REGION Network 20: CHANGE TO BA3 MODE ALARM
   RUNG wire#powerrail
      Contact( #MODE_GROUP_BA_DB.BA3_REQUEST )
      Contact( #ANY_MCH_CYCLE_RUN )
      wire#w1
      I_Contact( #MODE_GROUP_BA_DB.CHANGE_TO_BA1_ALARM )
      I_Contact( #MODE_GROUP_BA_DB.CHANGE_TO_BA2_ALARM )
      I_Contact( #MODE_GROUP_BA_DB.CHANGE_TO_BA5_ALARM )
      Contact( #O_BYTE_0.CHANGE_MODE_SEOC_ALARM )
      wire#w2
      Coil( #MODE_GROUP_BA_DB.CHANGE_TO_BA3_ALARM )
   END_RUNG
   RUNG wire#powerrail
      Contact( #MODE_GROUP_BA_DB.CHANGE_TO_BA3_ALARM )
      I_Contact( #MCH_RESET_FAULTS )
   END_RUNG wire#w1
   RUNG wire#w2
      Coil( #CHANGE_TO_BA3_MODE_WRN )
   END_RUNG
   // the same network as SCL:
   #MODE_GROUP_BA_DB.CHANGE_TO_BA3_ALARM := ((#MODE_GROUP_BA_DB.BA3_REQUEST AND #ANY_MCH_CYCLE_RUN) OR (#MODE_GROUP_BA_DB.CHANGE_TO_BA3_ALARM AND NOT #MCH_RESET_FAULTS)) AND NOT #MODE_GROUP_BA_DB.CHANGE_TO_BA1_ALARM AND NOT #MODE_GROUP_BA_DB.CHANGE_TO_BA2_ALARM AND NOT #MODE_GROUP_BA_DB.CHANGE_TO_BA5_ALARM AND #O_BYTE_0.CHANGE_MODE_SEOC_ALARM;
   #CHANGE_TO_BA3_MODE_WRN := #MODE_GROUP_BA_DB.CHANGE_TO_BA3_ALARM;
END_REGION

REGION Network 21: CHANGE TO BA5 MODE ALARM
   RUNG wire#powerrail
      Contact( #MODE_GROUP_BA_DB.BA5_REQUEST )
      Contact( #ANY_MCH_CYCLE_RUN )
      wire#w1
      I_Contact( #MODE_GROUP_BA_DB.CHANGE_TO_BA1_ALARM )
      I_Contact( #MODE_GROUP_BA_DB.CHANGE_TO_BA2_ALARM )
      I_Contact( #MODE_GROUP_BA_DB.CHANGE_TO_BA3_ALARM )
      Contact( #O_BYTE_0.CHANGE_MODE_SEOC_ALARM )
      wire#w2
      Coil( #MODE_GROUP_BA_DB.CHANGE_TO_BA5_ALARM )
   END_RUNG
   RUNG wire#powerrail
      Contact( #MODE_GROUP_BA_DB.CHANGE_TO_BA5_ALARM )
      I_Contact( #MCH_RESET_FAULTS )
   END_RUNG wire#w1
   RUNG wire#w2
      Coil( #CHANGE_TO_BA5_MODE_WRN )
   END_RUNG
   // the same network as SCL:
   #MODE_GROUP_BA_DB.CHANGE_TO_BA5_ALARM := ((#MODE_GROUP_BA_DB.BA5_REQUEST AND #ANY_MCH_CYCLE_RUN) OR (#MODE_GROUP_BA_DB.CHANGE_TO_BA5_ALARM AND NOT #MCH_RESET_FAULTS)) AND NOT #MODE_GROUP_BA_DB.CHANGE_TO_BA1_ALARM AND NOT #MODE_GROUP_BA_DB.CHANGE_TO_BA2_ALARM AND NOT #MODE_GROUP_BA_DB.CHANGE_TO_BA3_ALARM AND #O_BYTE_0.CHANGE_MODE_SEOC_ALARM;
   #CHANGE_TO_BA5_MODE_WRN := #MODE_GROUP_BA_DB.CHANGE_TO_BA5_ALARM;
END_REGION

REGION Network 22: STOP END OF CYCLE WARNINGS
   RUNG wire#powerrail
      I_Contact( #MODE_GROUP_BA_DB.CHANGE_TO_BA1_ALARM )
      I_Contact( #MODE_GROUP_BA_DB.CHANGE_TO_BA2_ALARM )
      I_Contact( #MODE_GROUP_BA_DB.CHANGE_TO_BA3_ALARM )
      I_Contact( #MODE_GROUP_BA_DB.CHANGE_TO_BA5_ALARM )
      Not()
      { S7_GenerateENO := "TRUE" } Move(in := #DB_NUMBER, out1 => "DB440_MACHINE_ALARM_DECODING".GLOBAL_ALARMS_MACHINE.ALARM_DECODING)
      S_Coil( "DB440_MACHINE_ALARM_DECODING".ALARMS_CENTRAL.SEOC_WARNING )
   END_RUNG
   // the same network as SCL:
   // ENO of a box is taken as its EN; it also drops when the box reports an error
   IF NOT (NOT #MODE_GROUP_BA_DB.CHANGE_TO_BA1_ALARM AND NOT #MODE_GROUP_BA_DB.CHANGE_TO_BA2_ALARM AND NOT #MODE_GROUP_BA_DB.CHANGE_TO_BA3_ALARM AND NOT #MODE_GROUP_BA_DB.CHANGE_TO_BA5_ALARM) THEN
       "DB440_MACHINE_ALARM_DECODING".GLOBAL_ALARMS_MACHINE.ALARM_DECODING := #DB_NUMBER;
       "DB440_MACHINE_ALARM_DECODING".ALARMS_CENTRAL.SEOC_WARNING := TRUE;
   END_IF;
END_REGION

REGION Network 23: WARNINGS
   RUNG wire#powerrail
      I_Contact( #MODE_GROUP_BA_DB.NO_BA_SELECTED )
      Not()
      Move(in := #DB_NUMBER, out1 => "DB440_MACHINE_ALARM_DECODING".GLOBAL_ALARMS_MACHINE.WARNING_DECODING)
      wire#w1
      S_Coil( "DB440_MACHINE_ALARM_DECODING".ALARMS_CENTRAL.WARNING )
   END_RUNG
   RUNG wire#w1
      N_Trig( #MODE_GROUP_BA_DB.WARNING_GONE )
      Move(in := 0, out1 => "DB440_MACHINE_ALARM_DECODING".GLOBAL_ALARMS_MACHINE.WARNING_DECODING)
      R_Coil( "DB440_MACHINE_ALARM_DECODING".ALARMS_CENTRAL.WARNING )
   END_RUNG
   // the same network as SCL:
   #_w1 := NOT (NOT #MODE_GROUP_BA_DB.NO_BA_SELECTED);
   IF #_w1 THEN
       "DB440_MACHINE_ALARM_DECODING".GLOBAL_ALARMS_MACHINE.WARNING_DECODING := #DB_NUMBER;
       "DB440_MACHINE_ALARM_DECODING".ALARMS_CENTRAL.WARNING := TRUE;
   END_IF;
   #_w2 := NOT #_w1 AND #MODE_GROUP_BA_DB.WARNING_GONE;   // falling edge
   #MODE_GROUP_BA_DB.WARNING_GONE := #_w1;
   IF #_w2 THEN
       "DB440_MACHINE_ALARM_DECODING".GLOBAL_ALARMS_MACHINE.WARNING_DECODING := 0;
       "DB440_MACHINE_ALARM_DECODING".ALARMS_CENTRAL.WARNING := FALSE;
   END_IF;
END_REGION

REGION Network 24: CHANGE MODE GENERAL CONDITIONS HELP
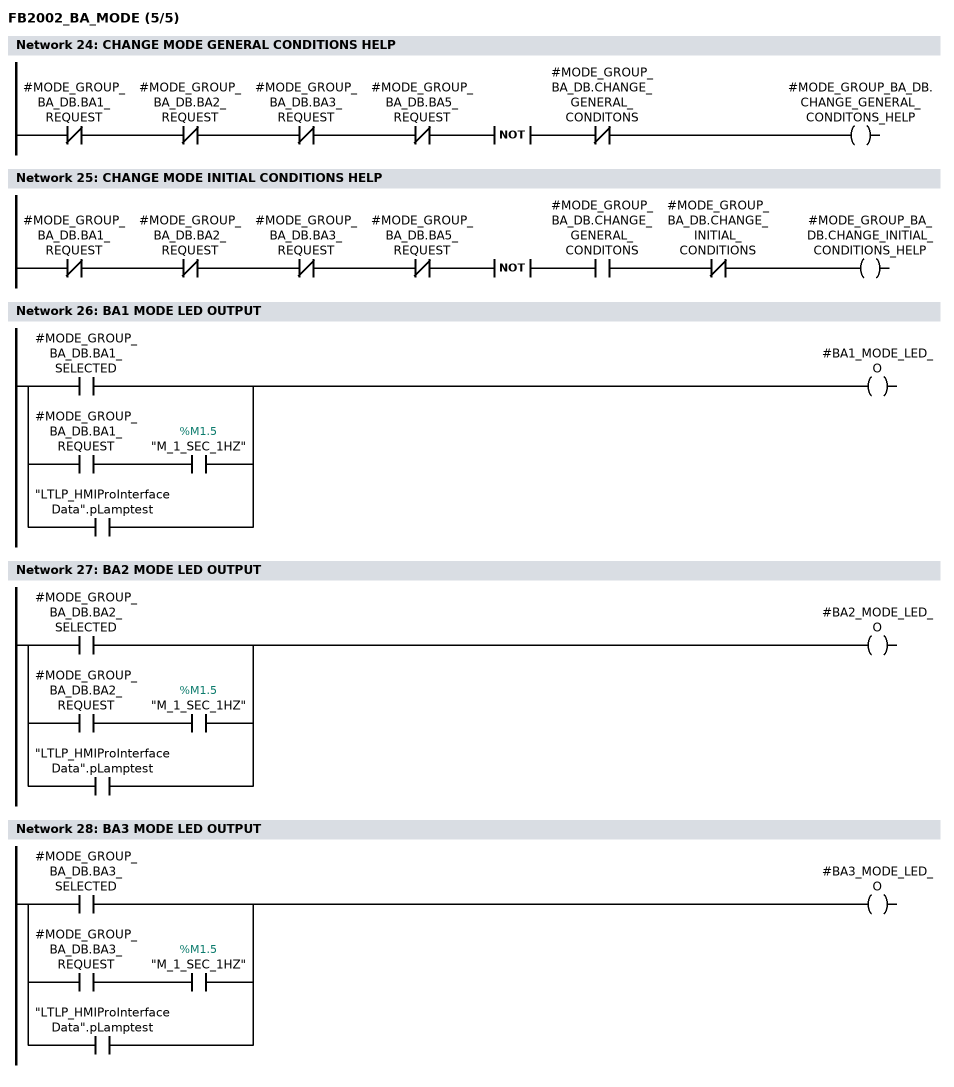
   RUNG wire#powerrail
      I_Contact( #MODE_GROUP_BA_DB.BA1_REQUEST )
      I_Contact( #MODE_GROUP_BA_DB.BA2_REQUEST )
      I_Contact( #MODE_GROUP_BA_DB.BA3_REQUEST )
      I_Contact( #MODE_GROUP_BA_DB.BA5_REQUEST )
      Not()
      I_Contact( #MODE_GROUP_BA_DB.CHANGE_GENERAL_CONDITONS )
      Coil( #MODE_GROUP_BA_DB.CHANGE_GENERAL_CONDITONS_HELP )
   END_RUNG
   // the same network as SCL:
   #MODE_GROUP_BA_DB.CHANGE_GENERAL_CONDITONS_HELP := NOT (NOT #MODE_GROUP_BA_DB.BA1_REQUEST AND NOT #MODE_GROUP_BA_DB.BA2_REQUEST AND NOT #MODE_GROUP_BA_DB.BA3_REQUEST AND NOT #MODE_GROUP_BA_DB.BA5_REQUEST) AND NOT #MODE_GROUP_BA_DB.CHANGE_GENERAL_CONDITONS;
END_REGION

REGION Network 25: CHANGE MODE INITIAL CONDITIONS HELP
   RUNG wire#powerrail
      I_Contact( #MODE_GROUP_BA_DB.BA1_REQUEST )
      I_Contact( #MODE_GROUP_BA_DB.BA2_REQUEST )
      I_Contact( #MODE_GROUP_BA_DB.BA3_REQUEST )
      I_Contact( #MODE_GROUP_BA_DB.BA5_REQUEST )
      Not()
      Contact( #MODE_GROUP_BA_DB.CHANGE_GENERAL_CONDITONS )
      I_Contact( #MODE_GROUP_BA_DB.CHANGE_INITIAL_CONDITIONS )
      Coil( #MODE_GROUP_BA_DB.CHANGE_INITIAL_CONDITIONS_HELP )
   END_RUNG
   // the same network as SCL:
   #MODE_GROUP_BA_DB.CHANGE_INITIAL_CONDITIONS_HELP := NOT (NOT #MODE_GROUP_BA_DB.BA1_REQUEST AND NOT #MODE_GROUP_BA_DB.BA2_REQUEST AND NOT #MODE_GROUP_BA_DB.BA3_REQUEST AND NOT #MODE_GROUP_BA_DB.BA5_REQUEST) AND #MODE_GROUP_BA_DB.CHANGE_GENERAL_CONDITONS AND NOT #MODE_GROUP_BA_DB.CHANGE_INITIAL_CONDITIONS;
END_REGION

REGION Network 26: BA1 MODE LED OUTPUT
   RUNG wire#powerrail
      Contact( #MODE_GROUP_BA_DB.BA1_SELECTED )
      wire#w1
      Coil( #BA1_MODE_LED_O )
   END_RUNG
   RUNG wire#powerrail
      Contact( #MODE_GROUP_BA_DB.BA1_REQUEST )
      Contact( "M_1_SEC_1HZ" )
   END_RUNG wire#w1
   RUNG wire#powerrail
      Contact( "LTLP_HMIProInterfaceData".pLamptest )
   END_RUNG wire#w1
   // the same network as SCL:
   #BA1_MODE_LED_O := #MODE_GROUP_BA_DB.BA1_SELECTED OR (#MODE_GROUP_BA_DB.BA1_REQUEST AND "M_1_SEC_1HZ") OR "LTLP_HMIProInterfaceData".pLamptest;
END_REGION

REGION Network 27: BA2 MODE LED OUTPUT
   RUNG wire#powerrail
      Contact( #MODE_GROUP_BA_DB.BA2_SELECTED )
      wire#w1
      Coil( #BA2_MODE_LED_O )
   END_RUNG
   RUNG wire#powerrail
      Contact( #MODE_GROUP_BA_DB.BA2_REQUEST )
      Contact( "M_1_SEC_1HZ" )
   END_RUNG wire#w1
   RUNG wire#powerrail
      Contact( "LTLP_HMIProInterfaceData".pLamptest )
   END_RUNG wire#w1
   // the same network as SCL:
   #BA2_MODE_LED_O := #MODE_GROUP_BA_DB.BA2_SELECTED OR (#MODE_GROUP_BA_DB.BA2_REQUEST AND "M_1_SEC_1HZ") OR "LTLP_HMIProInterfaceData".pLamptest;
END_REGION

REGION Network 28: BA3 MODE LED OUTPUT
   RUNG wire#powerrail
      Contact( #MODE_GROUP_BA_DB.BA3_SELECTED )
      wire#w1
      Coil( #BA3_MODE_LED_O )
   END_RUNG
   RUNG wire#powerrail
      Contact( #MODE_GROUP_BA_DB.BA3_REQUEST )
      Contact( "M_1_SEC_1HZ" )
   END_RUNG wire#w1
   RUNG wire#powerrail
      Contact( "LTLP_HMIProInterfaceData".pLamptest )
   END_RUNG wire#w1
   // the same network as SCL:
   #BA3_MODE_LED_O := #MODE_GROUP_BA_DB.BA3_SELECTED OR (#MODE_GROUP_BA_DB.BA3_REQUEST AND "M_1_SEC_1HZ") OR "LTLP_HMIProInterfaceData".pLamptest;
END_REGION
END_FUNCTION_BLOCK

FUNCTION_BLOCK "FB2003_CNC_MODES"   // FB2003, LAD
{ S7_Optimized_Access := 'TRUE' }
VERSION : 0.1
// stored: AutoNumber false, IsIECCheckEnabled false, IsRetainMemResEnabled false, MemoryReserve 100, SetENOAutomatically false, UDAEnableTagReadback false
   VAR_INPUT
      MODE_GROUP_NUMBER { ExternalAccessible := 'False'; ExternalVisible := 'False'; ExternalWritable := 'False'} : Int;   // MODE GROUP NUMBER
      MCH_RESET_FAULTS { ExternalAccessible := 'False'; ExternalVisible := 'False'; ExternalWritable := 'False'} : Bool;   // MACHINE RESET
      MDA_MODE_SLCTD { ExternalAccessible := 'False'; ExternalVisible := 'False'; ExternalWritable := 'False'} : Bool;   // MDA MODE SELECTED
      REF_MODE_SLCTD { ExternalAccessible := 'False'; ExternalVisible := 'False'; ExternalWritable := 'False'} : Bool;   // REFERENCE MODE SELECTED
      MODE_GROUP_GENERAL_DB { ExternalAccessible := 'False'; ExternalVisible := 'False'; ExternalWritable := 'False'} : "AUTO_SINGLE_SEMI_MANUAL";
   END_VAR
   VAR_OUTPUT
      ADDITIONAL_MODE_GROUP { ExternalAccessible := 'False'; ExternalVisible := 'False'; ExternalWritable := 'False'} : Struct
         A_AUTO { ExternalAccessible := 'False'; ExternalVisible := 'False'; ExternalWritable := 'False'} : Bool;
         A_MDA { ExternalAccessible := 'False'; ExternalVisible := 'False'; ExternalWritable := 'False'} : Bool;
         A_JOG { ExternalAccessible := 'False'; ExternalVisible := 'False'; ExternalWritable := 'False'} : Bool;
         f0_3 { ExternalAccessible := 'False'; ExternalVisible := 'False'; ExternalWritable := 'False'} : Bool;
         A_MCDisable { ExternalAccessible := 'False'; ExternalVisible := 'False'; ExternalWritable := 'False'} : Bool;
         A_MGStop { ExternalAccessible := 'False'; ExternalVisible := 'False'; ExternalWritable := 'False'} : Bool;
         A_MGStopASp { ExternalAccessible := 'False'; ExternalVisible := 'False'; ExternalWritable := 'False'} : Bool;
         A_MGReset { ExternalAccessible := 'False'; ExternalVisible := 'False'; ExternalWritable := 'False'} : Bool;
         A_TEACHIN { ExternalAccessible := 'False'; ExternalVisible := 'False'; ExternalWritable := 'False'} : Bool;
         A_REPOS { ExternalAccessible := 'False'; ExternalVisible := 'False'; ExternalWritable := 'False'} : Bool;
         A_REF { ExternalAccessible := 'False'; ExternalVisible := 'False'; ExternalWritable := 'False'} : Bool;
         f1_3 { ExternalAccessible := 'False'; ExternalVisible := 'False'; ExternalWritable := 'False'} : Bool;
         f1_4 { ExternalAccessible := 'False'; ExternalVisible := 'False'; ExternalWritable := 'False'} : Bool;
         f1_5 { ExternalAccessible := 'False'; ExternalVisible := 'False'; ExternalWritable := 'False'} : Bool;
         A_SingleBlock_B { ExternalAccessible := 'False'; ExternalVisible := 'False'; ExternalWritable := 'False'} : Bool;
         A_SingleBlock_A { ExternalAccessible := 'False'; ExternalVisible := 'False'; ExternalWritable := 'False'} : Bool;
         A_INC1 { ExternalAccessible := 'False'; ExternalVisible := 'False'; ExternalWritable := 'False'} : Bool;
         A_INC10 { ExternalAccessible := 'False'; ExternalVisible := 'False'; ExternalWritable := 'False'} : Bool;
         A_INC100 { ExternalAccessible := 'False'; ExternalVisible := 'False'; ExternalWritable := 'False'} : Bool;
         A_INC1000 { ExternalAccessible := 'False'; ExternalVisible := 'False'; ExternalWritable := 'False'} : Bool;
         A_INC10000 { ExternalAccessible := 'False'; ExternalVisible := 'False'; ExternalWritable := 'False'} : Bool;
         A_INCVar { ExternalAccessible := 'False'; ExternalVisible := 'False'; ExternalWritable := 'False'} : Bool;
         A_ContManTravel { ExternalAccessible := 'False'; ExternalVisible := 'False'; ExternalWritable := 'False'} : Bool;
         f2_7 { ExternalAccessible := 'False'; ExternalVisible := 'False'; ExternalWritable := 'False'} : Bool;
         f3 { ExternalAccessible := 'False'; ExternalVisible := 'False'; ExternalWritable := 'False'} : Byte;
         E_MMC_AUTO { ExternalAccessible := 'False'; ExternalVisible := 'False'; ExternalWritable := 'False'} : Bool;
         E_MMC_MDA { ExternalAccessible := 'False'; ExternalVisible := 'False'; ExternalWritable := 'False'} : Bool;
         E_MMC_JOG { ExternalAccessible := 'False'; ExternalVisible := 'False'; ExternalWritable := 'False'} : Bool;
         f4_3 { ExternalAccessible := 'False'; ExternalVisible := 'False'; ExternalWritable := 'False'} : Bool;
         f4_4 { ExternalAccessible := 'False'; ExternalVisible := 'False'; ExternalWritable := 'False'} : Bool;
         f4_5 { ExternalAccessible := 'False'; ExternalVisible := 'False'; ExternalWritable := 'False'} : Bool;
         f4_6 { ExternalAccessible := 'False'; ExternalVisible := 'False'; ExternalWritable := 'False'} : Bool;
         f4_7 { ExternalAccessible := 'False'; ExternalVisible := 'False'; ExternalWritable := 'False'} : Bool;
         E_MMC_TEACHIN { ExternalAccessible := 'False'; ExternalVisible := 'False'; ExternalWritable := 'False'} : Bool;
         E_MMC_REPOS { ExternalAccessible := 'False'; ExternalVisible := 'False'; ExternalWritable := 'False'} : Bool;
         E_MMC_REF { ExternalAccessible := 'False'; ExternalVisible := 'False'; ExternalWritable := 'False'} : Bool;
         f5_3 { ExternalAccessible := 'False'; ExternalVisible := 'False'; ExternalWritable := 'False'} : Bool;
         f5_4 { ExternalAccessible := 'False'; ExternalVisible := 'False'; ExternalWritable := 'False'} : Bool;
         f5_5 { ExternalAccessible := 'False'; ExternalVisible := 'False'; ExternalWritable := 'False'} : Bool;
         f5_6 { ExternalAccessible := 'False'; ExternalVisible := 'False'; ExternalWritable := 'False'} : Bool;
         f5_7 { ExternalAccessible := 'False'; ExternalVisible := 'False'; ExternalWritable := 'False'} : Bool;
         E_AUTO { ExternalAccessible := 'False'; ExternalVisible := 'False'; ExternalWritable := 'False'} : Bool;
         E_MDA { ExternalAccessible := 'False'; ExternalVisible := 'False'; ExternalWritable := 'False'} : Bool;
         E_JOG { ExternalAccessible := 'False'; ExternalVisible := 'False'; ExternalWritable := 'False'} : Bool;
         E_MGOK { ExternalAccessible := 'False'; ExternalVisible := 'False'; ExternalWritable := 'False'} : Bool;
         E_MGreseted { ExternalAccessible := 'False'; ExternalVisible := 'False'; ExternalWritable := 'False'} : Bool;
         E_NCKintJOG { ExternalAccessible := 'False'; ExternalVisible := 'False'; ExternalWritable := 'False'} : Bool;
         f6_6 { ExternalAccessible := 'False'; ExternalVisible := 'False'; ExternalWritable := 'False'} : Bool;
         E_ChanReset { ExternalAccessible := 'False'; ExternalVisible := 'False'; ExternalWritable := 'False'} : Bool;
         E_TEACHIN { ExternalAccessible := 'False'; ExternalVisible := 'False'; ExternalWritable := 'False'} : Bool;
         E_REPOS { ExternalAccessible := 'False'; ExternalVisible := 'False'; ExternalWritable := 'False'} : Bool;
         E_REF { ExternalAccessible := 'False'; ExternalVisible := 'False'; ExternalWritable := 'False'} : Bool;
         f7_3 { ExternalAccessible := 'False'; ExternalVisible := 'False'; ExternalWritable := 'False'} : Bool;
         f7_4 { ExternalAccessible := 'False'; ExternalVisible := 'False'; ExternalWritable := 'False'} : Bool;
         f7_5 { ExternalAccessible := 'False'; ExternalVisible := 'False'; ExternalWritable := 'False'} : Bool;
         f7_6 { ExternalAccessible := 'False'; ExternalVisible := 'False'; ExternalWritable := 'False'} : Bool;
         f7_7 { ExternalAccessible := 'False'; ExternalVisible := 'False'; ExternalWritable := 'False'} : Bool;
         E_INC1 { ExternalAccessible := 'False'; ExternalVisible := 'False'; ExternalWritable := 'False'} : Bool;
         E_INC10 { ExternalAccessible := 'False'; ExternalVisible := 'False'; ExternalWritable := 'False'} : Bool;
         E_INC100 { ExternalAccessible := 'False'; ExternalVisible := 'False'; ExternalWritable := 'False'} : Bool;
         E_INC1000 { ExternalAccessible := 'False'; ExternalVisible := 'False'; ExternalWritable := 'False'} : Bool;
         E_INC10000 { ExternalAccessible := 'False'; ExternalVisible := 'False'; ExternalWritable := 'False'} : Bool;
         E_INCVar { ExternalAccessible := 'False'; ExternalVisible := 'False'; ExternalWritable := 'False'} : Bool;
         E_ContManTravelAct { ExternalAccessible := 'False'; ExternalVisible := 'False'; ExternalWritable := 'False'} : Bool;
         f8_7 { ExternalAccessible := 'False'; ExternalVisible := 'False'; ExternalWritable := 'False'} : Bool;
         f9 { ExternalAccessible := 'False'; ExternalVisible := 'False'; ExternalWritable := 'False'} : Byte;
         E_HMI_INC1 { ExternalAccessible := 'False'; ExternalVisible := 'False'; ExternalWritable := 'False'} : Bool;
         E_HMI_INC10 { ExternalAccessible := 'False'; ExternalVisible := 'False'; ExternalWritable := 'False'} : Bool;
         E_HMI_INC100 { ExternalAccessible := 'False'; ExternalVisible := 'False'; ExternalWritable := 'False'} : Bool;
         E_HMI_INC1000 { ExternalAccessible := 'False'; ExternalVisible := 'False'; ExternalWritable := 'False'} : Bool;
         E_HMI_INC10000 { ExternalAccessible := 'False'; ExternalVisible := 'False'; ExternalWritable := 'False'} : Bool;
         E_HMI_INCVar { ExternalAccessible := 'False'; ExternalVisible := 'False'; ExternalWritable := 'False'} : Bool;
         E_HMI_ContManTravel { ExternalAccessible := 'False'; ExternalVisible := 'False'; ExternalWritable := 'False'} : Bool;
         f10_7 { ExternalAccessible := 'False'; ExternalVisible := 'False'; ExternalWritable := 'False'} : Bool;
         f11 { ExternalAccessible := 'False'; ExternalVisible := 'False'; ExternalWritable := 'False'} : Byte;
         f12 { ExternalAccessible := 'False'; ExternalVisible := 'False'; ExternalWritable := 'False'} : Array[12..19] of Byte;
      END_STRUCT;
   END_VAR
   VAR_TEMP   // added for the SCL form of the ladder/FBD networks
      _w1 : Bool;
   END_VAR
BEGIN

NETWORK
TITLE = ACTUAL VALUE IN WCS 0=MCS / Actual value in WCS 0=MCS
// WKS/MKS

      AN    "LBP_HMI".E_ActWCS;
      JC    M001;
      AN    "LBP_HMI".A_ActWCS;
      =     "LBP_HMI".A_ActWCS;
      CLR;
      =     "LBP_HMI".E_ActWCS;
M001: NOP   0;

REGION Network 2: MODE GROUP RESET / Mode group reset
   // BAG Reset
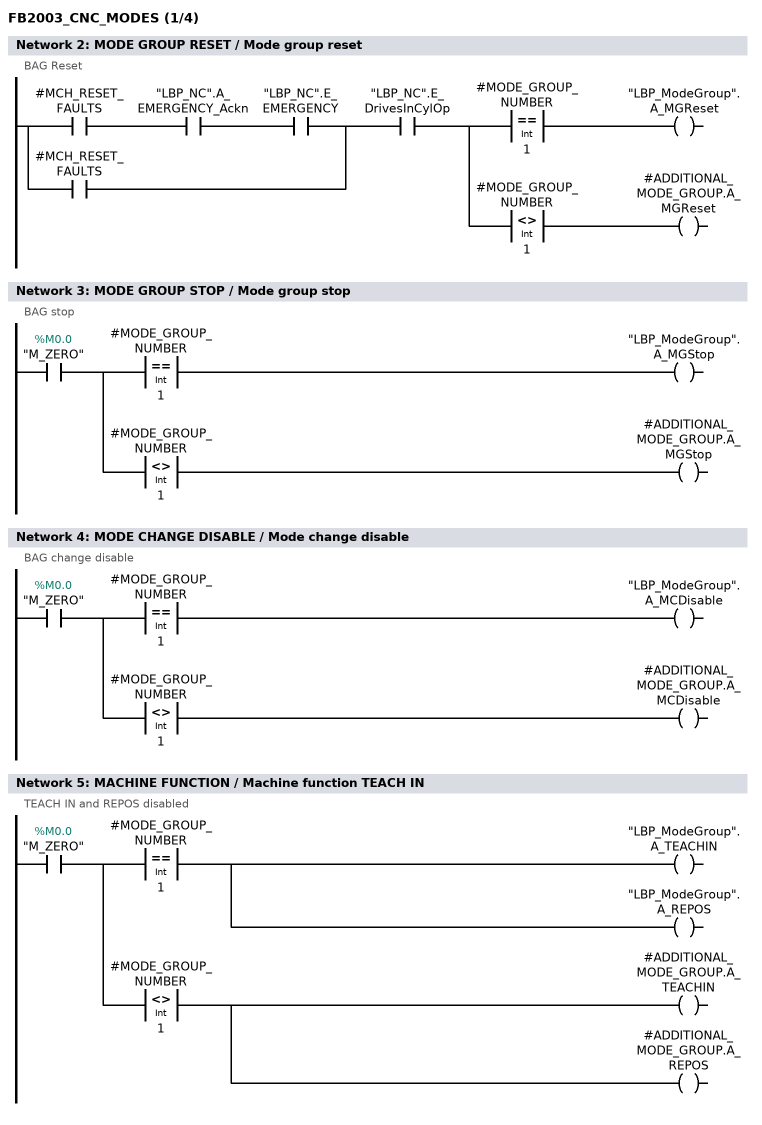
   RUNG wire#powerrail
      Contact( #MCH_RESET_FAULTS )
      Contact( "LBP_NC".A_EMERGENCY_Ackn )
      Contact( "LBP_NC".E_EMERGENCY )
      wire#w1
      Contact( "LBP_NC".E_DrivesInCylOp )
      wire#w2
      { S7_Templates := "SrcType := Int" } EQ_Contact(in1 := #MODE_GROUP_NUMBER, in2 := 1)
      Coil( "LBP_ModeGroup".A_MGReset )
   END_RUNG
   RUNG wire#powerrail
      Contact( #MCH_RESET_FAULTS )
   END_RUNG wire#w1
   RUNG wire#w2
      { S7_Templates := "SrcType := Int" } NE_Contact(in1 := #MODE_GROUP_NUMBER, in2 := 1)
      Coil( #ADDITIONAL_MODE_GROUP.A_MGReset )
   END_RUNG
   // the same network as SCL:
   #_w1 := ((#MCH_RESET_FAULTS AND "LBP_NC".A_EMERGENCY_Ackn AND "LBP_NC".E_EMERGENCY) OR #MCH_RESET_FAULTS) AND "LBP_NC".E_DrivesInCylOp;
   "LBP_ModeGroup".A_MGReset := #_w1 AND (#MODE_GROUP_NUMBER = 1);
   #ADDITIONAL_MODE_GROUP.A_MGReset := #_w1 AND (#MODE_GROUP_NUMBER <> 1);
END_REGION

REGION Network 3: MODE GROUP STOP / Mode group stop
   // BAG stop
   RUNG wire#powerrail
      Contact( "M_ZERO" )
      wire#w1
      { S7_Templates := "SrcType := Int" } EQ_Contact(in1 := #MODE_GROUP_NUMBER, in2 := 1)
      Coil( "LBP_ModeGroup".A_MGStop )
   END_RUNG
   RUNG wire#w1
      { S7_Templates := "SrcType := Int" } NE_Contact(in1 := #MODE_GROUP_NUMBER, in2 := 1)
      Coil( #ADDITIONAL_MODE_GROUP.A_MGStop )
   END_RUNG
   // the same network as SCL:
   "LBP_ModeGroup".A_MGStop := "M_ZERO" AND (#MODE_GROUP_NUMBER = 1);
   #ADDITIONAL_MODE_GROUP.A_MGStop := "M_ZERO" AND (#MODE_GROUP_NUMBER <> 1);
END_REGION

REGION Network 4: MODE CHANGE DISABLE / Mode change disable
   // BAG change disable
   RUNG wire#powerrail
      Contact( "M_ZERO" )
      wire#w1
      { S7_Templates := "SrcType := Int" } EQ_Contact(in1 := #MODE_GROUP_NUMBER, in2 := 1)
      Coil( "LBP_ModeGroup".A_MCDisable )
   END_RUNG
   RUNG wire#w1
      { S7_Templates := "SrcType := Int" } NE_Contact(in1 := #MODE_GROUP_NUMBER, in2 := 1)
      Coil( #ADDITIONAL_MODE_GROUP.A_MCDisable )
   END_RUNG
   // the same network as SCL:
   "LBP_ModeGroup".A_MCDisable := "M_ZERO" AND (#MODE_GROUP_NUMBER = 1);
   #ADDITIONAL_MODE_GROUP.A_MCDisable := "M_ZERO" AND (#MODE_GROUP_NUMBER <> 1);
END_REGION

REGION Network 5: MACHINE FUNCTION / Machine function TEACH IN
   // TEACH IN and REPOS disabled
   RUNG wire#powerrail
      Contact( "M_ZERO" )
      wire#w1
      { S7_Templates := "SrcType := Int" } EQ_Contact(in1 := #MODE_GROUP_NUMBER, in2 := 1)
      wire#w2
      Coil( "LBP_ModeGroup".A_TEACHIN )
   END_RUNG
   RUNG wire#w2
      Coil( "LBP_ModeGroup".A_REPOS )
   END_RUNG
   RUNG wire#w1
      { S7_Templates := "SrcType := Int" } NE_Contact(in1 := #MODE_GROUP_NUMBER, in2 := 1)
      wire#w3
      Coil( #ADDITIONAL_MODE_GROUP.A_TEACHIN )
   END_RUNG
   RUNG wire#w3
      Coil( #ADDITIONAL_MODE_GROUP.A_REPOS )
   END_RUNG
   // the same network as SCL:
   "LBP_ModeGroup".A_TEACHIN := "M_ZERO" AND (#MODE_GROUP_NUMBER = 1);
   "LBP_ModeGroup".A_REPOS := "LBP_ModeGroup".A_TEACHIN;
   #ADDITIONAL_MODE_GROUP.A_TEACHIN := "M_ZERO" AND (#MODE_GROUP_NUMBER <> 1);
   #ADDITIONAL_MODE_GROUP.A_REPOS := #ADDITIONAL_MODE_GROUP.A_TEACHIN;
END_REGION

REGION Network 6: OPERATING MODE AUTOMATIC / AUTOMATIC MODE
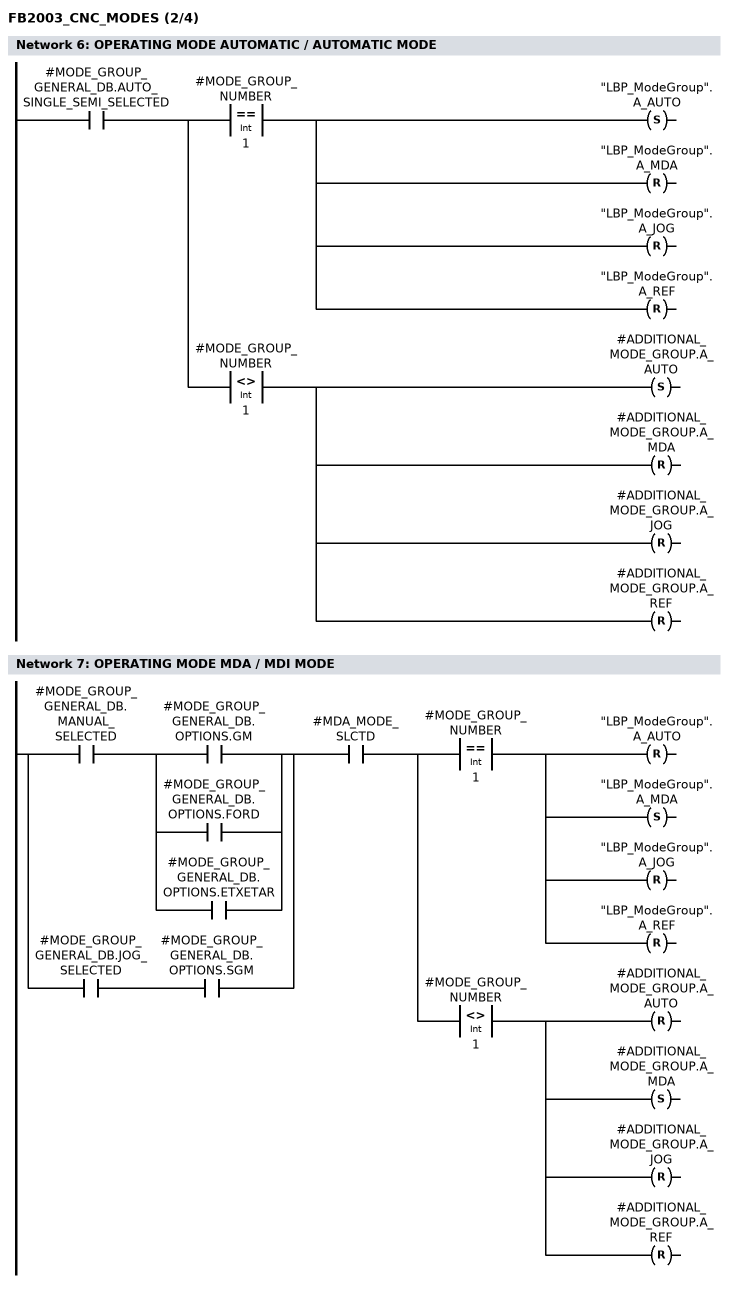
   RUNG wire#powerrail
      Contact( #MODE_GROUP_GENERAL_DB.AUTO_SINGLE_SEMI_SELECTED )
      wire#w1
      { S7_Templates := "SrcType := Int" } EQ_Contact(in1 := #MODE_GROUP_NUMBER, in2 := 1)
      wire#w2
      S_Coil( "LBP_ModeGroup".A_AUTO )
   END_RUNG
   RUNG wire#w2
      R_Coil( "LBP_ModeGroup".A_MDA )
   END_RUNG
   RUNG wire#w2
      R_Coil( "LBP_ModeGroup".A_JOG )
   END_RUNG
   RUNG wire#w2
      R_Coil( "LBP_ModeGroup".A_REF )
   END_RUNG
   RUNG wire#w1
      { S7_Templates := "SrcType := Int" } NE_Contact(in1 := #MODE_GROUP_NUMBER, in2 := 1)
      wire#w3
      S_Coil( #ADDITIONAL_MODE_GROUP.A_AUTO )
   END_RUNG
   RUNG wire#w3
      R_Coil( #ADDITIONAL_MODE_GROUP.A_MDA )
   END_RUNG
   RUNG wire#w3
      R_Coil( #ADDITIONAL_MODE_GROUP.A_JOG )
   END_RUNG
   RUNG wire#w3
      R_Coil( #ADDITIONAL_MODE_GROUP.A_REF )
   END_RUNG
   // the same network as SCL:
   IF #MODE_GROUP_GENERAL_DB.AUTO_SINGLE_SEMI_SELECTED AND (#MODE_GROUP_NUMBER = 1) THEN
       "LBP_ModeGroup".A_AUTO := TRUE;
       "LBP_ModeGroup".A_MDA := FALSE;
       "LBP_ModeGroup".A_JOG := FALSE;
       "LBP_ModeGroup".A_REF := FALSE;
   END_IF;
   IF #MODE_GROUP_GENERAL_DB.AUTO_SINGLE_SEMI_SELECTED AND (#MODE_GROUP_NUMBER <> 1) THEN
       #ADDITIONAL_MODE_GROUP.A_AUTO := TRUE;
       #ADDITIONAL_MODE_GROUP.A_MDA := FALSE;
       #ADDITIONAL_MODE_GROUP.A_JOG := FALSE;
       #ADDITIONAL_MODE_GROUP.A_REF := FALSE;
   END_IF;
END_REGION

REGION Network 7: OPERATING MODE MDA / MDI MODE
   RUNG wire#powerrail
      Contact( #MODE_GROUP_GENERAL_DB.MANUAL_SELECTED )
      wire#w1
      Contact( #MODE_GROUP_GENERAL_DB.OPTIONS.GM )
      wire#w2
      Contact( #MDA_MODE_SLCTD )
      wire#w3
      { S7_Templates := "SrcType := Int" } EQ_Contact(in1 := #MODE_GROUP_NUMBER, in2 := 1)
      wire#w4
      R_Coil( "LBP_ModeGroup".A_AUTO )
   END_RUNG
   RUNG wire#w1
      Contact( #MODE_GROUP_GENERAL_DB.OPTIONS.FORD )
   END_RUNG wire#w2
   RUNG wire#w1
      Contact( #MODE_GROUP_GENERAL_DB.OPTIONS.ETXETAR )
   END_RUNG wire#w2
   RUNG wire#powerrail
      Contact( #MODE_GROUP_GENERAL_DB.JOG_SELECTED )
      Contact( #MODE_GROUP_GENERAL_DB.OPTIONS.SGM )
   END_RUNG wire#w2
   RUNG wire#w4
      S_Coil( "LBP_ModeGroup".A_MDA )
   END_RUNG
   RUNG wire#w4
      R_Coil( "LBP_ModeGroup".A_JOG )
   END_RUNG
   RUNG wire#w4
      R_Coil( "LBP_ModeGroup".A_REF )
   END_RUNG
   RUNG wire#w3
      { S7_Templates := "SrcType := Int" } NE_Contact(in1 := #MODE_GROUP_NUMBER, in2 := 1)
      wire#w5
      R_Coil( #ADDITIONAL_MODE_GROUP.A_AUTO )
   END_RUNG
   RUNG wire#w5
      S_Coil( #ADDITIONAL_MODE_GROUP.A_MDA )
   END_RUNG
   RUNG wire#w5
      R_Coil( #ADDITIONAL_MODE_GROUP.A_JOG )
   END_RUNG
   RUNG wire#w5
      R_Coil( #ADDITIONAL_MODE_GROUP.A_REF )
   END_RUNG
   // the same network as SCL:
   #_w1 := ((#MODE_GROUP_GENERAL_DB.MANUAL_SELECTED AND (#MODE_GROUP_GENERAL_DB.OPTIONS.GM OR #MODE_GROUP_GENERAL_DB.OPTIONS.FORD OR #MODE_GROUP_GENERAL_DB.OPTIONS.ETXETAR)) OR (#MODE_GROUP_GENERAL_DB.JOG_SELECTED AND #MODE_GROUP_GENERAL_DB.OPTIONS.SGM)) AND #MDA_MODE_SLCTD;
   IF #_w1 AND (#MODE_GROUP_NUMBER = 1) THEN
       "LBP_ModeGroup".A_AUTO := FALSE;
       "LBP_ModeGroup".A_MDA := TRUE;
       "LBP_ModeGroup".A_JOG := FALSE;
       "LBP_ModeGroup".A_REF := FALSE;
   END_IF;
   IF #_w1 AND (#MODE_GROUP_NUMBER <> 1) THEN
       #ADDITIONAL_MODE_GROUP.A_AUTO := FALSE;
       #ADDITIONAL_MODE_GROUP.A_MDA := TRUE;
       #ADDITIONAL_MODE_GROUP.A_JOG := FALSE;
       #ADDITIONAL_MODE_GROUP.A_REF := FALSE;
   END_IF;
END_REGION

REGION Network 8: OPERATING MODE MANUAL / JOG MODE
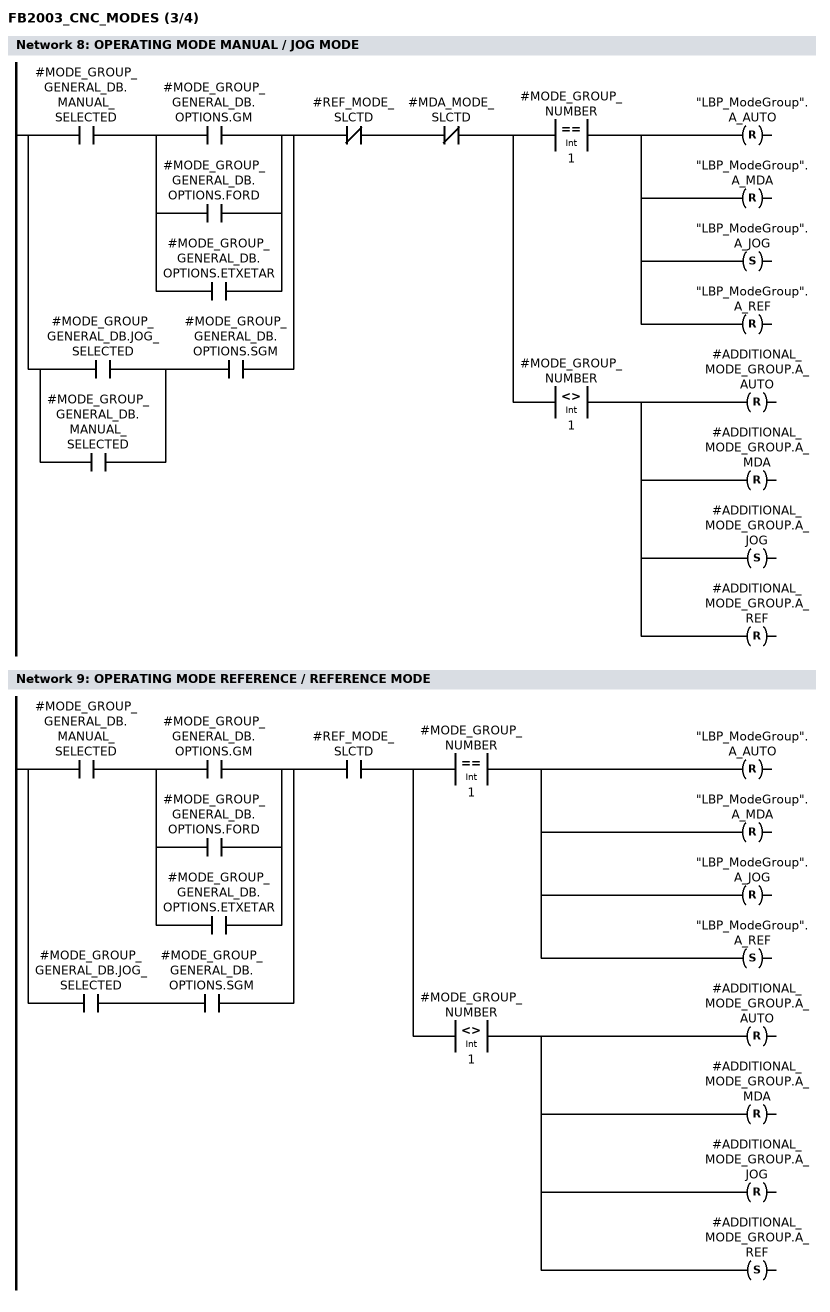
   RUNG wire#powerrail
      Contact( #MODE_GROUP_GENERAL_DB.MANUAL_SELECTED )
      wire#w1
      Contact( #MODE_GROUP_GENERAL_DB.OPTIONS.GM )
      wire#w2
      I_Contact( #REF_MODE_SLCTD )
      I_Contact( #MDA_MODE_SLCTD )
      wire#w4
      { S7_Templates := "SrcType := Int" } EQ_Contact(in1 := #MODE_GROUP_NUMBER, in2 := 1)
      wire#w5
      R_Coil( "LBP_ModeGroup".A_AUTO )
   END_RUNG
   RUNG wire#w1
      Contact( #MODE_GROUP_GENERAL_DB.OPTIONS.FORD )
   END_RUNG wire#w2
   RUNG wire#w1
      Contact( #MODE_GROUP_GENERAL_DB.OPTIONS.ETXETAR )
   END_RUNG wire#w2
   RUNG wire#powerrail
      Contact( #MODE_GROUP_GENERAL_DB.JOG_SELECTED )
      wire#w3
      Contact( #MODE_GROUP_GENERAL_DB.OPTIONS.SGM )
   END_RUNG wire#w2
   RUNG wire#powerrail
      Contact( #MODE_GROUP_GENERAL_DB.MANUAL_SELECTED )
   END_RUNG wire#w3
   RUNG wire#w5
      R_Coil( "LBP_ModeGroup".A_MDA )
   END_RUNG
   RUNG wire#w5
      S_Coil( "LBP_ModeGroup".A_JOG )
   END_RUNG
   RUNG wire#w5
      R_Coil( "LBP_ModeGroup".A_REF )
   END_RUNG
   RUNG wire#w4
      { S7_Templates := "SrcType := Int" } NE_Contact(in1 := #MODE_GROUP_NUMBER, in2 := 1)
      wire#w6
      R_Coil( #ADDITIONAL_MODE_GROUP.A_AUTO )
   END_RUNG
   RUNG wire#w6
      R_Coil( #ADDITIONAL_MODE_GROUP.A_MDA )
   END_RUNG
   RUNG wire#w6
      S_Coil( #ADDITIONAL_MODE_GROUP.A_JOG )
   END_RUNG
   RUNG wire#w6
      R_Coil( #ADDITIONAL_MODE_GROUP.A_REF )
   END_RUNG
   // the same network as SCL:
   #_w1 := ((#MODE_GROUP_GENERAL_DB.MANUAL_SELECTED AND (#MODE_GROUP_GENERAL_DB.OPTIONS.GM OR #MODE_GROUP_GENERAL_DB.OPTIONS.FORD OR #MODE_GROUP_GENERAL_DB.OPTIONS.ETXETAR)) OR ((#MODE_GROUP_GENERAL_DB.JOG_SELECTED OR #MODE_GROUP_GENERAL_DB.MANUAL_SELECTED) AND #MODE_GROUP_GENERAL_DB.OPTIONS.SGM)) AND NOT #REF_MODE_SLCTD AND NOT #MDA_MODE_SLCTD;
   IF #_w1 AND (#MODE_GROUP_NUMBER = 1) THEN
       "LBP_ModeGroup".A_AUTO := FALSE;
       "LBP_ModeGroup".A_MDA := FALSE;
       "LBP_ModeGroup".A_JOG := TRUE;
       "LBP_ModeGroup".A_REF := FALSE;
   END_IF;
   IF #_w1 AND (#MODE_GROUP_NUMBER <> 1) THEN
       #ADDITIONAL_MODE_GROUP.A_AUTO := FALSE;
       #ADDITIONAL_MODE_GROUP.A_MDA := FALSE;
       #ADDITIONAL_MODE_GROUP.A_JOG := TRUE;
       #ADDITIONAL_MODE_GROUP.A_REF := FALSE;
   END_IF;
END_REGION

REGION Network 9: OPERATING MODE REFERENCE / REFERENCE MODE
   RUNG wire#powerrail
      Contact( #MODE_GROUP_GENERAL_DB.MANUAL_SELECTED )
      wire#w1
      Contact( #MODE_GROUP_GENERAL_DB.OPTIONS.GM )
      wire#w2
      Contact( #REF_MODE_SLCTD )
      wire#w3
      { S7_Templates := "SrcType := Int" } EQ_Contact(in1 := #MODE_GROUP_NUMBER, in2 := 1)
      wire#w4
      R_Coil( "LBP_ModeGroup".A_AUTO )
   END_RUNG
   RUNG wire#w1
      Contact( #MODE_GROUP_GENERAL_DB.OPTIONS.FORD )
   END_RUNG wire#w2
   RUNG wire#w1
      Contact( #MODE_GROUP_GENERAL_DB.OPTIONS.ETXETAR )
   END_RUNG wire#w2
   RUNG wire#powerrail
      Contact( #MODE_GROUP_GENERAL_DB.JOG_SELECTED )
      Contact( #MODE_GROUP_GENERAL_DB.OPTIONS.SGM )
   END_RUNG wire#w2
   RUNG wire#w4
      R_Coil( "LBP_ModeGroup".A_MDA )
   END_RUNG
   RUNG wire#w4
      R_Coil( "LBP_ModeGroup".A_JOG )
   END_RUNG
   RUNG wire#w4
      S_Coil( "LBP_ModeGroup".A_REF )
   END_RUNG
   RUNG wire#w3
      { S7_Templates := "SrcType := Int" } NE_Contact(in1 := #MODE_GROUP_NUMBER, in2 := 1)
      wire#w5
      R_Coil( #ADDITIONAL_MODE_GROUP.A_AUTO )
   END_RUNG
   RUNG wire#w5
      R_Coil( #ADDITIONAL_MODE_GROUP.A_MDA )
   END_RUNG
   RUNG wire#w5
      R_Coil( #ADDITIONAL_MODE_GROUP.A_JOG )
   END_RUNG
   RUNG wire#w5
      S_Coil( #ADDITIONAL_MODE_GROUP.A_REF )
   END_RUNG
   // the same network as SCL:
   #_w1 := ((#MODE_GROUP_GENERAL_DB.MANUAL_SELECTED AND (#MODE_GROUP_GENERAL_DB.OPTIONS.GM OR #MODE_GROUP_GENERAL_DB.OPTIONS.FORD OR #MODE_GROUP_GENERAL_DB.OPTIONS.ETXETAR)) OR (#MODE_GROUP_GENERAL_DB.JOG_SELECTED AND #MODE_GROUP_GENERAL_DB.OPTIONS.SGM)) AND #REF_MODE_SLCTD;
   IF #_w1 AND (#MODE_GROUP_NUMBER = 1) THEN
       "LBP_ModeGroup".A_AUTO := FALSE;
       "LBP_ModeGroup".A_MDA := FALSE;
       "LBP_ModeGroup".A_JOG := FALSE;
       "LBP_ModeGroup".A_REF := TRUE;
   END_IF;
   IF #_w1 AND (#MODE_GROUP_NUMBER <> 1) THEN
       #ADDITIONAL_MODE_GROUP.A_AUTO := FALSE;
       #ADDITIONAL_MODE_GROUP.A_MDA := FALSE;
       #ADDITIONAL_MODE_GROUP.A_JOG := FALSE;
       #ADDITIONAL_MODE_GROUP.A_REF := TRUE;
   END_IF;
END_REGION

REGION Network 10: OPERATING MODE NO MODE / NO REFERENCE MODE
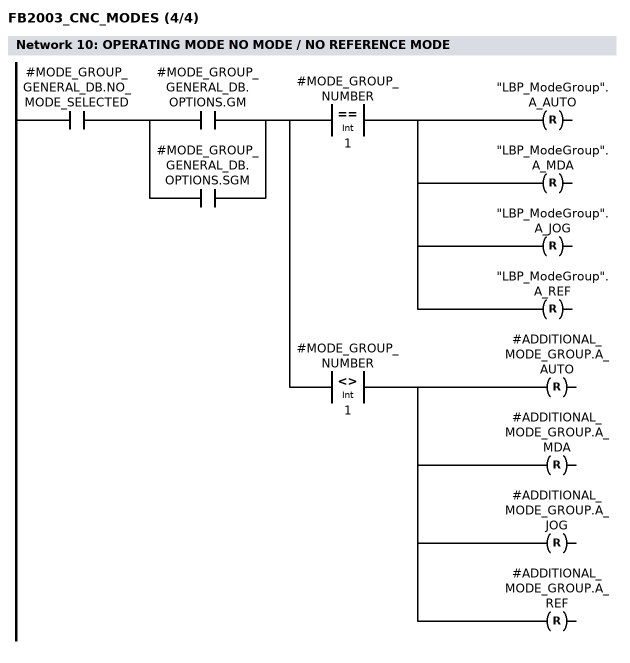
   RUNG wire#powerrail
      Contact( #MODE_GROUP_GENERAL_DB.NO_MODE_SELECTED )
      wire#w1
      Contact( #MODE_GROUP_GENERAL_DB.OPTIONS.GM )
      wire#w2
      { S7_Templates := "SrcType := Int" } EQ_Contact(in1 := #MODE_GROUP_NUMBER, in2 := 1)
      wire#w3
      R_Coil( "LBP_ModeGroup".A_AUTO )
   END_RUNG
   RUNG wire#w1
      Contact( #MODE_GROUP_GENERAL_DB.OPTIONS.SGM )
   END_RUNG wire#w2
   RUNG wire#w3
      R_Coil( "LBP_ModeGroup".A_MDA )
   END_RUNG
   RUNG wire#w3
      R_Coil( "LBP_ModeGroup".A_JOG )
   END_RUNG
   RUNG wire#w3
      R_Coil( "LBP_ModeGroup".A_REF )
   END_RUNG
   RUNG wire#w2
      { S7_Templates := "SrcType := Int" } NE_Contact(in1 := #MODE_GROUP_NUMBER, in2 := 1)
      wire#w4
      R_Coil( #ADDITIONAL_MODE_GROUP.A_AUTO )
   END_RUNG
   RUNG wire#w4
      R_Coil( #ADDITIONAL_MODE_GROUP.A_MDA )
   END_RUNG
   RUNG wire#w4
      R_Coil( #ADDITIONAL_MODE_GROUP.A_JOG )
   END_RUNG
   RUNG wire#w4
      R_Coil( #ADDITIONAL_MODE_GROUP.A_REF )
   END_RUNG
   // the same network as SCL:
   #_w1 := #MODE_GROUP_GENERAL_DB.NO_MODE_SELECTED AND (#MODE_GROUP_GENERAL_DB.OPTIONS.GM OR #MODE_GROUP_GENERAL_DB.OPTIONS.SGM);
   IF #_w1 AND (#MODE_GROUP_NUMBER = 1) THEN
       "LBP_ModeGroup".A_AUTO := FALSE;
       "LBP_ModeGroup".A_MDA := FALSE;
       "LBP_ModeGroup".A_JOG := FALSE;
       "LBP_ModeGroup".A_REF := FALSE;
   END_IF;
   IF #_w1 AND (#MODE_GROUP_NUMBER <> 1) THEN
       #ADDITIONAL_MODE_GROUP.A_AUTO := FALSE;
       #ADDITIONAL_MODE_GROUP.A_MDA := FALSE;
       #ADDITIONAL_MODE_GROUP.A_JOG := FALSE;
       #ADDITIONAL_MODE_GROUP.A_REF := FALSE;
   END_IF;
END_REGION
END_FUNCTION_BLOCK

FUNCTION_BLOCK "FB2005_MDA_MODE"   // FB2005, LAD
{ S7_Optimized_Access := 'FALSE' }
VERSION : 0.1
// stored: AutoNumber false, IsIECCheckEnabled false, SetENOAutomatically false, UDAEnableTagReadback false
   VAR_INPUT
      SAFETY_GATES_CLSD_N_LCKD { ExternalAccessible := 'False'; ExternalVisible := 'False'; ExternalWritable := 'False'} : Bool;   // SAFETY GATES CLOSED AND LOCKED
      ENABLE_REQ { ExternalAccessible := 'False'; ExternalVisible := 'False'; ExternalWritable := 'False'} : Bool;   // ENABLE REQUEST
      DISABLE_REQ { ExternalAccessible := 'False'; ExternalVisible := 'False'; ExternalWritable := 'False'} : Bool;   // DISABLE REQUEST
      MACHINE_SEQ_RUN { ExternalAccessible := 'False'; ExternalVisible := 'False'; ExternalWritable := 'False'} : Bool;   // MACHINE SEQUENCE RUNNING
      ANY_MCH_CYCLE_RUN { ExternalAccessible := 'False'; ExternalVisible := 'False'; ExternalWritable := 'False'} : Bool;   // ANY MACHINE CYCLE RUNNING
   END_VAR
   VAR_OUTPUT
      MDA_MODE_SLCTD_WRN { ExternalAccessible := 'False'; ExternalVisible := 'False'; ExternalWritable := 'False'} : Bool;   // MDA MODE SELECTED WARNING
   END_VAR
   VAR_IN_OUT
      MODE_GROUP_DB : Struct   // MODE GROUP DB
         GENERAL : "AUTO_SINGLE_SEMI_MANUAL";
         STEP_BY_STEP : "MODES";
         MDA : "MODES";
         REFERENCE : "MODES";
         INCREMENTAL : "INCREMENTAL";
         BA : "BA_MODE";
      END_STRUCT;
   END_VAR
   VAR_TEMP
      DB_NUMBER : DInt;   // DB NUMBER FOR ALARM DECODING
   END_VAR
   // // MODE_GROUP_DB.STEP_BY_STEP.MODE_SELECTED : STEP BY STEP MODE SELECTED
   // // MODE_GROUP_DB.MDA.MODE_SELECTED : MDA MODE SELECTED
   // // MODE_GROUP_DB.REFERENCE.MODE_SELECTED : REFERENCE MODE SELECTED
   VAR_TEMP   // added for the SCL form of the ladder/FBD networks
      _w1 : Bool;
      _w2 : Bool;
   END_VAR
BEGIN

NETWORK
TITLE = READ INSTANCE DB
      L     DINO;
      +     10#800000;
      T     #DB_NUMBER;


REGION Network 2: GENERAL CONDITIONS
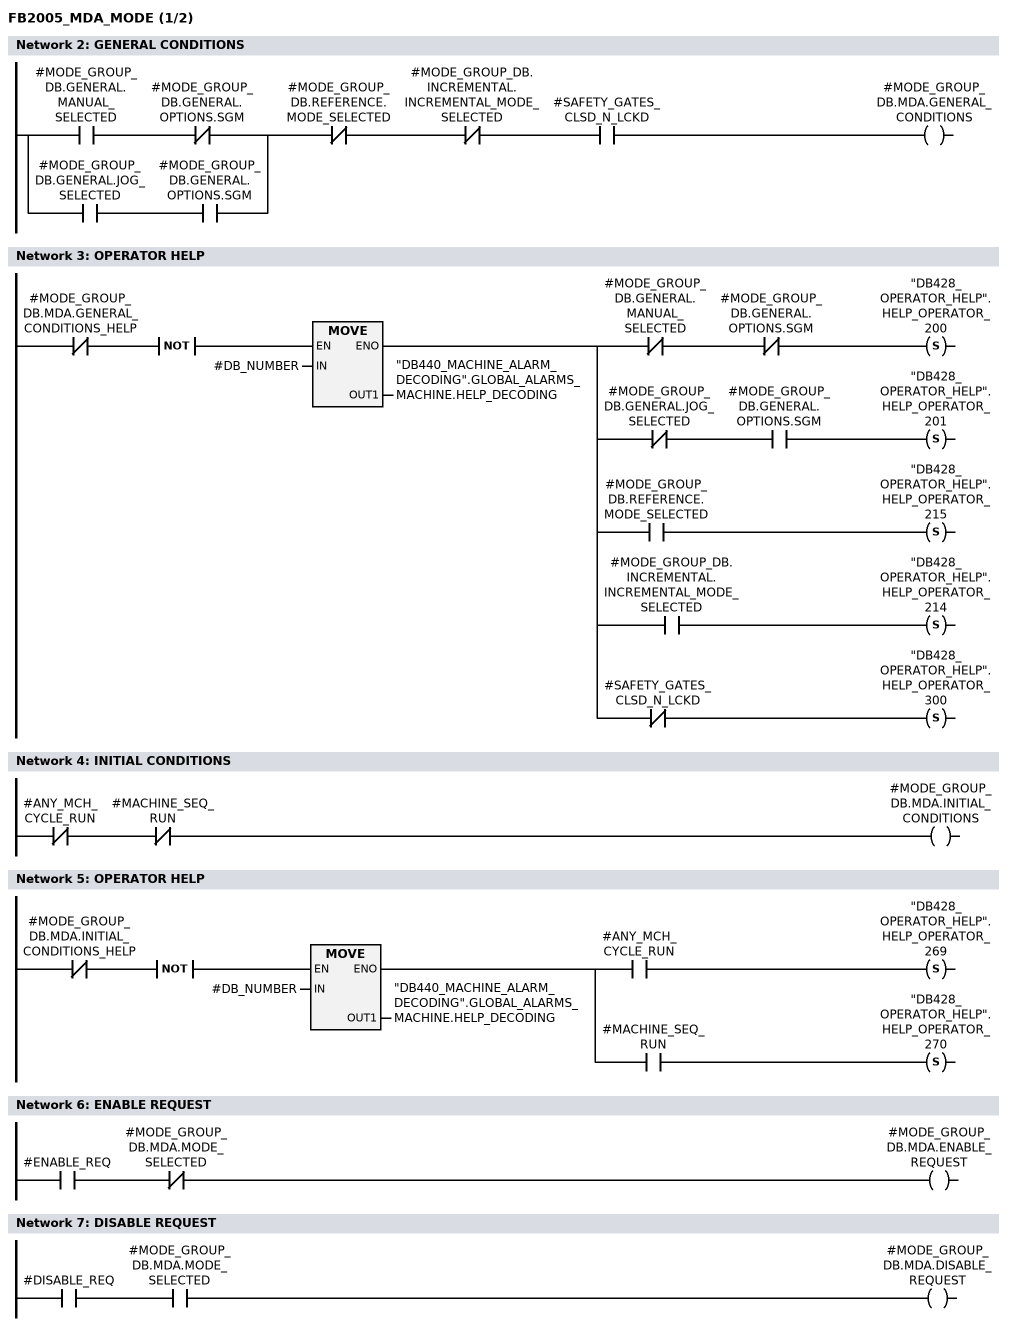
   RUNG wire#powerrail
      Contact( #MODE_GROUP_DB.GENERAL.MANUAL_SELECTED )
      I_Contact( #MODE_GROUP_DB.GENERAL.OPTIONS.SGM )
      wire#w1
      I_Contact( #MODE_GROUP_DB.REFERENCE.MODE_SELECTED )
      I_Contact( #MODE_GROUP_DB.INCREMENTAL.INCREMENTAL_MODE_SELECTED )
      Contact( #SAFETY_GATES_CLSD_N_LCKD )
      Coil( #MODE_GROUP_DB.MDA.GENERAL_CONDITIONS )
   END_RUNG
   RUNG wire#powerrail
      Contact( #MODE_GROUP_DB.GENERAL.JOG_SELECTED )
      Contact( #MODE_GROUP_DB.GENERAL.OPTIONS.SGM )
   END_RUNG wire#w1
   // the same network as SCL:
   #MODE_GROUP_DB.MDA.GENERAL_CONDITIONS := ((#MODE_GROUP_DB.GENERAL.MANUAL_SELECTED AND NOT #MODE_GROUP_DB.GENERAL.OPTIONS.SGM) OR (#MODE_GROUP_DB.GENERAL.JOG_SELECTED AND #MODE_GROUP_DB.GENERAL.OPTIONS.SGM)) AND NOT #MODE_GROUP_DB.REFERENCE.MODE_SELECTED AND NOT #MODE_GROUP_DB.INCREMENTAL.INCREMENTAL_MODE_SELECTED AND #SAFETY_GATES_CLSD_N_LCKD;
END_REGION

REGION Network 3: OPERATOR HELP
   RUNG wire#powerrail
      I_Contact( #MODE_GROUP_DB.MDA.GENERAL_CONDITIONS_HELP )
      Not()
      { S7_GenerateENO := "TRUE" } Move(in := #DB_NUMBER, out1 => "DB440_MACHINE_ALARM_DECODING".GLOBAL_ALARMS_MACHINE.HELP_DECODING)
      wire#w1
      I_Contact( #MODE_GROUP_DB.GENERAL.MANUAL_SELECTED )
      I_Contact( #MODE_GROUP_DB.GENERAL.OPTIONS.SGM )
      S_Coil( "DB428_OPERATOR_HELP".HELP_OPERATOR_200 )
   END_RUNG
   RUNG wire#w1
      I_Contact( #MODE_GROUP_DB.GENERAL.JOG_SELECTED )
      Contact( #MODE_GROUP_DB.GENERAL.OPTIONS.SGM )
      S_Coil( "DB428_OPERATOR_HELP".HELP_OPERATOR_201 )
   END_RUNG
   RUNG wire#w1
      Contact( #MODE_GROUP_DB.REFERENCE.MODE_SELECTED )
      S_Coil( "DB428_OPERATOR_HELP".HELP_OPERATOR_215 )
   END_RUNG
   RUNG wire#w1
      Contact( #MODE_GROUP_DB.INCREMENTAL.INCREMENTAL_MODE_SELECTED )
      S_Coil( "DB428_OPERATOR_HELP".HELP_OPERATOR_214 )
   END_RUNG
   RUNG wire#w1
      I_Contact( #SAFETY_GATES_CLSD_N_LCKD )
      S_Coil( "DB428_OPERATOR_HELP".HELP_OPERATOR_300 )
   END_RUNG
   // the same network as SCL:
   // ENO of a box is taken as its EN; it also drops when the box reports an error
   #_w1 := NOT (NOT #MODE_GROUP_DB.MDA.GENERAL_CONDITIONS_HELP);
   IF #_w1 THEN "DB440_MACHINE_ALARM_DECODING".GLOBAL_ALARMS_MACHINE.HELP_DECODING := #DB_NUMBER; END_IF;
   IF #_w1 AND NOT #MODE_GROUP_DB.GENERAL.MANUAL_SELECTED AND NOT #MODE_GROUP_DB.GENERAL.OPTIONS.SGM THEN
       "DB428_OPERATOR_HELP".HELP_OPERATOR_200 := TRUE;
   END_IF;
   IF #_w1 AND NOT #MODE_GROUP_DB.GENERAL.JOG_SELECTED AND #MODE_GROUP_DB.GENERAL.OPTIONS.SGM THEN
       "DB428_OPERATOR_HELP".HELP_OPERATOR_201 := TRUE;
   END_IF;
   IF #_w1 AND #MODE_GROUP_DB.REFERENCE.MODE_SELECTED THEN
       "DB428_OPERATOR_HELP".HELP_OPERATOR_215 := TRUE;
   END_IF;
   IF #_w1 AND #MODE_GROUP_DB.INCREMENTAL.INCREMENTAL_MODE_SELECTED THEN
       "DB428_OPERATOR_HELP".HELP_OPERATOR_214 := TRUE;
   END_IF;
   IF #_w1 AND NOT #SAFETY_GATES_CLSD_N_LCKD THEN "DB428_OPERATOR_HELP".HELP_OPERATOR_300 := TRUE; END_IF;
END_REGION

REGION Network 4: INITIAL CONDITIONS
   RUNG wire#powerrail
      I_Contact( #ANY_MCH_CYCLE_RUN )
      I_Contact( #MACHINE_SEQ_RUN )
      Coil( #MODE_GROUP_DB.MDA.INITIAL_CONDITIONS )
   END_RUNG
   // the same network as SCL:
   #MODE_GROUP_DB.MDA.INITIAL_CONDITIONS := NOT #ANY_MCH_CYCLE_RUN AND NOT #MACHINE_SEQ_RUN;
END_REGION

REGION Network 5: OPERATOR HELP
   RUNG wire#powerrail
      I_Contact( #MODE_GROUP_DB.MDA.INITIAL_CONDITIONS_HELP )
      Not()
      { S7_GenerateENO := "TRUE" } Move(in := #DB_NUMBER, out1 => "DB440_MACHINE_ALARM_DECODING".GLOBAL_ALARMS_MACHINE.HELP_DECODING)
      wire#w1
      Contact( #ANY_MCH_CYCLE_RUN )
      S_Coil( "DB428_OPERATOR_HELP".HELP_OPERATOR_269 )
   END_RUNG
   RUNG wire#w1
      Contact( #MACHINE_SEQ_RUN )
      S_Coil( "DB428_OPERATOR_HELP".HELP_OPERATOR_270 )
   END_RUNG
   // the same network as SCL:
   // ENO of a box is taken as its EN; it also drops when the box reports an error
   #_w1 := NOT (NOT #MODE_GROUP_DB.MDA.INITIAL_CONDITIONS_HELP);
   IF #_w1 THEN "DB440_MACHINE_ALARM_DECODING".GLOBAL_ALARMS_MACHINE.HELP_DECODING := #DB_NUMBER; END_IF;
   IF #_w1 AND #ANY_MCH_CYCLE_RUN THEN "DB428_OPERATOR_HELP".HELP_OPERATOR_269 := TRUE; END_IF;
   IF #_w1 AND #MACHINE_SEQ_RUN THEN "DB428_OPERATOR_HELP".HELP_OPERATOR_270 := TRUE; END_IF;
END_REGION

REGION Network 6: ENABLE REQUEST
   RUNG wire#powerrail
      Contact( #ENABLE_REQ )
      I_Contact( #MODE_GROUP_DB.MDA.MODE_SELECTED )
      Coil( #MODE_GROUP_DB.MDA.ENABLE_REQUEST )
   END_RUNG
   // the same network as SCL:
   #MODE_GROUP_DB.MDA.ENABLE_REQUEST := #ENABLE_REQ AND NOT #MODE_GROUP_DB.MDA.MODE_SELECTED;
END_REGION

REGION Network 7: DISABLE REQUEST
   RUNG wire#powerrail
      Contact( #DISABLE_REQ )
      Contact( #MODE_GROUP_DB.MDA.MODE_SELECTED )
      Coil( #MODE_GROUP_DB.MDA.DISABLE_REQUEST )
   END_RUNG
   // the same network as SCL:
   #MODE_GROUP_DB.MDA.DISABLE_REQUEST := #DISABLE_REQ AND #MODE_GROUP_DB.MDA.MODE_SELECTED;
END_REGION

REGION Network 8: TOGGLE COMMAND
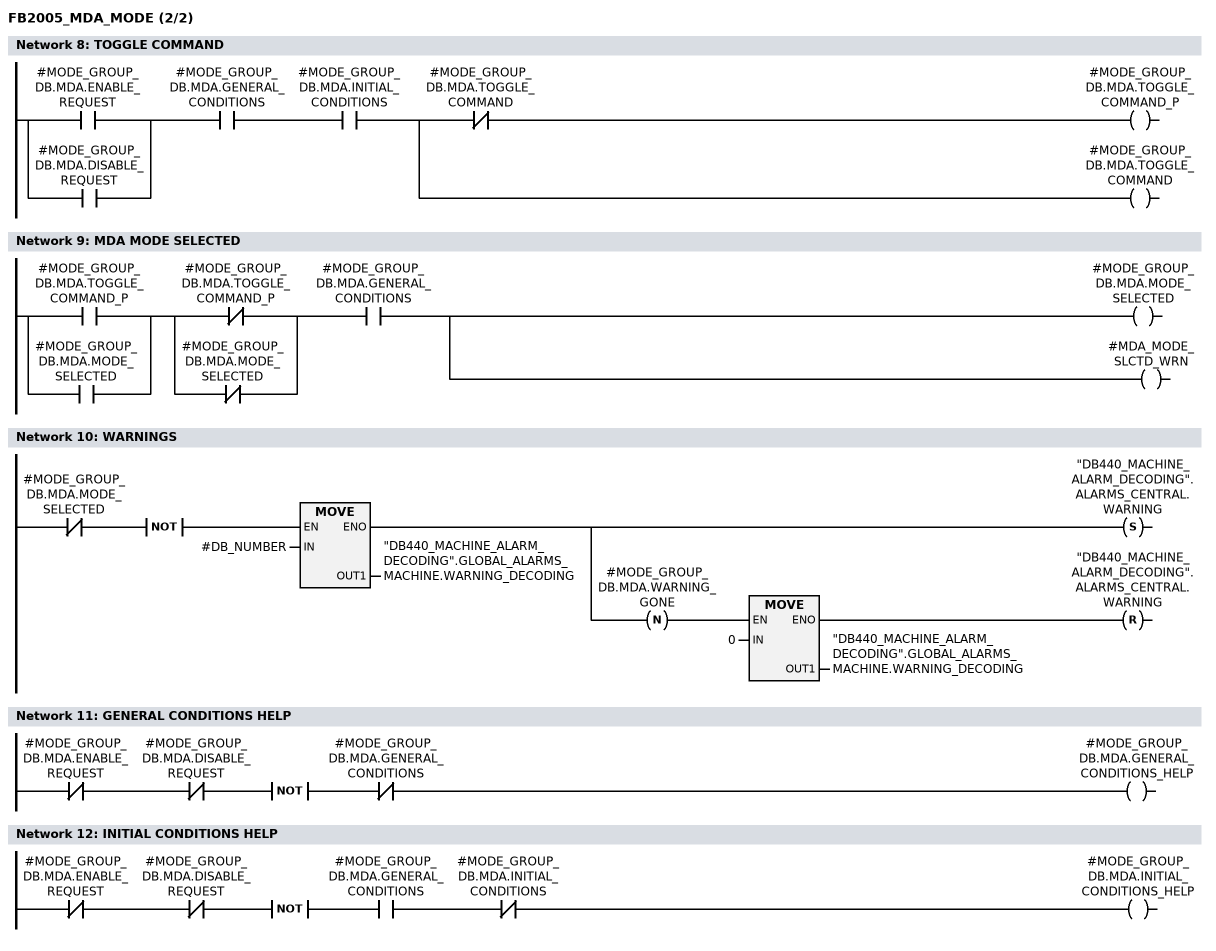
   RUNG wire#powerrail
      Contact( #MODE_GROUP_DB.MDA.ENABLE_REQUEST )
      wire#w1
      Contact( #MODE_GROUP_DB.MDA.GENERAL_CONDITIONS )
      Contact( #MODE_GROUP_DB.MDA.INITIAL_CONDITIONS )
      wire#w2
      I_Contact( #MODE_GROUP_DB.MDA.TOGGLE_COMMAND )
      Coil( #MODE_GROUP_DB.MDA.TOGGLE_COMMAND_P )
   END_RUNG
   RUNG wire#powerrail
      Contact( #MODE_GROUP_DB.MDA.DISABLE_REQUEST )
   END_RUNG wire#w1
   RUNG wire#w2
      Coil( #MODE_GROUP_DB.MDA.TOGGLE_COMMAND )
   END_RUNG
   // the same network as SCL:
   #_w1 := (#MODE_GROUP_DB.MDA.ENABLE_REQUEST OR #MODE_GROUP_DB.MDA.DISABLE_REQUEST) AND #MODE_GROUP_DB.MDA.GENERAL_CONDITIONS AND #MODE_GROUP_DB.MDA.INITIAL_CONDITIONS;
   #MODE_GROUP_DB.MDA.TOGGLE_COMMAND_P := #_w1 AND NOT #MODE_GROUP_DB.MDA.TOGGLE_COMMAND;
   #MODE_GROUP_DB.MDA.TOGGLE_COMMAND := #_w1;
END_REGION

REGION Network 9: MDA MODE SELECTED
   RUNG wire#powerrail
      Contact( #MODE_GROUP_DB.MDA.TOGGLE_COMMAND_P )
      wire#w1
      I_Contact( #MODE_GROUP_DB.MDA.TOGGLE_COMMAND_P )
      wire#w2
      Contact( #MODE_GROUP_DB.MDA.GENERAL_CONDITIONS )
      wire#w3
      Coil( #MODE_GROUP_DB.MDA.MODE_SELECTED )
   END_RUNG
   RUNG wire#powerrail
      Contact( #MODE_GROUP_DB.MDA.MODE_SELECTED )
   END_RUNG wire#w1
   RUNG wire#w1
      I_Contact( #MODE_GROUP_DB.MDA.MODE_SELECTED )
   END_RUNG wire#w2
   RUNG wire#w3
      Coil( #MDA_MODE_SLCTD_WRN )
   END_RUNG
   // the same network as SCL:
   #MODE_GROUP_DB.MDA.MODE_SELECTED := (#MODE_GROUP_DB.MDA.TOGGLE_COMMAND_P OR #MODE_GROUP_DB.MDA.MODE_SELECTED) AND (NOT #MODE_GROUP_DB.MDA.TOGGLE_COMMAND_P OR NOT #MODE_GROUP_DB.MDA.MODE_SELECTED) AND #MODE_GROUP_DB.MDA.GENERAL_CONDITIONS;
   #MDA_MODE_SLCTD_WRN := #MODE_GROUP_DB.MDA.MODE_SELECTED;
END_REGION

REGION Network 10: WARNINGS
   RUNG wire#powerrail
      I_Contact( #MODE_GROUP_DB.MDA.MODE_SELECTED )
      Not()
      Move(in := #DB_NUMBER, out1 => "DB440_MACHINE_ALARM_DECODING".GLOBAL_ALARMS_MACHINE.WARNING_DECODING)
      wire#w1
      S_Coil( "DB440_MACHINE_ALARM_DECODING".ALARMS_CENTRAL.WARNING )
   END_RUNG
   RUNG wire#w1
      N_Trig( #MODE_GROUP_DB.MDA.WARNING_GONE )
      Move(in := 0, out1 => "DB440_MACHINE_ALARM_DECODING".GLOBAL_ALARMS_MACHINE.WARNING_DECODING)
      R_Coil( "DB440_MACHINE_ALARM_DECODING".ALARMS_CENTRAL.WARNING )
   END_RUNG
   // the same network as SCL:
   #_w1 := NOT (NOT #MODE_GROUP_DB.MDA.MODE_SELECTED);
   IF #_w1 THEN
       "DB440_MACHINE_ALARM_DECODING".GLOBAL_ALARMS_MACHINE.WARNING_DECODING := #DB_NUMBER;
       "DB440_MACHINE_ALARM_DECODING".ALARMS_CENTRAL.WARNING := TRUE;
   END_IF;
   #_w2 := NOT #_w1 AND #MODE_GROUP_DB.MDA.WARNING_GONE;   // falling edge
   #MODE_GROUP_DB.MDA.WARNING_GONE := #_w1;
   IF #_w2 THEN
       "DB440_MACHINE_ALARM_DECODING".GLOBAL_ALARMS_MACHINE.WARNING_DECODING := 0;
       "DB440_MACHINE_ALARM_DECODING".ALARMS_CENTRAL.WARNING := FALSE;
   END_IF;
END_REGION

REGION Network 11: GENERAL CONDITIONS HELP
   RUNG wire#powerrail
      I_Contact( #MODE_GROUP_DB.MDA.ENABLE_REQUEST )
      I_Contact( #MODE_GROUP_DB.MDA.DISABLE_REQUEST )
      Not()
      I_Contact( #MODE_GROUP_DB.MDA.GENERAL_CONDITIONS )
      Coil( #MODE_GROUP_DB.MDA.GENERAL_CONDITIONS_HELP )
   END_RUNG
   // the same network as SCL:
   #MODE_GROUP_DB.MDA.GENERAL_CONDITIONS_HELP := NOT (NOT #MODE_GROUP_DB.MDA.ENABLE_REQUEST AND NOT #MODE_GROUP_DB.MDA.DISABLE_REQUEST) AND NOT #MODE_GROUP_DB.MDA.GENERAL_CONDITIONS;
END_REGION

REGION Network 12: INITIAL CONDITIONS HELP
   RUNG wire#powerrail
      I_Contact( #MODE_GROUP_DB.MDA.ENABLE_REQUEST )
      I_Contact( #MODE_GROUP_DB.MDA.DISABLE_REQUEST )
      Not()
      Contact( #MODE_GROUP_DB.MDA.GENERAL_CONDITIONS )
      I_Contact( #MODE_GROUP_DB.MDA.INITIAL_CONDITIONS )
      Coil( #MODE_GROUP_DB.MDA.INITIAL_CONDITIONS_HELP )
   END_RUNG
   // the same network as SCL:
   #MODE_GROUP_DB.MDA.INITIAL_CONDITIONS_HELP := NOT (NOT #MODE_GROUP_DB.MDA.ENABLE_REQUEST AND NOT #MODE_GROUP_DB.MDA.DISABLE_REQUEST) AND #MODE_GROUP_DB.MDA.GENERAL_CONDITIONS AND NOT #MODE_GROUP_DB.MDA.INITIAL_CONDITIONS;
END_REGION
END_FUNCTION_BLOCK

FUNCTION_BLOCK "FB2006_REFERENCE_MODE"   // FB2006, LAD
{ S7_Optimized_Access := 'FALSE' }
VERSION : 0.1
// stored: AutoNumber false, IsIECCheckEnabled false, SetENOAutomatically false, UDAEnableTagReadback false
   VAR_INPUT
      ENABLE_REQ { ExternalAccessible := 'False'; ExternalVisible := 'False'; ExternalWritable := 'False'} : Bool;   // ENABLE_REQUEST
      DISABLE_REQ { ExternalAccessible := 'False'; ExternalVisible := 'False'; ExternalWritable := 'False'} : Bool;   // DISABLE_REQUEST
   END_VAR
   VAR_OUTPUT
      REF_MODE_SLCTD_WRN { ExternalAccessible := 'False'; ExternalVisible := 'False'; ExternalWritable := 'False'} : Bool;   // REFERENCE MODE SELECTED WARNING
   END_VAR
   VAR_IN_OUT
      MODE_GROUP_DB : Struct   // MODE GROUP DB
         GENERAL : "AUTO_SINGLE_SEMI_MANUAL";
         STEP_BY_STEP : "MODES";
         MDA : "MODES";
         REFERENCE : "MODES";
         INCREMENTAL : "INCREMENTAL";
         BA : "BA_MODE";
      END_STRUCT;
   END_VAR
   VAR_TEMP
      DB_NUMBER : DInt;   // DB NUMBER FOR ALARM DECODING
   END_VAR
   // // MODE_GROUP_DB.STEP_BY_STEP.MODE_SELECTED : STEP BY STEP MODE SELECTED
   // // MODE_GROUP_DB.MDA.MODE_SELECTED : MDA MODE SELECTED
   // // MODE_GROUP_DB.REFERENCE.MODE_SELECTED : REFERENCE MODE SELECTED
   VAR_TEMP   // added for the SCL form of the ladder/FBD networks
      _w1 : Bool;
      _w2 : Bool;
   END_VAR
BEGIN

NETWORK
TITLE = READ INSTANCE DB
      L     DINO;
      +     10#800000;
      T     #DB_NUMBER;


REGION Network 2: GENERAL CONDITIONS
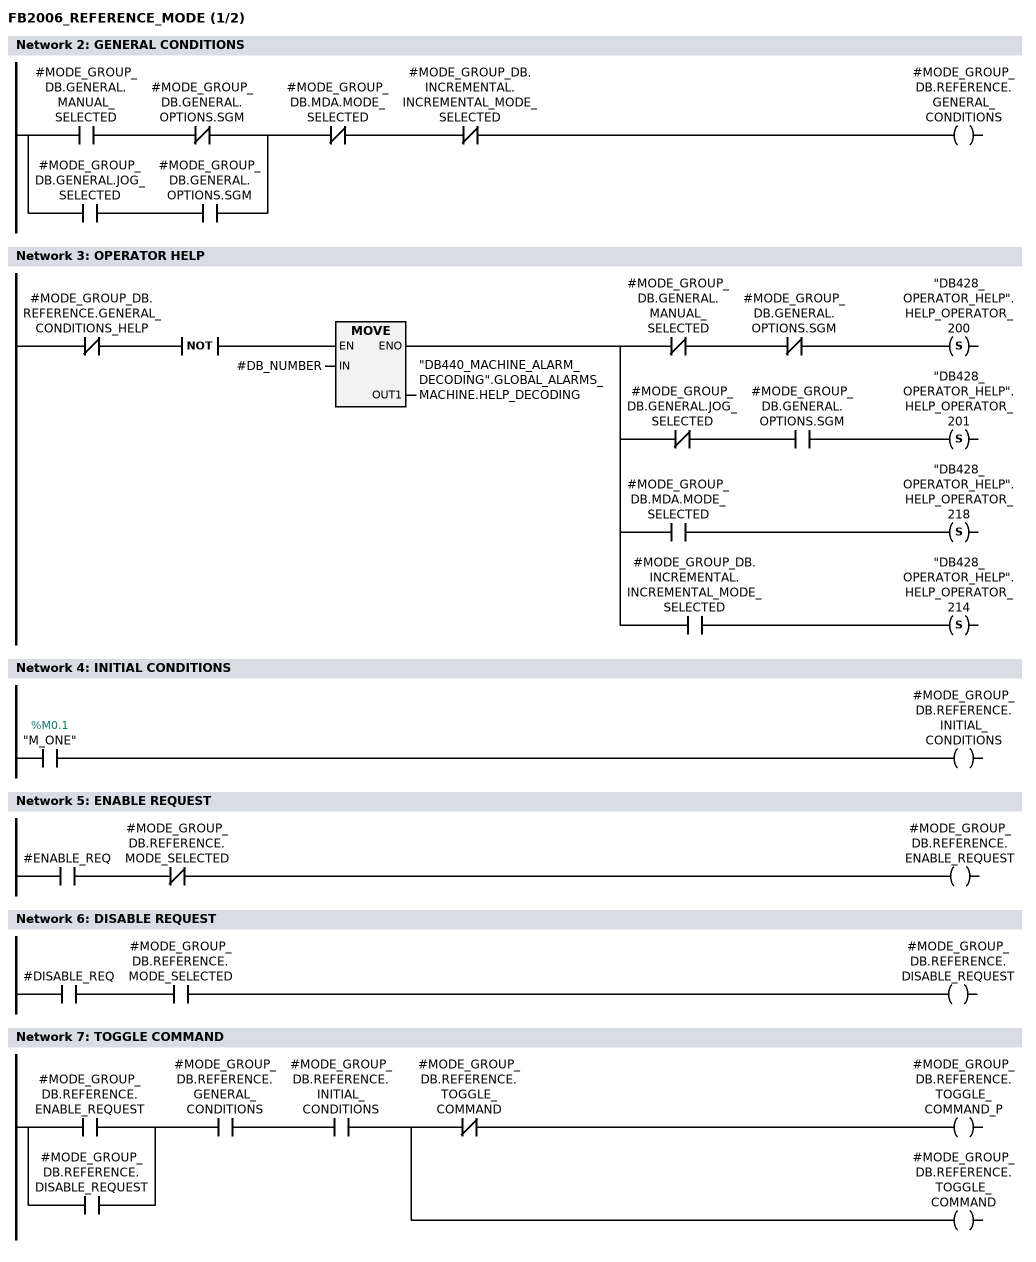
   RUNG wire#powerrail
      Contact( #MODE_GROUP_DB.GENERAL.MANUAL_SELECTED )
      I_Contact( #MODE_GROUP_DB.GENERAL.OPTIONS.SGM )
      wire#w1
      I_Contact( #MODE_GROUP_DB.MDA.MODE_SELECTED )
      I_Contact( #MODE_GROUP_DB.INCREMENTAL.INCREMENTAL_MODE_SELECTED )
      Coil( #MODE_GROUP_DB.REFERENCE.GENERAL_CONDITIONS )
   END_RUNG
   RUNG wire#powerrail
      Contact( #MODE_GROUP_DB.GENERAL.JOG_SELECTED )
      Contact( #MODE_GROUP_DB.GENERAL.OPTIONS.SGM )
   END_RUNG wire#w1
   // the same network as SCL:
   #MODE_GROUP_DB.REFERENCE.GENERAL_CONDITIONS := ((#MODE_GROUP_DB.GENERAL.MANUAL_SELECTED AND NOT #MODE_GROUP_DB.GENERAL.OPTIONS.SGM) OR (#MODE_GROUP_DB.GENERAL.JOG_SELECTED AND #MODE_GROUP_DB.GENERAL.OPTIONS.SGM)) AND NOT #MODE_GROUP_DB.MDA.MODE_SELECTED AND NOT #MODE_GROUP_DB.INCREMENTAL.INCREMENTAL_MODE_SELECTED;
END_REGION

REGION Network 3: OPERATOR HELP
   RUNG wire#powerrail
      I_Contact( #MODE_GROUP_DB.REFERENCE.GENERAL_CONDITIONS_HELP )
      Not()
      { S7_GenerateENO := "TRUE" } Move(in := #DB_NUMBER, out1 => "DB440_MACHINE_ALARM_DECODING".GLOBAL_ALARMS_MACHINE.HELP_DECODING)
      wire#w1
      I_Contact( #MODE_GROUP_DB.GENERAL.MANUAL_SELECTED )
      I_Contact( #MODE_GROUP_DB.GENERAL.OPTIONS.SGM )
      S_Coil( "DB428_OPERATOR_HELP".HELP_OPERATOR_200 )
   END_RUNG
   RUNG wire#w1
      I_Contact( #MODE_GROUP_DB.GENERAL.JOG_SELECTED )
      Contact( #MODE_GROUP_DB.GENERAL.OPTIONS.SGM )
      S_Coil( "DB428_OPERATOR_HELP".HELP_OPERATOR_201 )
   END_RUNG
   RUNG wire#w1
      Contact( #MODE_GROUP_DB.MDA.MODE_SELECTED )
      S_Coil( "DB428_OPERATOR_HELP".HELP_OPERATOR_218 )
   END_RUNG
   RUNG wire#w1
      Contact( #MODE_GROUP_DB.INCREMENTAL.INCREMENTAL_MODE_SELECTED )
      S_Coil( "DB428_OPERATOR_HELP".HELP_OPERATOR_214 )
   END_RUNG
   // the same network as SCL:
   // ENO of a box is taken as its EN; it also drops when the box reports an error
   #_w1 := NOT (NOT #MODE_GROUP_DB.REFERENCE.GENERAL_CONDITIONS_HELP);
   IF #_w1 THEN "DB440_MACHINE_ALARM_DECODING".GLOBAL_ALARMS_MACHINE.HELP_DECODING := #DB_NUMBER; END_IF;
   IF #_w1 AND NOT #MODE_GROUP_DB.GENERAL.MANUAL_SELECTED AND NOT #MODE_GROUP_DB.GENERAL.OPTIONS.SGM THEN
       "DB428_OPERATOR_HELP".HELP_OPERATOR_200 := TRUE;
   END_IF;
   IF #_w1 AND NOT #MODE_GROUP_DB.GENERAL.JOG_SELECTED AND #MODE_GROUP_DB.GENERAL.OPTIONS.SGM THEN
       "DB428_OPERATOR_HELP".HELP_OPERATOR_201 := TRUE;
   END_IF;
   IF #_w1 AND #MODE_GROUP_DB.MDA.MODE_SELECTED THEN "DB428_OPERATOR_HELP".HELP_OPERATOR_218 := TRUE; END_IF;
   IF #_w1 AND #MODE_GROUP_DB.INCREMENTAL.INCREMENTAL_MODE_SELECTED THEN
       "DB428_OPERATOR_HELP".HELP_OPERATOR_214 := TRUE;
   END_IF;
END_REGION

REGION Network 4: INITIAL CONDITIONS
   RUNG wire#powerrail
      Contact( "M_ONE" )
      Coil( #MODE_GROUP_DB.REFERENCE.INITIAL_CONDITIONS )
   END_RUNG
   // the same network as SCL:
   #MODE_GROUP_DB.REFERENCE.INITIAL_CONDITIONS := "M_ONE";
END_REGION

REGION Network 5: ENABLE REQUEST
   RUNG wire#powerrail
      Contact( #ENABLE_REQ )
      I_Contact( #MODE_GROUP_DB.REFERENCE.MODE_SELECTED )
      Coil( #MODE_GROUP_DB.REFERENCE.ENABLE_REQUEST )
   END_RUNG
   // the same network as SCL:
   #MODE_GROUP_DB.REFERENCE.ENABLE_REQUEST := #ENABLE_REQ AND NOT #MODE_GROUP_DB.REFERENCE.MODE_SELECTED;
END_REGION

REGION Network 6: DISABLE REQUEST
   RUNG wire#powerrail
      Contact( #DISABLE_REQ )
      Contact( #MODE_GROUP_DB.REFERENCE.MODE_SELECTED )
      Coil( #MODE_GROUP_DB.REFERENCE.DISABLE_REQUEST )
   END_RUNG
   // the same network as SCL:
   #MODE_GROUP_DB.REFERENCE.DISABLE_REQUEST := #DISABLE_REQ AND #MODE_GROUP_DB.REFERENCE.MODE_SELECTED;
END_REGION

REGION Network 7: TOGGLE COMMAND
   RUNG wire#powerrail
      Contact( #MODE_GROUP_DB.REFERENCE.ENABLE_REQUEST )
      wire#w1
      Contact( #MODE_GROUP_DB.REFERENCE.GENERAL_CONDITIONS )
      Contact( #MODE_GROUP_DB.REFERENCE.INITIAL_CONDITIONS )
      wire#w2
      I_Contact( #MODE_GROUP_DB.REFERENCE.TOGGLE_COMMAND )
      Coil( #MODE_GROUP_DB.REFERENCE.TOGGLE_COMMAND_P )
   END_RUNG
   RUNG wire#powerrail
      Contact( #MODE_GROUP_DB.REFERENCE.DISABLE_REQUEST )
   END_RUNG wire#w1
   RUNG wire#w2
      Coil( #MODE_GROUP_DB.REFERENCE.TOGGLE_COMMAND )
   END_RUNG
   // the same network as SCL:
   #_w1 := (#MODE_GROUP_DB.REFERENCE.ENABLE_REQUEST OR #MODE_GROUP_DB.REFERENCE.DISABLE_REQUEST) AND #MODE_GROUP_DB.REFERENCE.GENERAL_CONDITIONS AND #MODE_GROUP_DB.REFERENCE.INITIAL_CONDITIONS;
   #MODE_GROUP_DB.REFERENCE.TOGGLE_COMMAND_P := #_w1 AND NOT #MODE_GROUP_DB.REFERENCE.TOGGLE_COMMAND;
   #MODE_GROUP_DB.REFERENCE.TOGGLE_COMMAND := #_w1;
END_REGION

REGION Network 8: REFERENCE MODE SELECTED
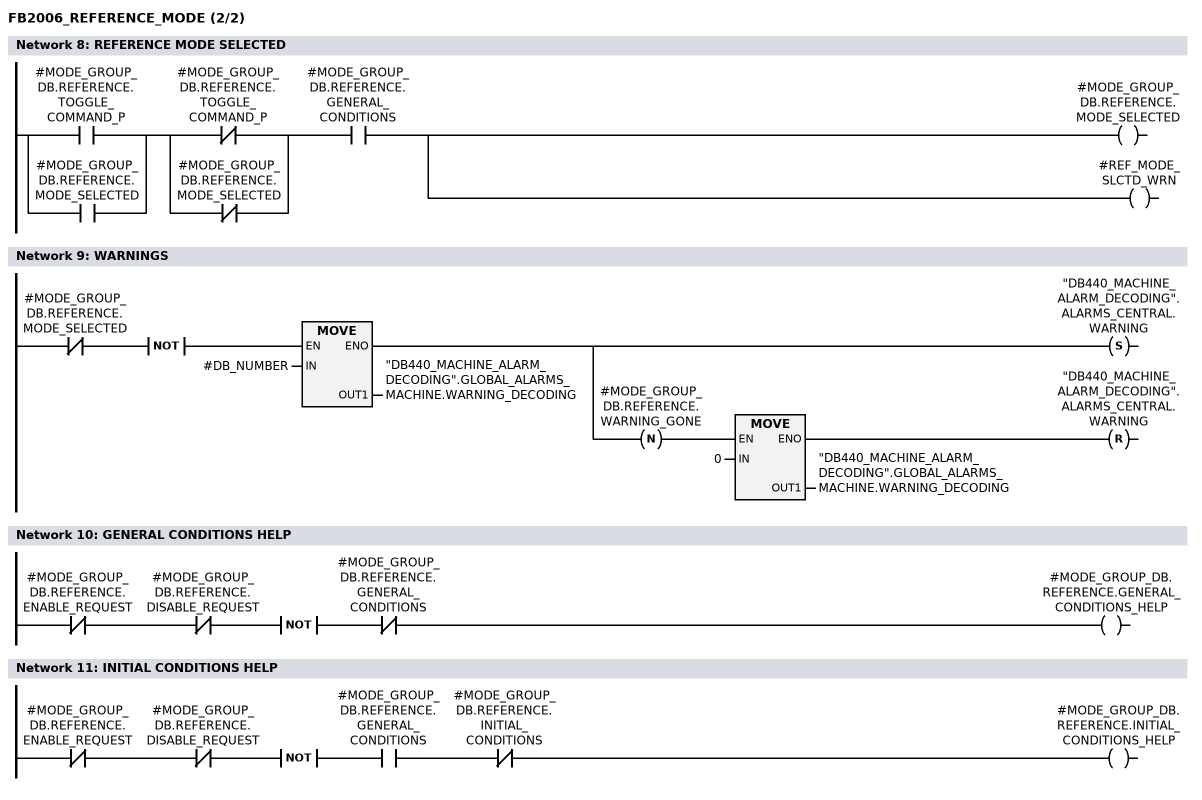
   RUNG wire#powerrail
      Contact( #MODE_GROUP_DB.REFERENCE.TOGGLE_COMMAND_P )
      wire#w1
      I_Contact( #MODE_GROUP_DB.REFERENCE.TOGGLE_COMMAND_P )
      wire#w2
      Contact( #MODE_GROUP_DB.REFERENCE.GENERAL_CONDITIONS )
      wire#w3
      Coil( #MODE_GROUP_DB.REFERENCE.MODE_SELECTED )
   END_RUNG
   RUNG wire#powerrail
      Contact( #MODE_GROUP_DB.REFERENCE.MODE_SELECTED )
   END_RUNG wire#w1
   RUNG wire#w1
      I_Contact( #MODE_GROUP_DB.REFERENCE.MODE_SELECTED )
   END_RUNG wire#w2
   RUNG wire#w3
      Coil( #REF_MODE_SLCTD_WRN )
   END_RUNG
   // the same network as SCL:
   #MODE_GROUP_DB.REFERENCE.MODE_SELECTED := (#MODE_GROUP_DB.REFERENCE.TOGGLE_COMMAND_P OR #MODE_GROUP_DB.REFERENCE.MODE_SELECTED) AND (NOT #MODE_GROUP_DB.REFERENCE.TOGGLE_COMMAND_P OR NOT #MODE_GROUP_DB.REFERENCE.MODE_SELECTED) AND #MODE_GROUP_DB.REFERENCE.GENERAL_CONDITIONS;
   #REF_MODE_SLCTD_WRN := #MODE_GROUP_DB.REFERENCE.MODE_SELECTED;
END_REGION

REGION Network 9: WARNINGS
   RUNG wire#powerrail
      I_Contact( #MODE_GROUP_DB.REFERENCE.MODE_SELECTED )
      Not()
      Move(in := #DB_NUMBER, out1 => "DB440_MACHINE_ALARM_DECODING".GLOBAL_ALARMS_MACHINE.WARNING_DECODING)
      wire#w1
      S_Coil( "DB440_MACHINE_ALARM_DECODING".ALARMS_CENTRAL.WARNING )
   END_RUNG
   RUNG wire#w1
      N_Trig( #MODE_GROUP_DB.REFERENCE.WARNING_GONE )
      Move(in := 0, out1 => "DB440_MACHINE_ALARM_DECODING".GLOBAL_ALARMS_MACHINE.WARNING_DECODING)
      R_Coil( "DB440_MACHINE_ALARM_DECODING".ALARMS_CENTRAL.WARNING )
   END_RUNG
   // the same network as SCL:
   #_w1 := NOT (NOT #MODE_GROUP_DB.REFERENCE.MODE_SELECTED);
   IF #_w1 THEN
       "DB440_MACHINE_ALARM_DECODING".GLOBAL_ALARMS_MACHINE.WARNING_DECODING := #DB_NUMBER;
       "DB440_MACHINE_ALARM_DECODING".ALARMS_CENTRAL.WARNING := TRUE;
   END_IF;
   #_w2 := NOT #_w1 AND #MODE_GROUP_DB.REFERENCE.WARNING_GONE;   // falling edge
   #MODE_GROUP_DB.REFERENCE.WARNING_GONE := #_w1;
   IF #_w2 THEN
       "DB440_MACHINE_ALARM_DECODING".GLOBAL_ALARMS_MACHINE.WARNING_DECODING := 0;
       "DB440_MACHINE_ALARM_DECODING".ALARMS_CENTRAL.WARNING := FALSE;
   END_IF;
END_REGION

REGION Network 10: GENERAL CONDITIONS HELP
   RUNG wire#powerrail
      I_Contact( #MODE_GROUP_DB.REFERENCE.ENABLE_REQUEST )
      I_Contact( #MODE_GROUP_DB.REFERENCE.DISABLE_REQUEST )
      Not()
      I_Contact( #MODE_GROUP_DB.REFERENCE.GENERAL_CONDITIONS )
      Coil( #MODE_GROUP_DB.REFERENCE.GENERAL_CONDITIONS_HELP )
   END_RUNG
   // the same network as SCL:
   #MODE_GROUP_DB.REFERENCE.GENERAL_CONDITIONS_HELP := NOT (NOT #MODE_GROUP_DB.REFERENCE.ENABLE_REQUEST AND NOT #MODE_GROUP_DB.REFERENCE.DISABLE_REQUEST) AND NOT #MODE_GROUP_DB.REFERENCE.GENERAL_CONDITIONS;
END_REGION

REGION Network 11: INITIAL CONDITIONS HELP
   RUNG wire#powerrail
      I_Contact( #MODE_GROUP_DB.REFERENCE.ENABLE_REQUEST )
      I_Contact( #MODE_GROUP_DB.REFERENCE.DISABLE_REQUEST )
      Not()
      Contact( #MODE_GROUP_DB.REFERENCE.GENERAL_CONDITIONS )
      I_Contact( #MODE_GROUP_DB.REFERENCE.INITIAL_CONDITIONS )
      Coil( #MODE_GROUP_DB.REFERENCE.INITIAL_CONDITIONS_HELP )
   END_RUNG
   // the same network as SCL:
   #MODE_GROUP_DB.REFERENCE.INITIAL_CONDITIONS_HELP := NOT (NOT #MODE_GROUP_DB.REFERENCE.ENABLE_REQUEST AND NOT #MODE_GROUP_DB.REFERENCE.DISABLE_REQUEST) AND #MODE_GROUP_DB.REFERENCE.GENERAL_CONDITIONS AND NOT #MODE_GROUP_DB.REFERENCE.INITIAL_CONDITIONS;
END_REGION
END_FUNCTION_BLOCK

FUNCTION_BLOCK "FB2007_INCREMENTAL_MODE"   // FB2007, LAD
{ S7_Optimized_Access := 'FALSE' }
VERSION : 0.1
// stored: AutoNumber false, IsIECCheckEnabled false, SetENOAutomatically false, UDAEnableTagReadback false
   VAR_INPUT
      ENABLE_REQ { ExternalAccessible := 'False'; ExternalVisible := 'False'; ExternalWritable := 'False'} : Bool;   // ENABLE REQUEST
      DISABLE_REQ { ExternalAccessible := 'False'; ExternalVisible := 'False'; ExternalWritable := 'False'} : Bool;   // DISABLE REQUEST
      NC_MANUAL_SCRN_SLCTD { ExternalAccessible := 'False'; ExternalVisible := 'False'; ExternalWritable := 'False'} : Bool;   // NC MANUAL SCREEN SELECTED
      BA3_SCRN_SLCTD { ExternalAccessible := 'False'; ExternalVisible := 'False'; ExternalWritable := 'False'} : Bool;   // BA3 SCREEN SELECTED
      OTHER_MG_INCREMENTAL_MODE_SLCTD { ExternalAccessible := 'False'; ExternalVisible := 'False'; ExternalWritable := 'False'} : Bool;   // OTHER MODE GROUP INCREMENTAL MODE SELECTED
      "1_MICRA_REQ" { ExternalAccessible := 'False'; ExternalVisible := 'False'; ExternalWritable := 'False'} : Bool;   // 1 MICRA REQUEST
      "10_MICRA_REQ" { ExternalAccessible := 'False'; ExternalVisible := 'False'; ExternalWritable := 'False'} : Bool;   // 10 MICRA REQUEST
      "100_MICRA_REQ" { ExternalAccessible := 'False'; ExternalVisible := 'False'; ExternalWritable := 'False'} : Bool;   // 100 MICRA REQUEST
      "1000_MICRA_REQ" { ExternalAccessible := 'False'; ExternalVisible := 'False'; ExternalWritable := 'False'} : Bool;   // 1000 MICRA REQUEST
   END_VAR
   VAR_OUTPUT
      INCREMENTAL_MODE_SLCTD_WRN { ExternalAccessible := 'False'; ExternalVisible := 'False'; ExternalWritable := 'False'} : Bool;   // INCREMENTAL MODE SELECTED WARNING
   END_VAR
   VAR_IN_OUT
      MODE_GROUP_DB : Struct   // MODE GROUP DB
         GENERAL : "AUTO_SINGLE_SEMI_MANUAL";
         STEP_BY_STEP : "MODES";
         MDA : "MODES";
         REFERENCE : "MODES";
         INCREMENTAL : "INCREMENTAL";
         BA : "BA_MODE";
      END_STRUCT;
   END_VAR
   VAR_TEMP
      DB_NUMBER : DInt;   // DB NUMBER FOR ALARM DECODING
   END_VAR
   // // MODE_GROUP_DB.STEP_BY_STEP.MODE_SELECTED : STEP BY STEP MODE SELECTED
   // // MODE_GROUP_DB.MDA.MODE_SELECTED : MDA MODE SELECTED
   // // MODE_GROUP_DB.REFERENCE.MODE_SELECTED : REFERENCE MODE SELECTED
   VAR_TEMP   // added for the SCL form of the ladder/FBD networks
      _w1 : Bool;
      _w2 : Bool;
   END_VAR
BEGIN

NETWORK
TITLE = READ INSTANCE DB
      L     DINO;
      +     10#800000;
      T     #DB_NUMBER;


REGION Network 2: GENERAL CONDITIONS
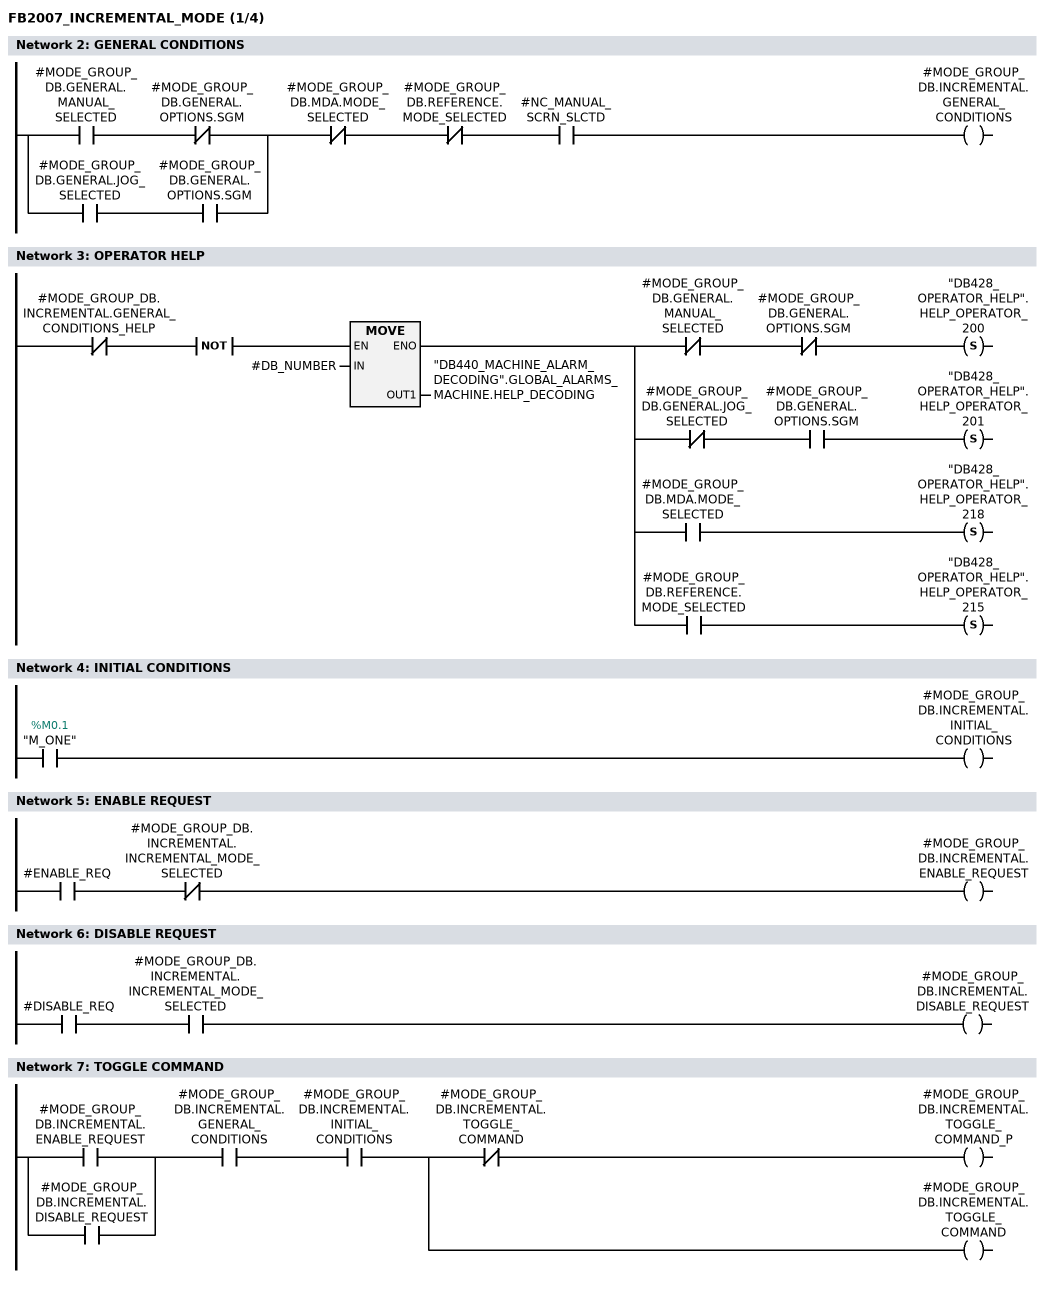
   RUNG wire#powerrail
      Contact( #MODE_GROUP_DB.GENERAL.MANUAL_SELECTED )
      I_Contact( #MODE_GROUP_DB.GENERAL.OPTIONS.SGM )
      wire#w1
      I_Contact( #MODE_GROUP_DB.MDA.MODE_SELECTED )
      I_Contact( #MODE_GROUP_DB.REFERENCE.MODE_SELECTED )
      Contact( #NC_MANUAL_SCRN_SLCTD )
      Coil( #MODE_GROUP_DB.INCREMENTAL.GENERAL_CONDITIONS )
   END_RUNG
   RUNG wire#powerrail
      Contact( #MODE_GROUP_DB.GENERAL.JOG_SELECTED )
      Contact( #MODE_GROUP_DB.GENERAL.OPTIONS.SGM )
   END_RUNG wire#w1
   // the same network as SCL:
   #MODE_GROUP_DB.INCREMENTAL.GENERAL_CONDITIONS := ((#MODE_GROUP_DB.GENERAL.MANUAL_SELECTED AND NOT #MODE_GROUP_DB.GENERAL.OPTIONS.SGM) OR (#MODE_GROUP_DB.GENERAL.JOG_SELECTED AND #MODE_GROUP_DB.GENERAL.OPTIONS.SGM)) AND NOT #MODE_GROUP_DB.MDA.MODE_SELECTED AND NOT #MODE_GROUP_DB.REFERENCE.MODE_SELECTED AND #NC_MANUAL_SCRN_SLCTD;
END_REGION

REGION Network 3: OPERATOR HELP
   RUNG wire#powerrail
      I_Contact( #MODE_GROUP_DB.INCREMENTAL.GENERAL_CONDITIONS_HELP )
      Not()
      { S7_GenerateENO := "TRUE" } Move(in := #DB_NUMBER, out1 => "DB440_MACHINE_ALARM_DECODING".GLOBAL_ALARMS_MACHINE.HELP_DECODING)
      wire#w1
      I_Contact( #MODE_GROUP_DB.GENERAL.MANUAL_SELECTED )
      I_Contact( #MODE_GROUP_DB.GENERAL.OPTIONS.SGM )
      S_Coil( "DB428_OPERATOR_HELP".HELP_OPERATOR_200 )
   END_RUNG
   RUNG wire#w1
      I_Contact( #MODE_GROUP_DB.GENERAL.JOG_SELECTED )
      Contact( #MODE_GROUP_DB.GENERAL.OPTIONS.SGM )
      S_Coil( "DB428_OPERATOR_HELP".HELP_OPERATOR_201 )
   END_RUNG
   RUNG wire#w1
      Contact( #MODE_GROUP_DB.MDA.MODE_SELECTED )
      S_Coil( "DB428_OPERATOR_HELP".HELP_OPERATOR_218 )
   END_RUNG
   RUNG wire#w1
      Contact( #MODE_GROUP_DB.REFERENCE.MODE_SELECTED )
      S_Coil( "DB428_OPERATOR_HELP".HELP_OPERATOR_215 )
   END_RUNG
   // the same network as SCL:
   // ENO of a box is taken as its EN; it also drops when the box reports an error
   #_w1 := NOT (NOT #MODE_GROUP_DB.INCREMENTAL.GENERAL_CONDITIONS_HELP);
   IF #_w1 THEN "DB440_MACHINE_ALARM_DECODING".GLOBAL_ALARMS_MACHINE.HELP_DECODING := #DB_NUMBER; END_IF;
   IF #_w1 AND NOT #MODE_GROUP_DB.GENERAL.MANUAL_SELECTED AND NOT #MODE_GROUP_DB.GENERAL.OPTIONS.SGM THEN
       "DB428_OPERATOR_HELP".HELP_OPERATOR_200 := TRUE;
   END_IF;
   IF #_w1 AND NOT #MODE_GROUP_DB.GENERAL.JOG_SELECTED AND #MODE_GROUP_DB.GENERAL.OPTIONS.SGM THEN
       "DB428_OPERATOR_HELP".HELP_OPERATOR_201 := TRUE;
   END_IF;
   IF #_w1 AND #MODE_GROUP_DB.MDA.MODE_SELECTED THEN "DB428_OPERATOR_HELP".HELP_OPERATOR_218 := TRUE; END_IF;
   IF #_w1 AND #MODE_GROUP_DB.REFERENCE.MODE_SELECTED THEN
       "DB428_OPERATOR_HELP".HELP_OPERATOR_215 := TRUE;
   END_IF;
END_REGION

REGION Network 4: INITIAL CONDITIONS
   RUNG wire#powerrail
      Contact( "M_ONE" )
      Coil( #MODE_GROUP_DB.INCREMENTAL.INITIAL_CONDITIONS )
   END_RUNG
   // the same network as SCL:
   #MODE_GROUP_DB.INCREMENTAL.INITIAL_CONDITIONS := "M_ONE";
END_REGION

REGION Network 5: ENABLE REQUEST
   RUNG wire#powerrail
      Contact( #ENABLE_REQ )
      I_Contact( #MODE_GROUP_DB.INCREMENTAL.INCREMENTAL_MODE_SELECTED )
      Coil( #MODE_GROUP_DB.INCREMENTAL.ENABLE_REQUEST )
   END_RUNG
   // the same network as SCL:
   #MODE_GROUP_DB.INCREMENTAL.ENABLE_REQUEST := #ENABLE_REQ AND NOT #MODE_GROUP_DB.INCREMENTAL.INCREMENTAL_MODE_SELECTED;
END_REGION

REGION Network 6: DISABLE REQUEST
   RUNG wire#powerrail
      Contact( #DISABLE_REQ )
      Contact( #MODE_GROUP_DB.INCREMENTAL.INCREMENTAL_MODE_SELECTED )
      Coil( #MODE_GROUP_DB.INCREMENTAL.DISABLE_REQUEST )
   END_RUNG
   // the same network as SCL:
   #MODE_GROUP_DB.INCREMENTAL.DISABLE_REQUEST := #DISABLE_REQ AND #MODE_GROUP_DB.INCREMENTAL.INCREMENTAL_MODE_SELECTED;
END_REGION

REGION Network 7: TOGGLE COMMAND
   RUNG wire#powerrail
      Contact( #MODE_GROUP_DB.INCREMENTAL.ENABLE_REQUEST )
      wire#w1
      Contact( #MODE_GROUP_DB.INCREMENTAL.GENERAL_CONDITIONS )
      Contact( #MODE_GROUP_DB.INCREMENTAL.INITIAL_CONDITIONS )
      wire#w2
      I_Contact( #MODE_GROUP_DB.INCREMENTAL.TOGGLE_COMMAND )
      Coil( #MODE_GROUP_DB.INCREMENTAL.TOGGLE_COMMAND_P )
   END_RUNG
   RUNG wire#powerrail
      Contact( #MODE_GROUP_DB.INCREMENTAL.DISABLE_REQUEST )
   END_RUNG wire#w1
   RUNG wire#w2
      Coil( #MODE_GROUP_DB.INCREMENTAL.TOGGLE_COMMAND )
   END_RUNG
   // the same network as SCL:
   #_w1 := (#MODE_GROUP_DB.INCREMENTAL.ENABLE_REQUEST OR #MODE_GROUP_DB.INCREMENTAL.DISABLE_REQUEST) AND #MODE_GROUP_DB.INCREMENTAL.GENERAL_CONDITIONS AND #MODE_GROUP_DB.INCREMENTAL.INITIAL_CONDITIONS;
   #MODE_GROUP_DB.INCREMENTAL.TOGGLE_COMMAND_P := #_w1 AND NOT #MODE_GROUP_DB.INCREMENTAL.TOGGLE_COMMAND;
   #MODE_GROUP_DB.INCREMENTAL.TOGGLE_COMMAND := #_w1;
END_REGION

REGION Network 8: INCREMENTAL MODE SELECTED
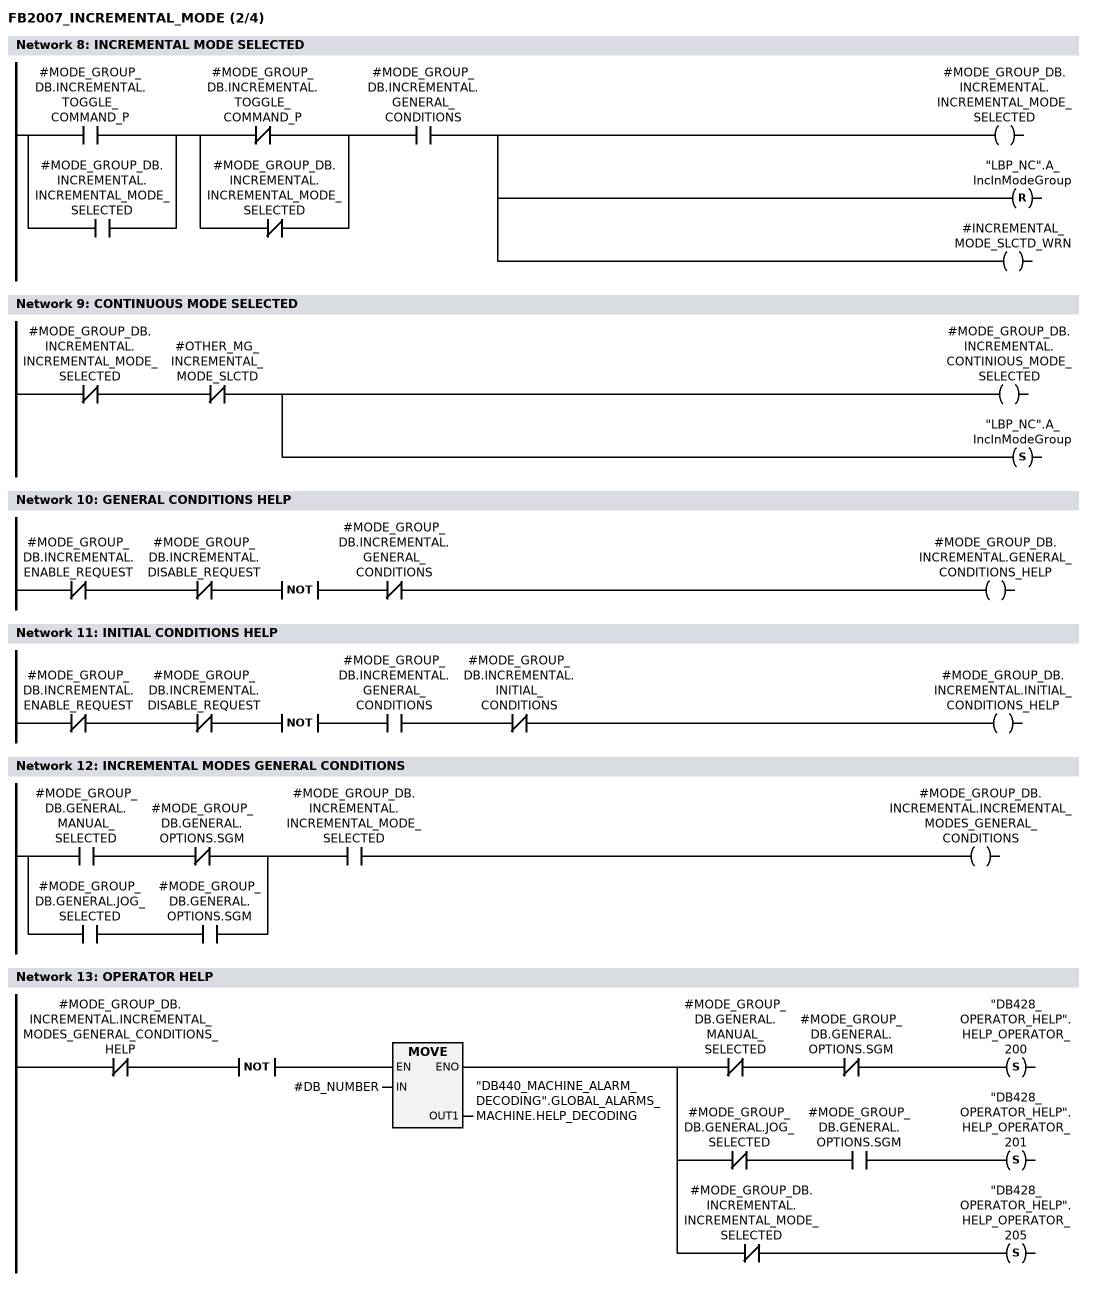
   RUNG wire#powerrail
      Contact( #MODE_GROUP_DB.INCREMENTAL.TOGGLE_COMMAND_P )
      wire#w1
      I_Contact( #MODE_GROUP_DB.INCREMENTAL.TOGGLE_COMMAND_P )
      wire#w2
      Contact( #MODE_GROUP_DB.INCREMENTAL.GENERAL_CONDITIONS )
      wire#w3
      Coil( #MODE_GROUP_DB.INCREMENTAL.INCREMENTAL_MODE_SELECTED )
   END_RUNG
   RUNG wire#powerrail
      Contact( #MODE_GROUP_DB.INCREMENTAL.INCREMENTAL_MODE_SELECTED )
   END_RUNG wire#w1
   RUNG wire#w1
      I_Contact( #MODE_GROUP_DB.INCREMENTAL.INCREMENTAL_MODE_SELECTED )
   END_RUNG wire#w2
   RUNG wire#w3
      R_Coil( "LBP_NC".A_IncInModeGroup )
   END_RUNG
   RUNG wire#w3
      Coil( #INCREMENTAL_MODE_SLCTD_WRN )
   END_RUNG
   // the same network as SCL:
   #MODE_GROUP_DB.INCREMENTAL.INCREMENTAL_MODE_SELECTED := (#MODE_GROUP_DB.INCREMENTAL.TOGGLE_COMMAND_P OR #MODE_GROUP_DB.INCREMENTAL.INCREMENTAL_MODE_SELECTED) AND (NOT #MODE_GROUP_DB.INCREMENTAL.TOGGLE_COMMAND_P OR NOT #MODE_GROUP_DB.INCREMENTAL.INCREMENTAL_MODE_SELECTED) AND #MODE_GROUP_DB.INCREMENTAL.GENERAL_CONDITIONS;
   IF #MODE_GROUP_DB.INCREMENTAL.INCREMENTAL_MODE_SELECTED THEN "LBP_NC".A_IncInModeGroup := FALSE; END_IF;
   #INCREMENTAL_MODE_SLCTD_WRN := #MODE_GROUP_DB.INCREMENTAL.INCREMENTAL_MODE_SELECTED;
END_REGION

REGION Network 9: CONTINUOUS MODE SELECTED
   RUNG wire#powerrail
      I_Contact( #MODE_GROUP_DB.INCREMENTAL.INCREMENTAL_MODE_SELECTED )
      I_Contact( #OTHER_MG_INCREMENTAL_MODE_SLCTD )
      wire#w1
      Coil( #MODE_GROUP_DB.INCREMENTAL.CONTINIOUS_MODE_SELECTED )
   END_RUNG
   RUNG wire#w1
      S_Coil( "LBP_NC".A_IncInModeGroup )
   END_RUNG
   // the same network as SCL:
   #MODE_GROUP_DB.INCREMENTAL.CONTINIOUS_MODE_SELECTED := NOT #MODE_GROUP_DB.INCREMENTAL.INCREMENTAL_MODE_SELECTED AND NOT #OTHER_MG_INCREMENTAL_MODE_SLCTD;
   IF #MODE_GROUP_DB.INCREMENTAL.CONTINIOUS_MODE_SELECTED THEN "LBP_NC".A_IncInModeGroup := TRUE; END_IF;
END_REGION

REGION Network 10: GENERAL CONDITIONS HELP
   RUNG wire#powerrail
      I_Contact( #MODE_GROUP_DB.INCREMENTAL.ENABLE_REQUEST )
      I_Contact( #MODE_GROUP_DB.INCREMENTAL.DISABLE_REQUEST )
      Not()
      I_Contact( #MODE_GROUP_DB.INCREMENTAL.GENERAL_CONDITIONS )
      Coil( #MODE_GROUP_DB.INCREMENTAL.GENERAL_CONDITIONS_HELP )
   END_RUNG
   // the same network as SCL:
   #MODE_GROUP_DB.INCREMENTAL.GENERAL_CONDITIONS_HELP := NOT (NOT #MODE_GROUP_DB.INCREMENTAL.ENABLE_REQUEST AND NOT #MODE_GROUP_DB.INCREMENTAL.DISABLE_REQUEST) AND NOT #MODE_GROUP_DB.INCREMENTAL.GENERAL_CONDITIONS;
END_REGION

REGION Network 11: INITIAL CONDITIONS HELP
   RUNG wire#powerrail
      I_Contact( #MODE_GROUP_DB.INCREMENTAL.ENABLE_REQUEST )
      I_Contact( #MODE_GROUP_DB.INCREMENTAL.DISABLE_REQUEST )
      Not()
      Contact( #MODE_GROUP_DB.INCREMENTAL.GENERAL_CONDITIONS )
      I_Contact( #MODE_GROUP_DB.INCREMENTAL.INITIAL_CONDITIONS )
      Coil( #MODE_GROUP_DB.INCREMENTAL.INITIAL_CONDITIONS_HELP )
   END_RUNG
   // the same network as SCL:
   #MODE_GROUP_DB.INCREMENTAL.INITIAL_CONDITIONS_HELP := NOT (NOT #MODE_GROUP_DB.INCREMENTAL.ENABLE_REQUEST AND NOT #MODE_GROUP_DB.INCREMENTAL.DISABLE_REQUEST) AND #MODE_GROUP_DB.INCREMENTAL.GENERAL_CONDITIONS AND NOT #MODE_GROUP_DB.INCREMENTAL.INITIAL_CONDITIONS;
END_REGION

REGION Network 12: INCREMENTAL MODES GENERAL CONDITIONS
   RUNG wire#powerrail
      Contact( #MODE_GROUP_DB.GENERAL.MANUAL_SELECTED )
      I_Contact( #MODE_GROUP_DB.GENERAL.OPTIONS.SGM )
      wire#w1
      Contact( #MODE_GROUP_DB.INCREMENTAL.INCREMENTAL_MODE_SELECTED )
      Coil( #MODE_GROUP_DB.INCREMENTAL.INCREMENTAL_MODES_GENERAL_CONDITIONS )
   END_RUNG
   RUNG wire#powerrail
      Contact( #MODE_GROUP_DB.GENERAL.JOG_SELECTED )
      Contact( #MODE_GROUP_DB.GENERAL.OPTIONS.SGM )
   END_RUNG wire#w1
   // the same network as SCL:
   #MODE_GROUP_DB.INCREMENTAL.INCREMENTAL_MODES_GENERAL_CONDITIONS := ((#MODE_GROUP_DB.GENERAL.MANUAL_SELECTED AND NOT #MODE_GROUP_DB.GENERAL.OPTIONS.SGM) OR (#MODE_GROUP_DB.GENERAL.JOG_SELECTED AND #MODE_GROUP_DB.GENERAL.OPTIONS.SGM)) AND #MODE_GROUP_DB.INCREMENTAL.INCREMENTAL_MODE_SELECTED;
END_REGION

REGION Network 13: OPERATOR HELP
   RUNG wire#powerrail
      I_Contact( #MODE_GROUP_DB.INCREMENTAL.INCREMENTAL_MODES_GENERAL_CONDITIONS_HELP )
      Not()
      { S7_GenerateENO := "TRUE" } Move(in := #DB_NUMBER, out1 => "DB440_MACHINE_ALARM_DECODING".GLOBAL_ALARMS_MACHINE.HELP_DECODING)
      wire#w1
      I_Contact( #MODE_GROUP_DB.GENERAL.MANUAL_SELECTED )
      I_Contact( #MODE_GROUP_DB.GENERAL.OPTIONS.SGM )
      S_Coil( "DB428_OPERATOR_HELP".HELP_OPERATOR_200 )
   END_RUNG
   RUNG wire#w1
      I_Contact( #MODE_GROUP_DB.GENERAL.JOG_SELECTED )
      Contact( #MODE_GROUP_DB.GENERAL.OPTIONS.SGM )
      S_Coil( "DB428_OPERATOR_HELP".HELP_OPERATOR_201 )
   END_RUNG
   RUNG wire#w1
      I_Contact( #MODE_GROUP_DB.INCREMENTAL.INCREMENTAL_MODE_SELECTED )
      S_Coil( "DB428_OPERATOR_HELP".HELP_OPERATOR_205 )
   END_RUNG
   // the same network as SCL:
   // ENO of a box is taken as its EN; it also drops when the box reports an error
   #_w1 := NOT (NOT #MODE_GROUP_DB.INCREMENTAL.INCREMENTAL_MODES_GENERAL_CONDITIONS_HELP);
   IF #_w1 THEN "DB440_MACHINE_ALARM_DECODING".GLOBAL_ALARMS_MACHINE.HELP_DECODING := #DB_NUMBER; END_IF;
   IF #_w1 AND NOT #MODE_GROUP_DB.GENERAL.MANUAL_SELECTED AND NOT #MODE_GROUP_DB.GENERAL.OPTIONS.SGM THEN
       "DB428_OPERATOR_HELP".HELP_OPERATOR_200 := TRUE;
   END_IF;
   IF #_w1 AND NOT #MODE_GROUP_DB.GENERAL.JOG_SELECTED AND #MODE_GROUP_DB.GENERAL.OPTIONS.SGM THEN
       "DB428_OPERATOR_HELP".HELP_OPERATOR_201 := TRUE;
   END_IF;
   IF #_w1 AND NOT #MODE_GROUP_DB.INCREMENTAL.INCREMENTAL_MODE_SELECTED THEN
       "DB428_OPERATOR_HELP".HELP_OPERATOR_205 := TRUE;
   END_IF;
END_REGION

REGION Network 14: INCREMENTAL MODES INITIAL CONDITIONS
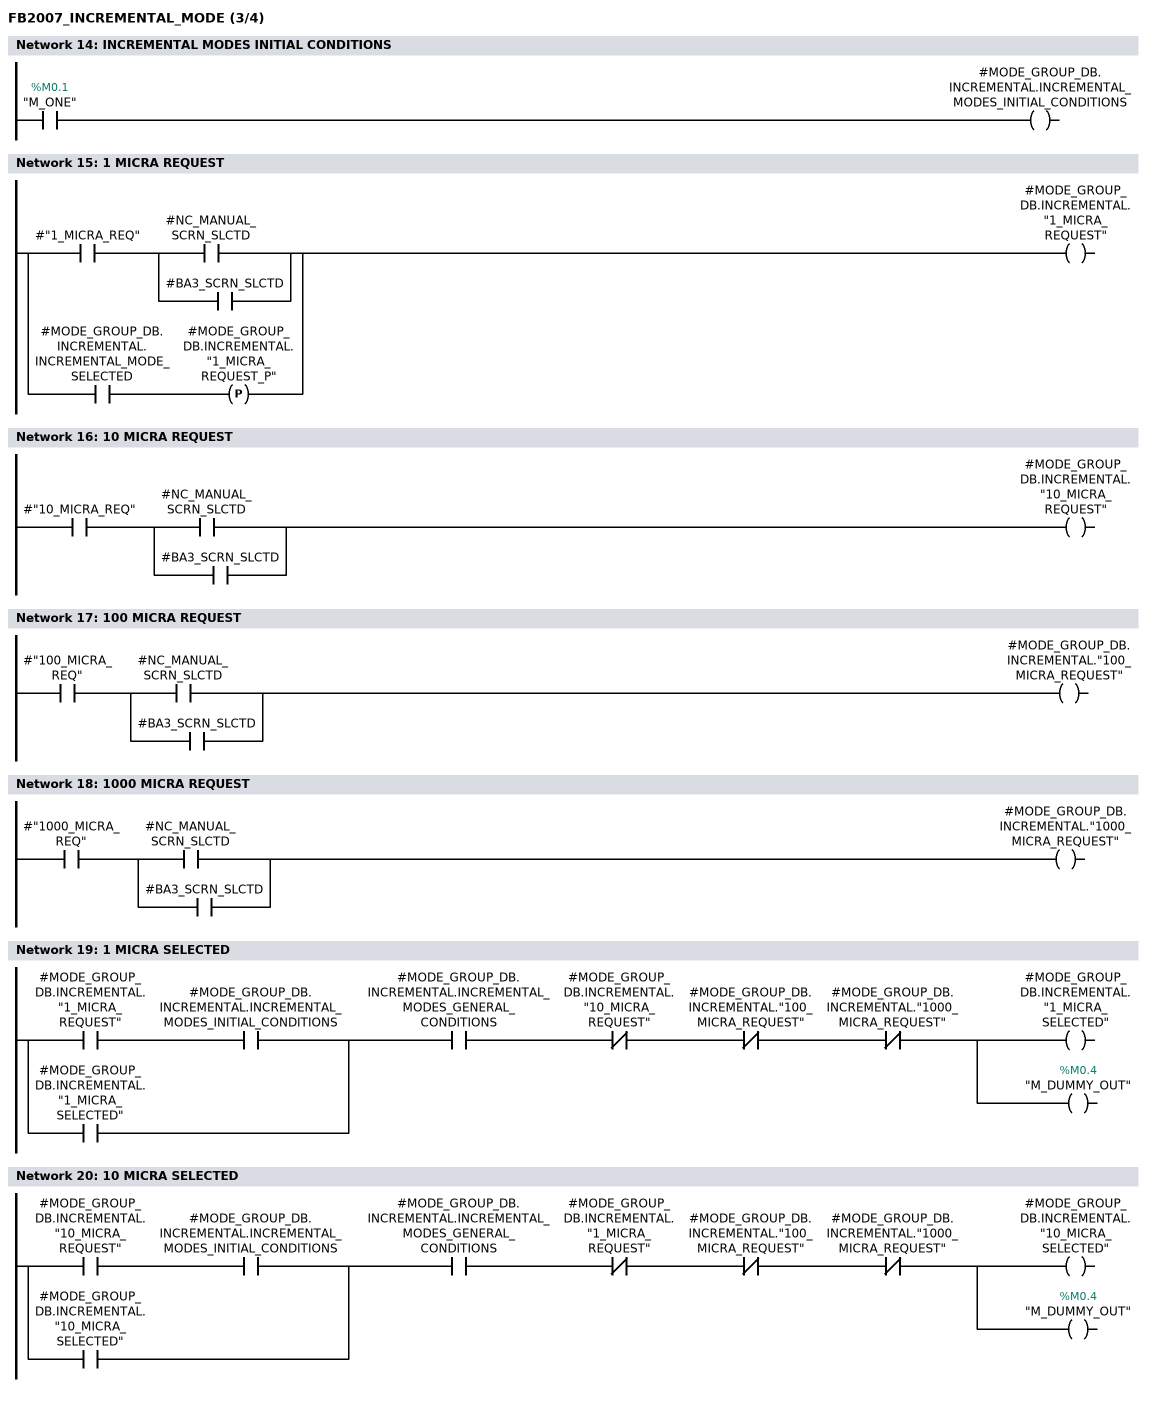
   RUNG wire#powerrail
      Contact( "M_ONE" )
      Coil( #MODE_GROUP_DB.INCREMENTAL.INCREMENTAL_MODES_INITIAL_CONDITIONS )
   END_RUNG
   // the same network as SCL:
   #MODE_GROUP_DB.INCREMENTAL.INCREMENTAL_MODES_INITIAL_CONDITIONS := "M_ONE";
END_REGION

REGION Network 15: 1 MICRA REQUEST
   RUNG wire#powerrail
      Contact( #"1_MICRA_REQ" )
      wire#w1
      Contact( #NC_MANUAL_SCRN_SLCTD )
      wire#w2
      Coil( #MODE_GROUP_DB.INCREMENTAL."1_MICRA_REQUEST" )
   END_RUNG
   RUNG wire#w1
      Contact( #BA3_SCRN_SLCTD )
   END_RUNG wire#w2
   RUNG wire#powerrail
      Contact( #MODE_GROUP_DB.INCREMENTAL.INCREMENTAL_MODE_SELECTED )
      P_Trig( #MODE_GROUP_DB.INCREMENTAL."1_MICRA_REQUEST_P" )
   END_RUNG wire#w2
   // the same network as SCL:
   #_w1 := #MODE_GROUP_DB.INCREMENTAL.INCREMENTAL_MODE_SELECTED AND NOT #MODE_GROUP_DB.INCREMENTAL."1_MICRA_REQUEST_P";   // rising edge
   #MODE_GROUP_DB.INCREMENTAL."1_MICRA_REQUEST_P" := #MODE_GROUP_DB.INCREMENTAL.INCREMENTAL_MODE_SELECTED;
   #MODE_GROUP_DB.INCREMENTAL."1_MICRA_REQUEST" := (#"1_MICRA_REQ" AND (#NC_MANUAL_SCRN_SLCTD OR #BA3_SCRN_SLCTD)) OR #_w1;
END_REGION

REGION Network 16: 10 MICRA REQUEST
   RUNG wire#powerrail
      Contact( #"10_MICRA_REQ" )
      wire#w1
      Contact( #NC_MANUAL_SCRN_SLCTD )
      wire#w2
      Coil( #MODE_GROUP_DB.INCREMENTAL."10_MICRA_REQUEST" )
   END_RUNG
   RUNG wire#w1
      Contact( #BA3_SCRN_SLCTD )
   END_RUNG wire#w2
   // the same network as SCL:
   #MODE_GROUP_DB.INCREMENTAL."10_MICRA_REQUEST" := #"10_MICRA_REQ" AND (#NC_MANUAL_SCRN_SLCTD OR #BA3_SCRN_SLCTD);
END_REGION

REGION Network 17: 100 MICRA REQUEST
   RUNG wire#powerrail
      Contact( #"100_MICRA_REQ" )
      wire#w1
      Contact( #NC_MANUAL_SCRN_SLCTD )
      wire#w2
      Coil( #MODE_GROUP_DB.INCREMENTAL."100_MICRA_REQUEST" )
   END_RUNG
   RUNG wire#w1
      Contact( #BA3_SCRN_SLCTD )
   END_RUNG wire#w2
   // the same network as SCL:
   #MODE_GROUP_DB.INCREMENTAL."100_MICRA_REQUEST" := #"100_MICRA_REQ" AND (#NC_MANUAL_SCRN_SLCTD OR #BA3_SCRN_SLCTD);
END_REGION

REGION Network 18: 1000 MICRA REQUEST
   RUNG wire#powerrail
      Contact( #"1000_MICRA_REQ" )
      wire#w1
      Contact( #NC_MANUAL_SCRN_SLCTD )
      wire#w2
      Coil( #MODE_GROUP_DB.INCREMENTAL."1000_MICRA_REQUEST" )
   END_RUNG
   RUNG wire#w1
      Contact( #BA3_SCRN_SLCTD )
   END_RUNG wire#w2
   // the same network as SCL:
   #MODE_GROUP_DB.INCREMENTAL."1000_MICRA_REQUEST" := #"1000_MICRA_REQ" AND (#NC_MANUAL_SCRN_SLCTD OR #BA3_SCRN_SLCTD);
END_REGION

REGION Network 19: 1 MICRA SELECTED
   RUNG wire#powerrail
      Contact( #MODE_GROUP_DB.INCREMENTAL."1_MICRA_REQUEST" )
      Contact( #MODE_GROUP_DB.INCREMENTAL.INCREMENTAL_MODES_INITIAL_CONDITIONS )
      wire#w1
      Contact( #MODE_GROUP_DB.INCREMENTAL.INCREMENTAL_MODES_GENERAL_CONDITIONS )
      I_Contact( #MODE_GROUP_DB.INCREMENTAL."10_MICRA_REQUEST" )
      I_Contact( #MODE_GROUP_DB.INCREMENTAL."100_MICRA_REQUEST" )
      I_Contact( #MODE_GROUP_DB.INCREMENTAL."1000_MICRA_REQUEST" )
      wire#w2
      Coil( #MODE_GROUP_DB.INCREMENTAL."1_MICRA_SELECTED" )
   END_RUNG
   RUNG wire#powerrail
      Contact( #MODE_GROUP_DB.INCREMENTAL."1_MICRA_SELECTED" )
   END_RUNG wire#w1
   RUNG wire#w2
      Coil( "M_DUMMY_OUT" )
   END_RUNG
   // the same network as SCL:
   #MODE_GROUP_DB.INCREMENTAL."1_MICRA_SELECTED" := ((#MODE_GROUP_DB.INCREMENTAL."1_MICRA_REQUEST" AND #MODE_GROUP_DB.INCREMENTAL.INCREMENTAL_MODES_INITIAL_CONDITIONS) OR #MODE_GROUP_DB.INCREMENTAL."1_MICRA_SELECTED") AND #MODE_GROUP_DB.INCREMENTAL.INCREMENTAL_MODES_GENERAL_CONDITIONS AND NOT #MODE_GROUP_DB.INCREMENTAL."10_MICRA_REQUEST" AND NOT #MODE_GROUP_DB.INCREMENTAL."100_MICRA_REQUEST" AND NOT #MODE_GROUP_DB.INCREMENTAL."1000_MICRA_REQUEST";
   "M_DUMMY_OUT" := #MODE_GROUP_DB.INCREMENTAL."1_MICRA_SELECTED";
END_REGION

REGION Network 20: 10 MICRA SELECTED
   RUNG wire#powerrail
      Contact( #MODE_GROUP_DB.INCREMENTAL."10_MICRA_REQUEST" )
      Contact( #MODE_GROUP_DB.INCREMENTAL.INCREMENTAL_MODES_INITIAL_CONDITIONS )
      wire#w1
      Contact( #MODE_GROUP_DB.INCREMENTAL.INCREMENTAL_MODES_GENERAL_CONDITIONS )
      I_Contact( #MODE_GROUP_DB.INCREMENTAL."1_MICRA_REQUEST" )
      I_Contact( #MODE_GROUP_DB.INCREMENTAL."100_MICRA_REQUEST" )
      I_Contact( #MODE_GROUP_DB.INCREMENTAL."1000_MICRA_REQUEST" )
      wire#w2
      Coil( #MODE_GROUP_DB.INCREMENTAL."10_MICRA_SELECTED" )
   END_RUNG
   RUNG wire#powerrail
      Contact( #MODE_GROUP_DB.INCREMENTAL."10_MICRA_SELECTED" )
   END_RUNG wire#w1
   RUNG wire#w2
      Coil( "M_DUMMY_OUT" )
   END_RUNG
   // the same network as SCL:
   #MODE_GROUP_DB.INCREMENTAL."10_MICRA_SELECTED" := ((#MODE_GROUP_DB.INCREMENTAL."10_MICRA_REQUEST" AND #MODE_GROUP_DB.INCREMENTAL.INCREMENTAL_MODES_INITIAL_CONDITIONS) OR #MODE_GROUP_DB.INCREMENTAL."10_MICRA_SELECTED") AND #MODE_GROUP_DB.INCREMENTAL.INCREMENTAL_MODES_GENERAL_CONDITIONS AND NOT #MODE_GROUP_DB.INCREMENTAL."1_MICRA_REQUEST" AND NOT #MODE_GROUP_DB.INCREMENTAL."100_MICRA_REQUEST" AND NOT #MODE_GROUP_DB.INCREMENTAL."1000_MICRA_REQUEST";
   "M_DUMMY_OUT" := #MODE_GROUP_DB.INCREMENTAL."10_MICRA_SELECTED";
END_REGION

REGION Network 21: 100 MICRA SELECTED
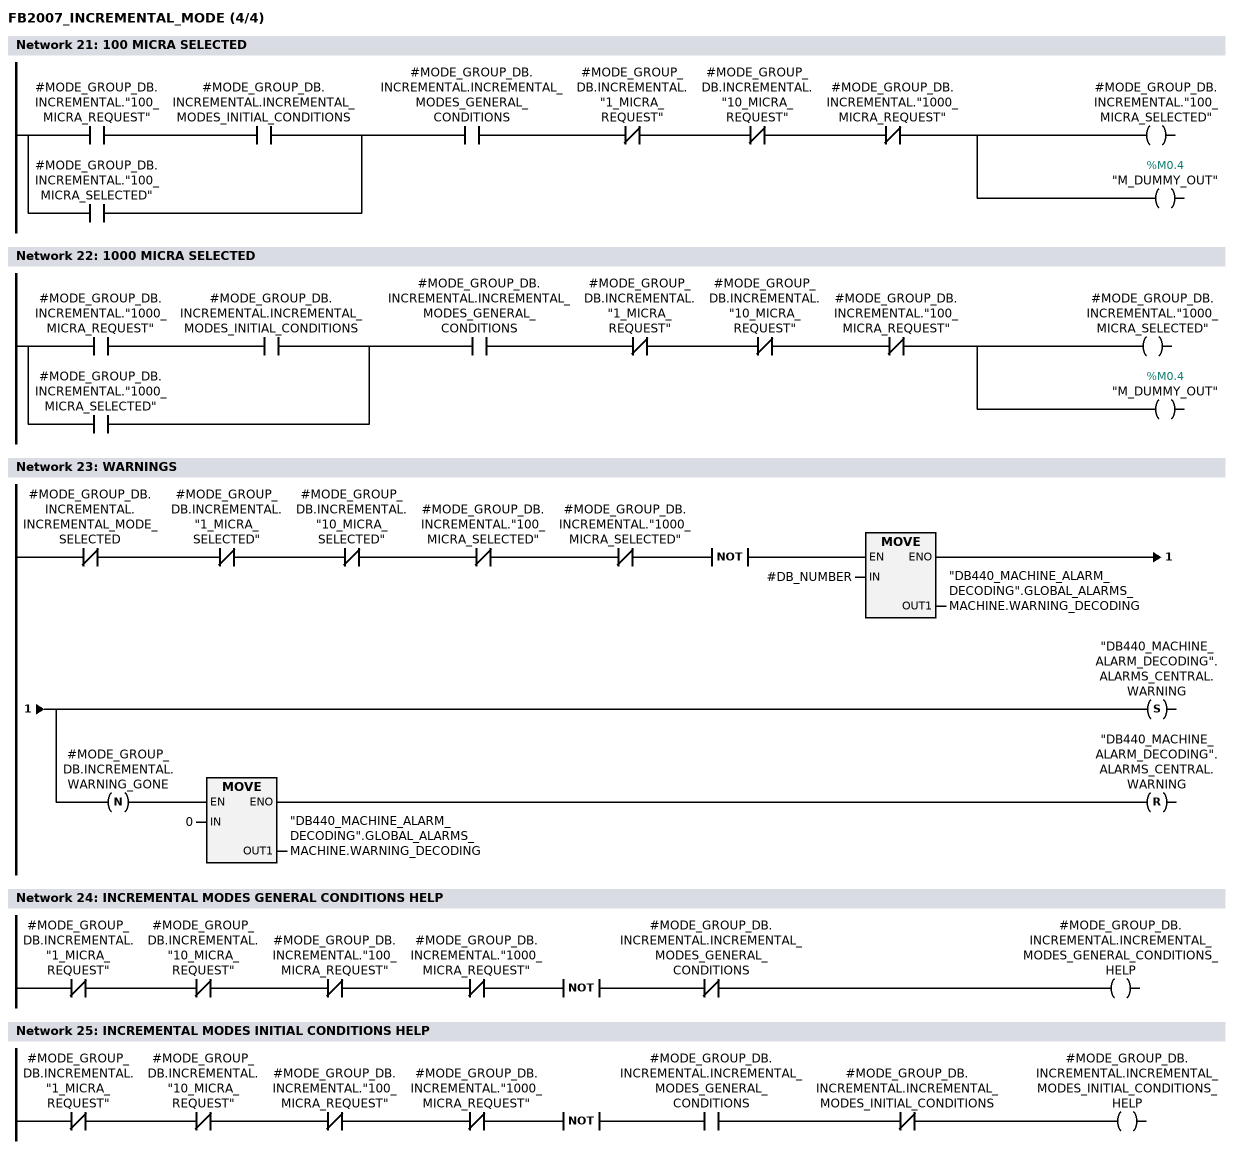
   RUNG wire#powerrail
      Contact( #MODE_GROUP_DB.INCREMENTAL."100_MICRA_REQUEST" )
      Contact( #MODE_GROUP_DB.INCREMENTAL.INCREMENTAL_MODES_INITIAL_CONDITIONS )
      wire#w1
      Contact( #MODE_GROUP_DB.INCREMENTAL.INCREMENTAL_MODES_GENERAL_CONDITIONS )
      I_Contact( #MODE_GROUP_DB.INCREMENTAL."1_MICRA_REQUEST" )
      I_Contact( #MODE_GROUP_DB.INCREMENTAL."10_MICRA_REQUEST" )
      I_Contact( #MODE_GROUP_DB.INCREMENTAL."1000_MICRA_REQUEST" )
      wire#w2
      Coil( #MODE_GROUP_DB.INCREMENTAL."100_MICRA_SELECTED" )
   END_RUNG
   RUNG wire#powerrail
      Contact( #MODE_GROUP_DB.INCREMENTAL."100_MICRA_SELECTED" )
   END_RUNG wire#w1
   RUNG wire#w2
      Coil( "M_DUMMY_OUT" )
   END_RUNG
   // the same network as SCL:
   #MODE_GROUP_DB.INCREMENTAL."100_MICRA_SELECTED" := ((#MODE_GROUP_DB.INCREMENTAL."100_MICRA_REQUEST" AND #MODE_GROUP_DB.INCREMENTAL.INCREMENTAL_MODES_INITIAL_CONDITIONS) OR #MODE_GROUP_DB.INCREMENTAL."100_MICRA_SELECTED") AND #MODE_GROUP_DB.INCREMENTAL.INCREMENTAL_MODES_GENERAL_CONDITIONS AND NOT #MODE_GROUP_DB.INCREMENTAL."1_MICRA_REQUEST" AND NOT #MODE_GROUP_DB.INCREMENTAL."10_MICRA_REQUEST" AND NOT #MODE_GROUP_DB.INCREMENTAL."1000_MICRA_REQUEST";
   "M_DUMMY_OUT" := #MODE_GROUP_DB.INCREMENTAL."100_MICRA_SELECTED";
END_REGION

REGION Network 22: 1000 MICRA SELECTED
   RUNG wire#powerrail
      Contact( #MODE_GROUP_DB.INCREMENTAL."1000_MICRA_REQUEST" )
      Contact( #MODE_GROUP_DB.INCREMENTAL.INCREMENTAL_MODES_INITIAL_CONDITIONS )
      wire#w1
      Contact( #MODE_GROUP_DB.INCREMENTAL.INCREMENTAL_MODES_GENERAL_CONDITIONS )
      I_Contact( #MODE_GROUP_DB.INCREMENTAL."1_MICRA_REQUEST" )
      I_Contact( #MODE_GROUP_DB.INCREMENTAL."10_MICRA_REQUEST" )
      I_Contact( #MODE_GROUP_DB.INCREMENTAL."100_MICRA_REQUEST" )
      wire#w2
      Coil( #MODE_GROUP_DB.INCREMENTAL."1000_MICRA_SELECTED" )
   END_RUNG
   RUNG wire#powerrail
      Contact( #MODE_GROUP_DB.INCREMENTAL."1000_MICRA_SELECTED" )
   END_RUNG wire#w1
   RUNG wire#w2
      Coil( "M_DUMMY_OUT" )
   END_RUNG
   // the same network as SCL:
   #MODE_GROUP_DB.INCREMENTAL."1000_MICRA_SELECTED" := ((#MODE_GROUP_DB.INCREMENTAL."1000_MICRA_REQUEST" AND #MODE_GROUP_DB.INCREMENTAL.INCREMENTAL_MODES_INITIAL_CONDITIONS) OR #MODE_GROUP_DB.INCREMENTAL."1000_MICRA_SELECTED") AND #MODE_GROUP_DB.INCREMENTAL.INCREMENTAL_MODES_GENERAL_CONDITIONS AND NOT #MODE_GROUP_DB.INCREMENTAL."1_MICRA_REQUEST" AND NOT #MODE_GROUP_DB.INCREMENTAL."10_MICRA_REQUEST" AND NOT #MODE_GROUP_DB.INCREMENTAL."100_MICRA_REQUEST";
   "M_DUMMY_OUT" := #MODE_GROUP_DB.INCREMENTAL."1000_MICRA_SELECTED";
END_REGION

REGION Network 23: WARNINGS
   RUNG wire#powerrail
      I_Contact( #MODE_GROUP_DB.INCREMENTAL.INCREMENTAL_MODE_SELECTED )
      I_Contact( #MODE_GROUP_DB.INCREMENTAL."1_MICRA_SELECTED" )
      I_Contact( #MODE_GROUP_DB.INCREMENTAL."10_MICRA_SELECTED" )
      I_Contact( #MODE_GROUP_DB.INCREMENTAL."100_MICRA_SELECTED" )
      I_Contact( #MODE_GROUP_DB.INCREMENTAL."1000_MICRA_SELECTED" )
      Not()
      Move(in := #DB_NUMBER, out1 => "DB440_MACHINE_ALARM_DECODING".GLOBAL_ALARMS_MACHINE.WARNING_DECODING)
      wire#w1
      S_Coil( "DB440_MACHINE_ALARM_DECODING".ALARMS_CENTRAL.WARNING )
   END_RUNG
   RUNG wire#w1
      N_Trig( #MODE_GROUP_DB.INCREMENTAL.WARNING_GONE )
      Move(in := 0, out1 => "DB440_MACHINE_ALARM_DECODING".GLOBAL_ALARMS_MACHINE.WARNING_DECODING)
      R_Coil( "DB440_MACHINE_ALARM_DECODING".ALARMS_CENTRAL.WARNING )
   END_RUNG
   // the same network as SCL:
   #_w1 := NOT (NOT #MODE_GROUP_DB.INCREMENTAL.INCREMENTAL_MODE_SELECTED AND NOT #MODE_GROUP_DB.INCREMENTAL."1_MICRA_SELECTED" AND NOT #MODE_GROUP_DB.INCREMENTAL."10_MICRA_SELECTED" AND NOT #MODE_GROUP_DB.INCREMENTAL."100_MICRA_SELECTED" AND NOT #MODE_GROUP_DB.INCREMENTAL."1000_MICRA_SELECTED");
   IF #_w1 THEN
       "DB440_MACHINE_ALARM_DECODING".GLOBAL_ALARMS_MACHINE.WARNING_DECODING := #DB_NUMBER;
       "DB440_MACHINE_ALARM_DECODING".ALARMS_CENTRAL.WARNING := TRUE;
   END_IF;
   #_w2 := NOT #_w1 AND #MODE_GROUP_DB.INCREMENTAL.WARNING_GONE;   // falling edge
   #MODE_GROUP_DB.INCREMENTAL.WARNING_GONE := #_w1;
   IF #_w2 THEN
       "DB440_MACHINE_ALARM_DECODING".GLOBAL_ALARMS_MACHINE.WARNING_DECODING := 0;
       "DB440_MACHINE_ALARM_DECODING".ALARMS_CENTRAL.WARNING := FALSE;
   END_IF;
END_REGION

REGION Network 24: INCREMENTAL MODES GENERAL CONDITIONS HELP
   RUNG wire#powerrail
      I_Contact( #MODE_GROUP_DB.INCREMENTAL."1_MICRA_REQUEST" )
      I_Contact( #MODE_GROUP_DB.INCREMENTAL."10_MICRA_REQUEST" )
      I_Contact( #MODE_GROUP_DB.INCREMENTAL."100_MICRA_REQUEST" )
      I_Contact( #MODE_GROUP_DB.INCREMENTAL."1000_MICRA_REQUEST" )
      Not()
      I_Contact( #MODE_GROUP_DB.INCREMENTAL.INCREMENTAL_MODES_GENERAL_CONDITIONS )
      Coil( #MODE_GROUP_DB.INCREMENTAL.INCREMENTAL_MODES_GENERAL_CONDITIONS_HELP )
   END_RUNG
   // the same network as SCL:
   #MODE_GROUP_DB.INCREMENTAL.INCREMENTAL_MODES_GENERAL_CONDITIONS_HELP := NOT (NOT #MODE_GROUP_DB.INCREMENTAL."1_MICRA_REQUEST" AND NOT #MODE_GROUP_DB.INCREMENTAL."10_MICRA_REQUEST" AND NOT #MODE_GROUP_DB.INCREMENTAL."100_MICRA_REQUEST" AND NOT #MODE_GROUP_DB.INCREMENTAL."1000_MICRA_REQUEST") AND NOT #MODE_GROUP_DB.INCREMENTAL.INCREMENTAL_MODES_GENERAL_CONDITIONS;
END_REGION

REGION Network 25: INCREMENTAL MODES INITIAL CONDITIONS HELP
   RUNG wire#powerrail
      I_Contact( #MODE_GROUP_DB.INCREMENTAL."1_MICRA_REQUEST" )
      I_Contact( #MODE_GROUP_DB.INCREMENTAL."10_MICRA_REQUEST" )
      I_Contact( #MODE_GROUP_DB.INCREMENTAL."100_MICRA_REQUEST" )
      I_Contact( #MODE_GROUP_DB.INCREMENTAL."1000_MICRA_REQUEST" )
      Not()
      Contact( #MODE_GROUP_DB.INCREMENTAL.INCREMENTAL_MODES_GENERAL_CONDITIONS )
      I_Contact( #MODE_GROUP_DB.INCREMENTAL.INCREMENTAL_MODES_INITIAL_CONDITIONS )
      Coil( #MODE_GROUP_DB.INCREMENTAL.INCREMENTAL_MODES_INITIAL_CONDITIONS_HELP )
   END_RUNG
   // the same network as SCL:
   #MODE_GROUP_DB.INCREMENTAL.INCREMENTAL_MODES_INITIAL_CONDITIONS_HELP := NOT (NOT #MODE_GROUP_DB.INCREMENTAL."1_MICRA_REQUEST" AND NOT #MODE_GROUP_DB.INCREMENTAL."10_MICRA_REQUEST" AND NOT #MODE_GROUP_DB.INCREMENTAL."100_MICRA_REQUEST" AND NOT #MODE_GROUP_DB.INCREMENTAL."1000_MICRA_REQUEST") AND #MODE_GROUP_DB.INCREMENTAL.INCREMENTAL_MODES_GENERAL_CONDITIONS AND NOT #MODE_GROUP_DB.INCREMENTAL.INCREMENTAL_MODES_INITIAL_CONDITIONS;
END_REGION
END_FUNCTION_BLOCK

FUNCTION_BLOCK "FB2107_LIGHTS"   // FB2107, LAD
{ S7_Optimized_Access := 'TRUE' }
VERSION : 0.1
// stored: AutoNumber false, IsIECCheckEnabled false, IsRetainMemResEnabled false, MemoryReserve 100, SetENOAutomatically false, UDAEnableTagReadback false
   VAR_INPUT
      GENERAL_MACHINE_LIGHT_OPTION : Bool;
      CIRCUIT_BRAKER_IN : Bool;
      LIGHT_ON_SELECTOR : Bool;
      MANUAL_REQ_LINE : Bool;   // MANUAL REQUEST HMI LINE NUMBER
      SWITCH_ON_AUTO_REQ : Bool;   // SWITCH ON AUTO REQUEST
      SWITCH_OFF_AUTO_REQ : Bool;   // SWITCH OFF AUTO REQUEST
   END_VAR
   VAR_OUTPUT
      LIGHTS_ON : Bool;   // LIGHTS ON OUTPUT
      HMI_LINE_ON_EXEC : Bool;   // HMI LINE ON EXECUTABILITY
      HMI_LINE_OFF_EXEC : Bool;   // HMI LINE OFF EXECUTABILITY
      HMI_LINE_ON_STATUS : Bool;   // HMI LINE ON STATUS
      HMI_LINE_OFF_STATUS : Bool;   // HMI LINE OFF STATUS
   END_VAR
   VAR
      SWITCH_ON_GENERAL_CONDITIONS : Bool;   // SWITCH ON GENERAL CONDITIONS
      SWITCH_ON_INITIAL_CONDITIONS : Bool;   // SWITCH ON INITIAL CONDITIONS
      SWITCH_ON_MANUAL_REQ : Bool;   // SWITCH ON MANUAL REQUEST
      SWITCH_ON_GLOBAL_REQ : Bool;   // SWITCH ON GLOBAL REQUEST
      SWITCH_ON_COMMAND : Bool;   // SWITCH ON COMMAND
      SWITCH_ON : Bool;   // SWITCH ON
      IN_SERVICE : Bool;   // IN SERVICE
      SWITCH_OFF_GENERAL_CONDITIONS : Bool;   // SWITCH OFF GENERAL CONDITIONS
      SWITCH_OFF_INITIAL_CONDITIONS : Bool;   // SWITCH OFF INITIAL CONDITIONS
      SWITCH_OFF_MANUAL_REQ : Bool;   // SWITCH OFF MANUAL REQUEST
      SWITCH_OFF_GLOBAL_REQ : Bool;   // SWITCH OFF GLOBAL REQUEST
      SWITCH_OFF_COMMAND : Bool;   // SWITCH OFF COMMAND
      SWITCH_OFF : Bool;   // SWITCH OFF
      OUT_OF_SERVICE : Bool;   // OUT OF SERVICE
      SWITCH_ON_GLOBAL_REQUEST_AUX0 : Bool;   // SWITCH ON GLOBAL REQUEST AUXILIARY 0
      SWITCH_ON_GLOBAL_REQUEST_AUX1 : Bool;   // SWITCH ON GLOBAL REQUEST AUXILIARY 1
      SWITCH_ON_GLOBAL_REQUEST_AUX2 : Bool;   // SWITCH ON GLOBAL REQUEST AUXILIARY 2
      SWITCH_ON_GLOBAL_REQUEST_AUX3 : Bool;   // SWITCH ON GLOBAL REQUEST AUXILIARY 3
      SWITCH_OFF_GLOBAL_REQUEST_AUX1 : Bool;   // SWITCH OFF GLOBAL REQUEST AUXILIARY 1
      SWITCH_OFF_GLOBAL_REQUEST_AUX2 : Bool;   // SWITCH OFF GLOBAL REQUEST AUXILIARY 2
      SWITCH_OFF_DOORS_CLOSED_TIMER : IEC_TIMER;
      SWITCH_OFF_IN_SERVICE_DELAY_TIMER : IEC_TIMER;
   END_VAR
   // SWITCH_OFF_DOORS_CLOSED_TIMER.PT := T#10M;
   // SWITCH_OFF_IN_SERVICE_DELAY_TIMER.PT := T#1H;
   VAR_TEMP   // added for the SCL form of the ladder/FBD networks
      _w1 : Bool;
      _w2 : Bool;
      _w3 : Bool;
      _w4 : Bool;
      _w5 : Bool;
      _w6 : Bool;
   END_VAR
BEGIN

REGION Network 1: SWITCH ON GENERAL CONDITIONS
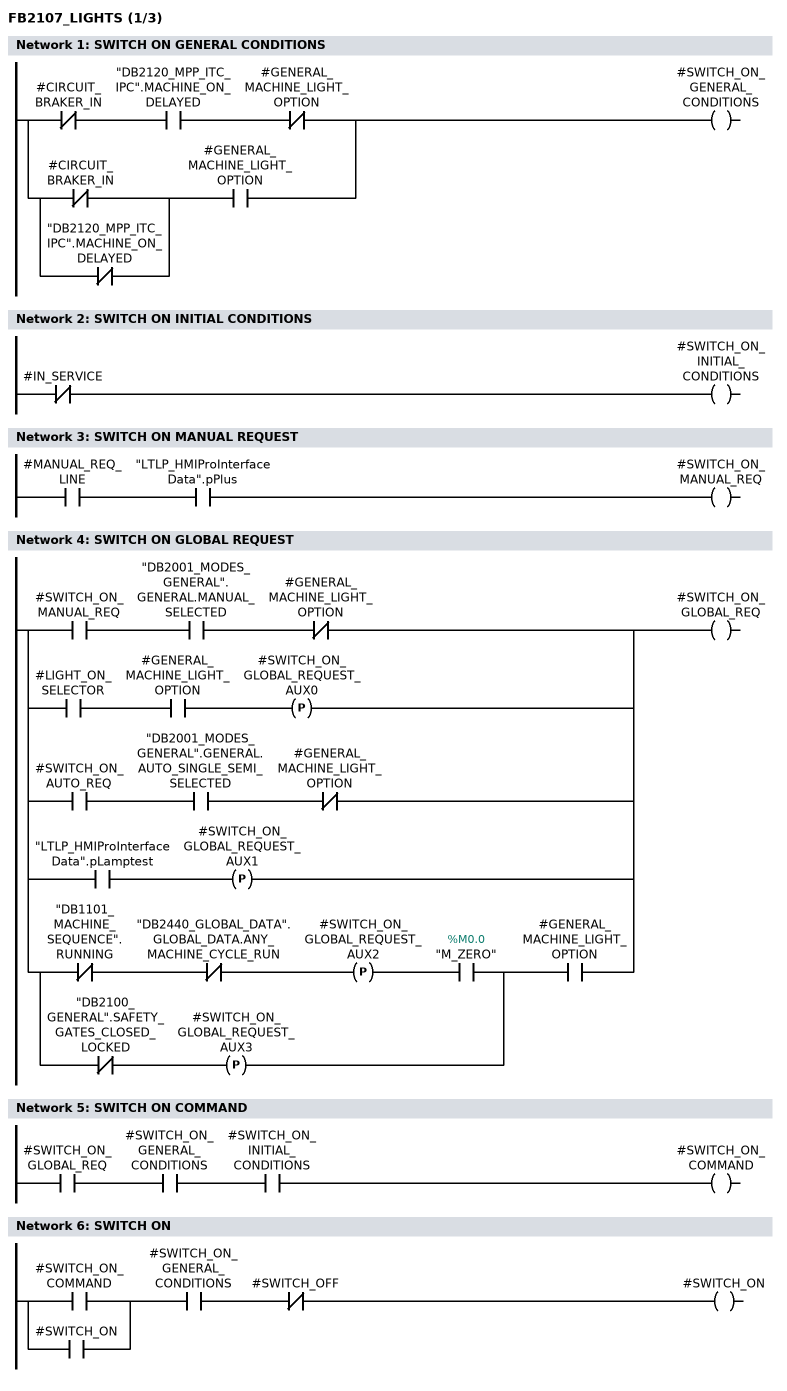
   RUNG wire#powerrail
      I_Contact( #CIRCUIT_BRAKER_IN )
      Contact( "DB2120_MPP_ITC_IPC".MACHINE_ON_DELAYED )
      I_Contact( #GENERAL_MACHINE_LIGHT_OPTION )
      wire#w1
      Coil( #SWITCH_ON_GENERAL_CONDITIONS )
   END_RUNG
   RUNG wire#powerrail
      I_Contact( #CIRCUIT_BRAKER_IN )
      wire#w2
      Contact( #GENERAL_MACHINE_LIGHT_OPTION )
   END_RUNG wire#w1
   RUNG wire#powerrail
      I_Contact( "DB2120_MPP_ITC_IPC".MACHINE_ON_DELAYED )
   END_RUNG wire#w2
   // the same network as SCL:
   #SWITCH_ON_GENERAL_CONDITIONS := (NOT #CIRCUIT_BRAKER_IN AND "DB2120_MPP_ITC_IPC".MACHINE_ON_DELAYED AND NOT #GENERAL_MACHINE_LIGHT_OPTION) OR ((NOT #CIRCUIT_BRAKER_IN OR NOT "DB2120_MPP_ITC_IPC".MACHINE_ON_DELAYED) AND #GENERAL_MACHINE_LIGHT_OPTION);
END_REGION

REGION Network 2: SWITCH ON INITIAL CONDITIONS
   RUNG wire#powerrail
      I_Contact( #IN_SERVICE )
      Coil( #SWITCH_ON_INITIAL_CONDITIONS )
   END_RUNG
   // the same network as SCL:
   #SWITCH_ON_INITIAL_CONDITIONS := NOT #IN_SERVICE;
END_REGION

REGION Network 3: SWITCH ON MANUAL REQUEST
   RUNG wire#powerrail
      Contact( #MANUAL_REQ_LINE )
      Contact( "LTLP_HMIProInterfaceData".pPlus )
      Coil( #SWITCH_ON_MANUAL_REQ )
   END_RUNG
   // the same network as SCL:
   #SWITCH_ON_MANUAL_REQ := #MANUAL_REQ_LINE AND "LTLP_HMIProInterfaceData".pPlus;
END_REGION

REGION Network 4: SWITCH ON GLOBAL REQUEST
   RUNG wire#powerrail
      Contact( #SWITCH_ON_MANUAL_REQ )
      Contact( "DB2001_MODES_GENERAL".GENERAL.MANUAL_SELECTED )
      I_Contact( #GENERAL_MACHINE_LIGHT_OPTION )
      wire#w1
      Coil( #SWITCH_ON_GLOBAL_REQ )
   END_RUNG
   RUNG wire#powerrail
      Contact( #LIGHT_ON_SELECTOR )
      Contact( #GENERAL_MACHINE_LIGHT_OPTION )
      P_Trig( #SWITCH_ON_GLOBAL_REQUEST_AUX0 )
   END_RUNG wire#w1
   RUNG wire#powerrail
      Contact( #SWITCH_ON_AUTO_REQ )
      Contact( "DB2001_MODES_GENERAL".GENERAL.AUTO_SINGLE_SEMI_SELECTED )
      I_Contact( #GENERAL_MACHINE_LIGHT_OPTION )
   END_RUNG wire#w1
   RUNG wire#powerrail
      Contact( "LTLP_HMIProInterfaceData".pLamptest )
      P_Trig( #SWITCH_ON_GLOBAL_REQUEST_AUX1 )
   END_RUNG wire#w1
   RUNG wire#powerrail
      I_Contact( "DB1101_MACHINE_SEQUENCE".RUNNING )
      I_Contact( "DB2440_GLOBAL_DATA".GLOBAL_DATA.ANY_MACHINE_CYCLE_RUN )
      P_Trig( #SWITCH_ON_GLOBAL_REQUEST_AUX2 )
      Contact( "M_ZERO" )
      wire#w2
      Contact( #GENERAL_MACHINE_LIGHT_OPTION )
   END_RUNG wire#w1
   RUNG wire#powerrail
      I_Contact( "DB2100_GENERAL".SAFETY_GATES_CLOSED_LOCKED )
      P_Trig( #SWITCH_ON_GLOBAL_REQUEST_AUX3 )
   END_RUNG wire#w2
   // the same network as SCL:
   #_w1 := #LIGHT_ON_SELECTOR AND #GENERAL_MACHINE_LIGHT_OPTION;
   #_w2 := #_w1 AND NOT #SWITCH_ON_GLOBAL_REQUEST_AUX0;   // rising edge
   #SWITCH_ON_GLOBAL_REQUEST_AUX0 := #_w1;
   #_w3 := "LTLP_HMIProInterfaceData".pLamptest AND NOT #SWITCH_ON_GLOBAL_REQUEST_AUX1;   // rising edge
   #SWITCH_ON_GLOBAL_REQUEST_AUX1 := "LTLP_HMIProInterfaceData".pLamptest;
   #_w4 := NOT "DB1101_MACHINE_SEQUENCE".RUNNING AND NOT "DB2440_GLOBAL_DATA".GLOBAL_DATA.ANY_MACHINE_CYCLE_RUN;
   #_w5 := #_w4 AND NOT #SWITCH_ON_GLOBAL_REQUEST_AUX2;   // rising edge
   #SWITCH_ON_GLOBAL_REQUEST_AUX2 := #_w4;
   #_w6 := NOT "DB2100_GENERAL".SAFETY_GATES_CLOSED_LOCKED AND NOT #SWITCH_ON_GLOBAL_REQUEST_AUX3;   // rising edge
   #SWITCH_ON_GLOBAL_REQUEST_AUX3 := NOT "DB2100_GENERAL".SAFETY_GATES_CLOSED_LOCKED;
   #SWITCH_ON_GLOBAL_REQ := (#SWITCH_ON_MANUAL_REQ AND "DB2001_MODES_GENERAL".GENERAL.MANUAL_SELECTED AND NOT #GENERAL_MACHINE_LIGHT_OPTION) OR #_w2 OR (#SWITCH_ON_AUTO_REQ AND "DB2001_MODES_GENERAL".GENERAL.AUTO_SINGLE_SEMI_SELECTED AND NOT #GENERAL_MACHINE_LIGHT_OPTION) OR #_w3 OR (((#_w5 AND "M_ZERO") OR #_w6) AND #GENERAL_MACHINE_LIGHT_OPTION);
END_REGION

REGION Network 5: SWITCH ON COMMAND
   RUNG wire#powerrail
      Contact( #SWITCH_ON_GLOBAL_REQ )
      Contact( #SWITCH_ON_GENERAL_CONDITIONS )
      Contact( #SWITCH_ON_INITIAL_CONDITIONS )
      Coil( #SWITCH_ON_COMMAND )
   END_RUNG
   // the same network as SCL:
   #SWITCH_ON_COMMAND := #SWITCH_ON_GLOBAL_REQ AND #SWITCH_ON_GENERAL_CONDITIONS AND #SWITCH_ON_INITIAL_CONDITIONS;
END_REGION

REGION Network 6: SWITCH ON
   RUNG wire#powerrail
      Contact( #SWITCH_ON_COMMAND )
      wire#w1
      Contact( #SWITCH_ON_GENERAL_CONDITIONS )
      I_Contact( #SWITCH_OFF )
      Coil( #SWITCH_ON )
   END_RUNG
   RUNG wire#powerrail
      Contact( #SWITCH_ON )
   END_RUNG wire#w1
   // the same network as SCL:
   #SWITCH_ON := (#SWITCH_ON_COMMAND OR #SWITCH_ON) AND #SWITCH_ON_GENERAL_CONDITIONS AND NOT #SWITCH_OFF;
END_REGION

REGION Network 7: IN SERVICE
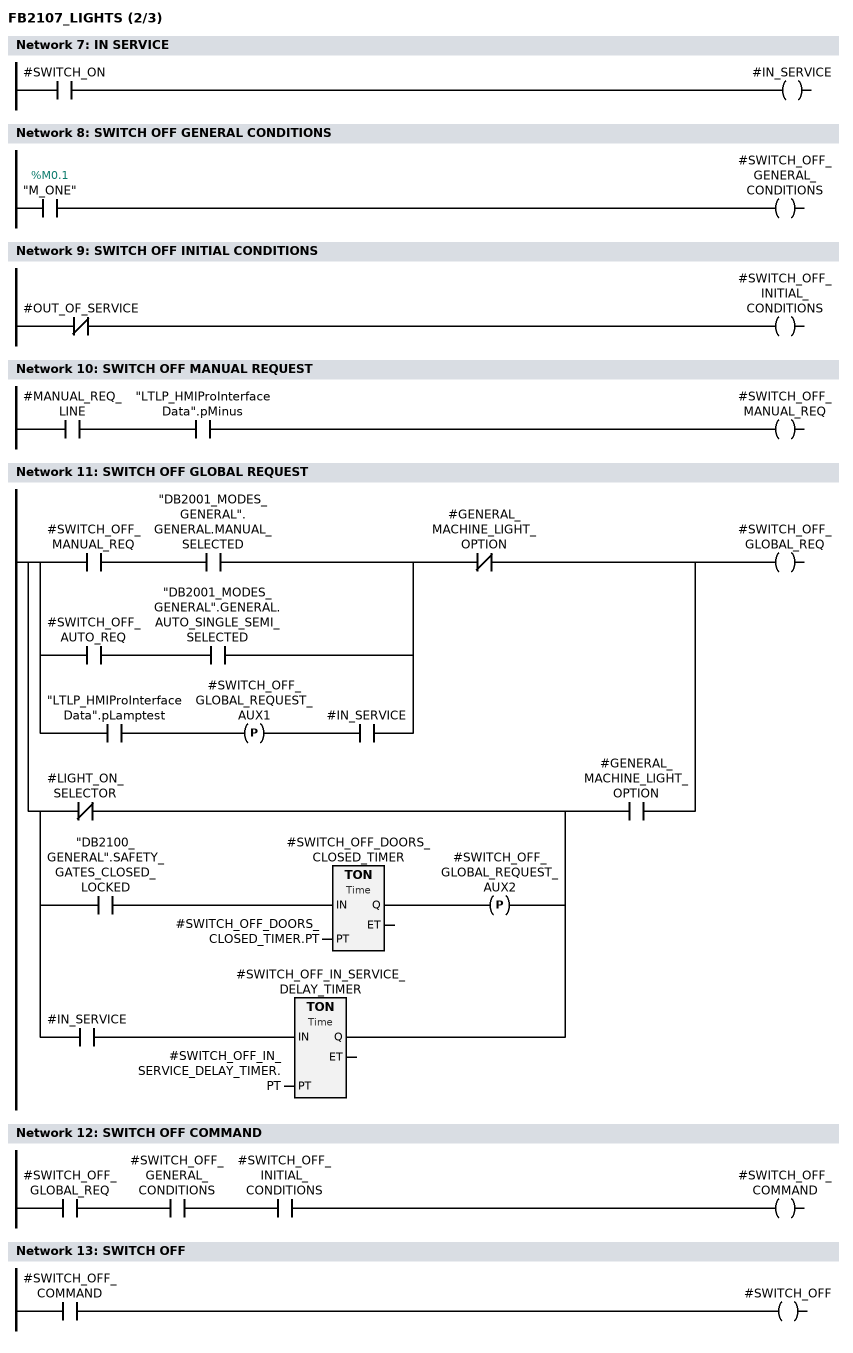
   RUNG wire#powerrail
      Contact( #SWITCH_ON )
      Coil( #IN_SERVICE )
   END_RUNG
   // the same network as SCL:
   #IN_SERVICE := #SWITCH_ON;
END_REGION

REGION Network 8: SWITCH OFF GENERAL CONDITIONS
   RUNG wire#powerrail
      Contact( "M_ONE" )
      Coil( #SWITCH_OFF_GENERAL_CONDITIONS )
   END_RUNG
   // the same network as SCL:
   #SWITCH_OFF_GENERAL_CONDITIONS := "M_ONE";
END_REGION

REGION Network 9: SWITCH OFF INITIAL CONDITIONS
   RUNG wire#powerrail
      I_Contact( #OUT_OF_SERVICE )
      Coil( #SWITCH_OFF_INITIAL_CONDITIONS )
   END_RUNG
   // the same network as SCL:
   #SWITCH_OFF_INITIAL_CONDITIONS := NOT #OUT_OF_SERVICE;
END_REGION

REGION Network 10: SWITCH OFF MANUAL REQUEST
   RUNG wire#powerrail
      Contact( #MANUAL_REQ_LINE )
      Contact( "LTLP_HMIProInterfaceData".pMinus )
      Coil( #SWITCH_OFF_MANUAL_REQ )
   END_RUNG
   // the same network as SCL:
   #SWITCH_OFF_MANUAL_REQ := #MANUAL_REQ_LINE AND "LTLP_HMIProInterfaceData".pMinus;
END_REGION

REGION Network 11: SWITCH OFF GLOBAL REQUEST
   RUNG wire#powerrail
      Contact( #SWITCH_OFF_MANUAL_REQ )
      Contact( "DB2001_MODES_GENERAL".GENERAL.MANUAL_SELECTED )
      wire#w1
      I_Contact( #GENERAL_MACHINE_LIGHT_OPTION )
      wire#w2
      Coil( #SWITCH_OFF_GLOBAL_REQ )
   END_RUNG
   RUNG wire#powerrail
      Contact( #SWITCH_OFF_AUTO_REQ )
      Contact( "DB2001_MODES_GENERAL".GENERAL.AUTO_SINGLE_SEMI_SELECTED )
   END_RUNG wire#w1
   RUNG wire#powerrail
      Contact( "LTLP_HMIProInterfaceData".pLamptest )
      P_Trig( #SWITCH_OFF_GLOBAL_REQUEST_AUX1 )
      Contact( #IN_SERVICE )
   END_RUNG wire#w1
   RUNG wire#powerrail
      I_Contact( #LIGHT_ON_SELECTOR )
      wire#w3
      Contact( #GENERAL_MACHINE_LIGHT_OPTION )
   END_RUNG wire#w2
   RUNG wire#powerrail
      Contact( "DB2100_GENERAL".SAFETY_GATES_CLOSED_LOCKED )
      { S7_Templates := "time_type := Time" } #SWITCH_OFF_DOORS_CLOSED_TIMER.TON(pt := #SWITCH_OFF_DOORS_CLOSED_TIMER.PT, et =>)
      P_Trig( #SWITCH_OFF_GLOBAL_REQUEST_AUX2 )
   END_RUNG wire#w3
   RUNG wire#powerrail
      Contact( #IN_SERVICE )
      { S7_Templates := "time_type := Time" } #SWITCH_OFF_IN_SERVICE_DELAY_TIMER.TON(pt := #SWITCH_OFF_IN_SERVICE_DELAY_TIMER.PT, et =>)
   END_RUNG wire#w3
   // the same network as SCL:
   #_w1 := "LTLP_HMIProInterfaceData".pLamptest AND NOT #SWITCH_OFF_GLOBAL_REQUEST_AUX1;   // rising edge
   #SWITCH_OFF_GLOBAL_REQUEST_AUX1 := "LTLP_HMIProInterfaceData".pLamptest;
   #SWITCH_OFF_DOORS_CLOSED_TIMER.TON(IN := "DB2100_GENERAL".SAFETY_GATES_CLOSED_LOCKED,
                           PT := #SWITCH_OFF_DOORS_CLOSED_TIMER.PT);
   #_w2 := #SWITCH_OFF_DOORS_CLOSED_TIMER.Q AND NOT #SWITCH_OFF_GLOBAL_REQUEST_AUX2;   // rising edge
   #SWITCH_OFF_GLOBAL_REQUEST_AUX2 := #SWITCH_OFF_DOORS_CLOSED_TIMER.Q;
   #SWITCH_OFF_IN_SERVICE_DELAY_TIMER.TON(IN := #IN_SERVICE, PT := #SWITCH_OFF_IN_SERVICE_DELAY_TIMER.PT);
   #SWITCH_OFF_GLOBAL_REQ := (((#SWITCH_OFF_MANUAL_REQ AND "DB2001_MODES_GENERAL".GENERAL.MANUAL_SELECTED) OR (#SWITCH_OFF_AUTO_REQ AND "DB2001_MODES_GENERAL".GENERAL.AUTO_SINGLE_SEMI_SELECTED) OR (#_w1 AND #IN_SERVICE)) AND NOT #GENERAL_MACHINE_LIGHT_OPTION) OR ((NOT #LIGHT_ON_SELECTOR OR #_w2 OR #SWITCH_OFF_IN_SERVICE_DELAY_TIMER.Q) AND #GENERAL_MACHINE_LIGHT_OPTION);
END_REGION

REGION Network 12: SWITCH OFF COMMAND
   RUNG wire#powerrail
      Contact( #SWITCH_OFF_GLOBAL_REQ )
      Contact( #SWITCH_OFF_GENERAL_CONDITIONS )
      Contact( #SWITCH_OFF_INITIAL_CONDITIONS )
      Coil( #SWITCH_OFF_COMMAND )
   END_RUNG
   // the same network as SCL:
   #SWITCH_OFF_COMMAND := #SWITCH_OFF_GLOBAL_REQ AND #SWITCH_OFF_GENERAL_CONDITIONS AND #SWITCH_OFF_INITIAL_CONDITIONS;
END_REGION

REGION Network 13: SWITCH OFF
   RUNG wire#powerrail
      Contact( #SWITCH_OFF_COMMAND )
      Coil( #SWITCH_OFF )
   END_RUNG
   // the same network as SCL:
   #SWITCH_OFF := #SWITCH_OFF_COMMAND;
END_REGION

REGION Network 14: OUT OF SERVICE
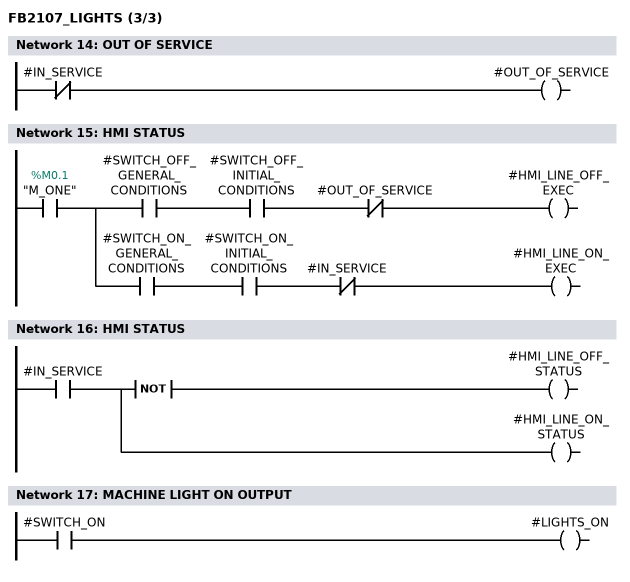
   RUNG wire#powerrail
      I_Contact( #IN_SERVICE )
      Coil( #OUT_OF_SERVICE )
   END_RUNG
   // the same network as SCL:
   #OUT_OF_SERVICE := NOT #IN_SERVICE;
END_REGION

REGION Network 15: HMI STATUS
   RUNG wire#powerrail
      Contact( "M_ONE" )
      wire#w1
      Contact( #SWITCH_OFF_GENERAL_CONDITIONS )
      Contact( #SWITCH_OFF_INITIAL_CONDITIONS )
      I_Contact( #OUT_OF_SERVICE )
      Coil( #HMI_LINE_OFF_EXEC )
   END_RUNG
   RUNG wire#w1
      Contact( #SWITCH_ON_GENERAL_CONDITIONS )
      Contact( #SWITCH_ON_INITIAL_CONDITIONS )
      I_Contact( #IN_SERVICE )
      Coil( #HMI_LINE_ON_EXEC )
   END_RUNG
   // the same network as SCL:
   #HMI_LINE_OFF_EXEC := "M_ONE" AND #SWITCH_OFF_GENERAL_CONDITIONS AND #SWITCH_OFF_INITIAL_CONDITIONS AND NOT #OUT_OF_SERVICE;
   #HMI_LINE_ON_EXEC := "M_ONE" AND #SWITCH_ON_GENERAL_CONDITIONS AND #SWITCH_ON_INITIAL_CONDITIONS AND NOT #IN_SERVICE;
END_REGION

REGION Network 16: HMI STATUS
   RUNG wire#powerrail
      Contact( #IN_SERVICE )
      wire#w1
      Not()
      Coil( #HMI_LINE_OFF_STATUS )
   END_RUNG
   RUNG wire#w1
      Coil( #HMI_LINE_ON_STATUS )
   END_RUNG
   // the same network as SCL:
   #HMI_LINE_OFF_STATUS := NOT #IN_SERVICE;
   #HMI_LINE_ON_STATUS := #IN_SERVICE;
END_REGION

REGION Network 17: MACHINE LIGHT ON OUTPUT
   RUNG wire#powerrail
      Contact( #SWITCH_ON )
      Coil( #LIGHTS_ON )
   END_RUNG
   // the same network as SCL:
   #LIGHTS_ON := #SWITCH_ON;
END_REGION
END_FUNCTION_BLOCK

FUNCTION_BLOCK "FB2123_PANEL_BUTTON"   // FB2123, LAD
{ S7_Optimized_Access := 'FALSE' }
AUTHOR : ETXETAR
VERSION : 1.0
// stored: AutoNumber false, IsIECCheckEnabled false, SetENOAutomatically false, UDAEnableTagReadback false
   VAR_INPUT
      OPTIONS_0 : Byte := 2#0000_0000;   // OPTIONS 0
      START_CYCLE : Bool;   // START CYCLE / INPUT START CYCLE
      STOP_END_CYCLE : Bool;   // STOP END OF CYCLE / INPUT STOP END CYCLE
      IMMEDIATE_STOP : Bool;   // INMEDIATE STOP / INPUT IMMEDIATE STOP
      EMERGENCY_STOP : Bool;   // EMERGENCY STOP / INPUT EMERGENCY STOP
      HOME_POSITION : Bool;   // INPUT HOME POSITION
      RESET_FAULT : Bool;   // RESET FAULT / INPUT RESET FAULT
      AUTO_SELECTOR : Bool;   // INPUT SELECTOR AUTO SELECTED
      MANUAL_LOAD_SELECTOR : Bool;   // INPUT SELECTOR MANUAL LOAD SELECTED
      LOCK_UNLOCK_GATES : Bool;   // LOCK UNLOCK GATES / INPUT LOCK UNLOCK GATES
      DOOR_LAMP_COND : Bool;   // INPUT DOOR LAMP CONDITIONS
      BHG_BYPASS_GATES : Bool;   // BY PASSED SAFETY GATES MAIN PANEL / INPUT BHG BYPASS GATES
      UNLOAD_PARTS : Bool;   // INPUT UNLOAD FIXTURE PARTS
      UNLOAD_PARTS_FIXT_COND : Bool;   // INPUT UNLOAD PARTS FIXTURE CONDITIONS
      LOAD_PARTS : Bool;   // INPUT LOAD FIXTURE PARTS
      LOAD_PARTS_FIXT_COND : Bool;   // INPUT LOAD PARTS FIXTURE CONDITIONS
   END_VAR
   VAR_OUTPUT
      START_CYCLE_LAMP : Bool;   // START CYCLE LAMP
      END_OF_CYCLE_LAMP : Bool;   // END OF CYCLE LAMP
      HOME_LAMP : Bool;   // HOME POSITION LAMP
      RESET_LAMP : Bool;   // RESET LAMP
      LOCK_DOOR_LAMP : Bool;   // LOCK DOOR LAMP
      UNLOAD_LAMP : Bool;   // UNLOAD PARTS LAMP
      LOAD_LAMP : Bool;   // LOAD PARTS LAMP
      EMERGENCY_STOP_ALARM : Bool;   // EMERGENCY STOP FAULT / EMERGENCY STOP ALARM
   END_VAR
   VAR DB_SPECIFIC
      MANUAL_REQUEST : Bool;   // MANUAL REQUEST
      SEMI_REQUEST : Bool;   // SEMI REQUEST
      AUTO_REQUEST : Bool;   // AUTO REQUEST
      SETUP_REQUEST : Bool;   // SETUP REQUEST
      PARTS_UNLOADED : Bool;   // PARTS UNLOADED
      PARTS_LOADED : Bool;   // PARTS LOADED
      END_OF_CYCLE_ALARM : Bool;   // END OF CYCLE ALARM
      IMMEDIATE_STOP_ALARM : Bool;   // IMMEDIATE STOP ALARM
      HOME_POSITION_ALARM : Bool;   // HOME POSITION ALARM
      SEOC_BY_OPERATOR : Bool;   // STOP END OF CYCLE BY OPERATOR / SEOC BY OPERATOR
      MANUAL_LOADING_SEL_BUTTO : Bool;   // MANUAL LOADING SELECTOR BUTTON / MANUAL LOADING SEL BUTTO
      WARNING_GONE : Bool;   // WARNING GONE
      E_RETURN_PULSE : Bool;   // EMERGENCY RETURN PULSE
      AUX1 : Bool;   // AUX1
      AUX2 : Bool;   // AUX2
      AUX3 : Bool;   // AUX3
      AUX4 : Bool;   // AUX4
      CONDITION_HELP : Bool;   // CONDITION HELP
   END_VAR
   VAR_TEMP
      INPUTS_MASK : Byte;   // INPUT MASK
      O_BYTE_0 : Struct   // OPTIONS BYTE 0
         CHANGE_MODE_WO_PANEL_ACTIVE : Bool;   // CHANGE MODE WITHOUT PANEL ACTIVE OPTION
         MAGAZINE_PANEL : Bool;   // MAGAZINE PANEL OPTION
         PHD_PANEL : Bool;   // PART HANDLING DEVICE PANEL OPTION
         BIMANUAL_PANEL : Bool;   // SPARE OPTION
         SPARE_4 : Bool;   // SPARE OPTION
         SPARE_5 : Bool;   // SPARE OPTION
         SPARE_6 : Bool;   // SPARE OPTION
         SPARE_7 : Bool;   // SPARE OPTION
      END_STRUCT;
      DB_NUMBER : DInt;   // DB NUMBER FOR ALARM AND HELP DECODING
   END_VAR
   VAR_TEMP   // added for the SCL form of the ladder/FBD networks
      _w1 : Bool;
      _w2 : Bool;
      _w3 : Bool;
   END_VAR
BEGIN

NETWORK
TITLE = READ INSTANCE DB
      L     DINO;
      +     10#800000;
      T     #DB_NUMBER;


REGION Network 2: OPTIONS
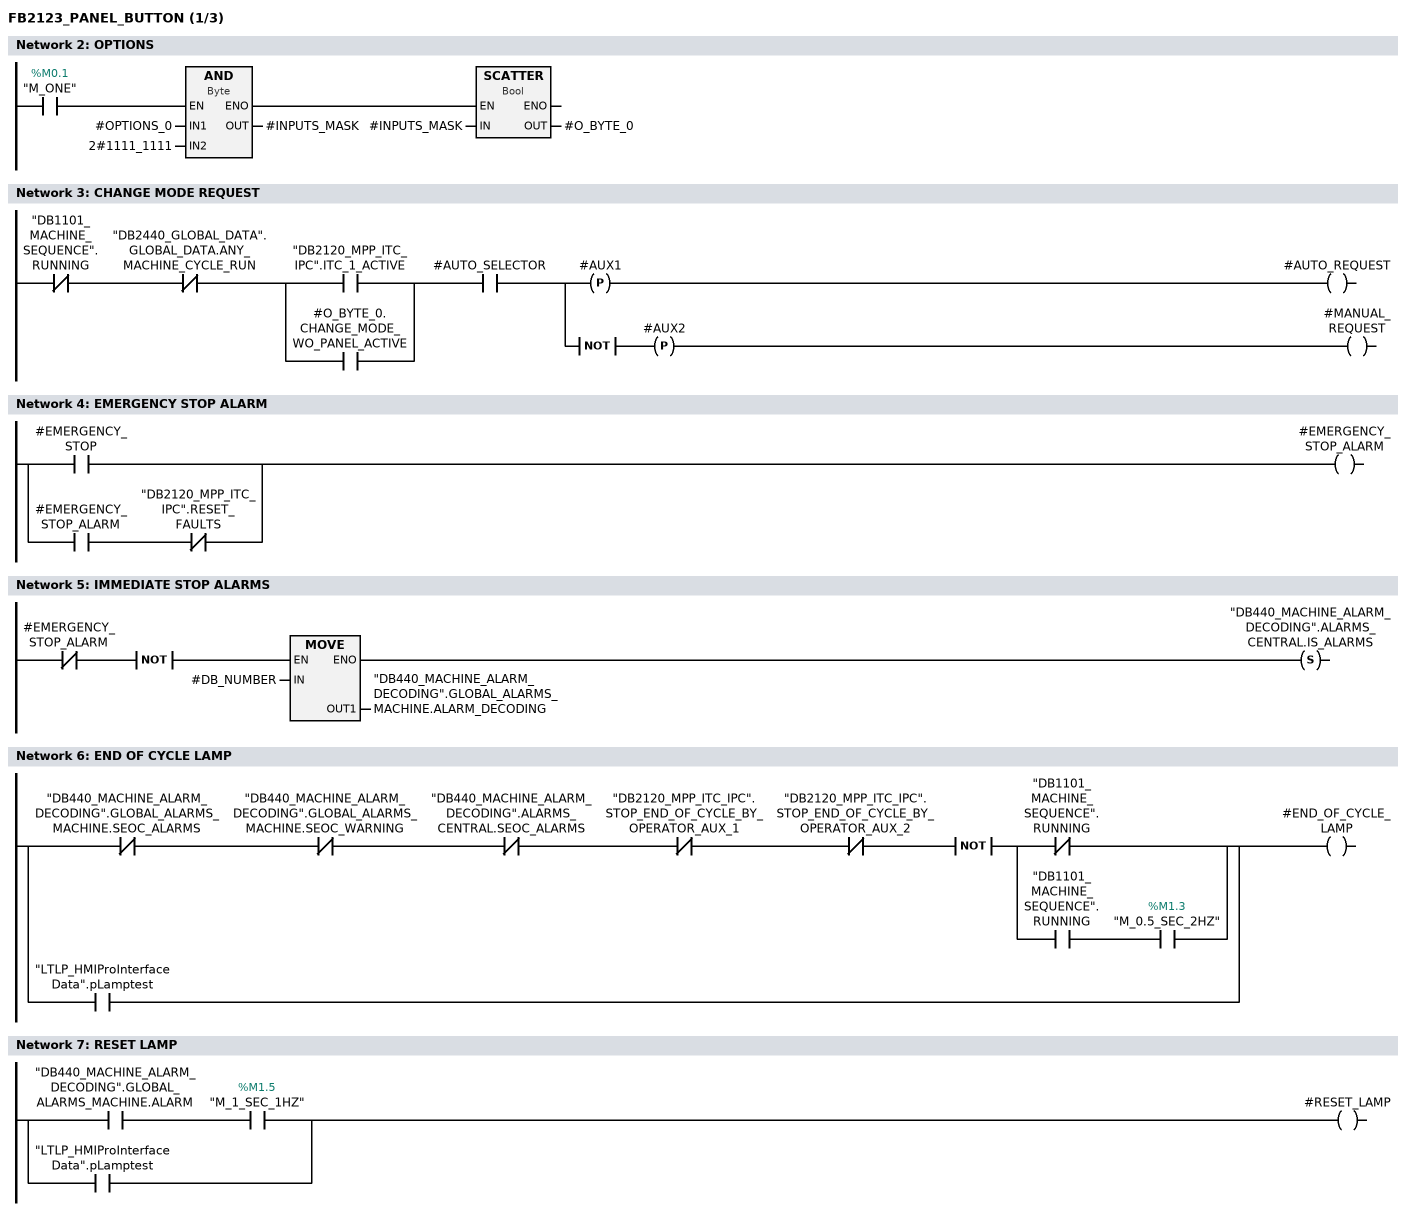
   RUNG wire#powerrail
      Contact( "M_ONE" )
      { S7_Templates := "SrcType := Byte"; S7_GenerateENO := "TRUE" } And(in1 := #OPTIONS_0, in2 := 2#1111_1111, out => #INPUTS_MASK)
      { S7_Templates := "[dest_type := Bool, src_type := Byte]" } SCATTER(IN := #INPUTS_MASK, OUT => #O_BYTE_0)
   END_RUNG
   // the same network as SCL:
   IF "M_ONE" THEN
       #INPUTS_MASK := #OPTIONS_0 AND 2#1111_1111;
       SCATTER(IN := #INPUTS_MASK, OUT => #O_BYTE_0);
   END_IF;
END_REGION

REGION Network 3: CHANGE MODE REQUEST
   RUNG wire#powerrail
      I_Contact( "DB1101_MACHINE_SEQUENCE".RUNNING )
      I_Contact( "DB2440_GLOBAL_DATA".GLOBAL_DATA.ANY_MACHINE_CYCLE_RUN )
      wire#w1
      Contact( "DB2120_MPP_ITC_IPC".ITC_1_ACTIVE )
      wire#w2
      Contact( #AUTO_SELECTOR )
      wire#w3
      P_Trig( #AUX1 )
      Coil( #AUTO_REQUEST )
   END_RUNG
   RUNG wire#w1
      Contact( #O_BYTE_0.CHANGE_MODE_WO_PANEL_ACTIVE )
   END_RUNG wire#w2
   RUNG wire#w3
      Not()
      P_Trig( #AUX2 )
      Coil( #MANUAL_REQUEST )
   END_RUNG
   // the same network as SCL:
   #_w1 := NOT "DB1101_MACHINE_SEQUENCE".RUNNING AND NOT "DB2440_GLOBAL_DATA".GLOBAL_DATA.ANY_MACHINE_CYCLE_RUN AND ("DB2120_MPP_ITC_IPC".ITC_1_ACTIVE OR #O_BYTE_0.CHANGE_MODE_WO_PANEL_ACTIVE) AND #AUTO_SELECTOR;
   #_w2 := #_w1 AND NOT #AUX1;   // rising edge
   #AUX1 := #_w1;
   #AUTO_REQUEST := #_w2;
   #_w3 := NOT #_w1 AND NOT #AUX2;   // rising edge
   #AUX2 := NOT #_w1;
   #MANUAL_REQUEST := #_w3;
END_REGION

REGION Network 4: EMERGENCY STOP ALARM
   RUNG wire#powerrail
      Contact( #EMERGENCY_STOP )
      wire#w1
      Coil( #EMERGENCY_STOP_ALARM )
   END_RUNG
   RUNG wire#powerrail
      Contact( #EMERGENCY_STOP_ALARM )
      I_Contact( "DB2120_MPP_ITC_IPC".RESET_FAULTS )
   END_RUNG wire#w1
   // the same network as SCL:
   #EMERGENCY_STOP_ALARM := #EMERGENCY_STOP OR (#EMERGENCY_STOP_ALARM AND NOT "DB2120_MPP_ITC_IPC".RESET_FAULTS);
END_REGION

REGION Network 5: IMMEDIATE STOP ALARMS
   RUNG wire#powerrail
      I_Contact( #EMERGENCY_STOP_ALARM )
      Not()
      { S7_GenerateENO := "TRUE" } Move(in := #DB_NUMBER, out1 => "DB440_MACHINE_ALARM_DECODING".GLOBAL_ALARMS_MACHINE.ALARM_DECODING)
      S_Coil( "DB440_MACHINE_ALARM_DECODING".ALARMS_CENTRAL.IS_ALARMS )
   END_RUNG
   // the same network as SCL:
   // ENO of a box is taken as its EN; it also drops when the box reports an error
   IF NOT (NOT #EMERGENCY_STOP_ALARM) THEN
       "DB440_MACHINE_ALARM_DECODING".GLOBAL_ALARMS_MACHINE.ALARM_DECODING := #DB_NUMBER;
       "DB440_MACHINE_ALARM_DECODING".ALARMS_CENTRAL.IS_ALARMS := TRUE;
   END_IF;
END_REGION

REGION Network 6: END OF CYCLE LAMP
   RUNG wire#powerrail
      I_Contact( "DB440_MACHINE_ALARM_DECODING".GLOBAL_ALARMS_MACHINE.SEOC_ALARMS )
      I_Contact( "DB440_MACHINE_ALARM_DECODING".GLOBAL_ALARMS_MACHINE.SEOC_WARNING )
      I_Contact( "DB440_MACHINE_ALARM_DECODING".ALARMS_CENTRAL.SEOC_ALARMS )
      I_Contact( "DB2120_MPP_ITC_IPC".STOP_END_OF_CYCLE_BY_OPERATOR_AUX_1 )
      I_Contact( "DB2120_MPP_ITC_IPC".STOP_END_OF_CYCLE_BY_OPERATOR_AUX_2 )
      Not()
      wire#w1
      I_Contact( "DB1101_MACHINE_SEQUENCE".RUNNING )
      wire#w2
      Coil( #END_OF_CYCLE_LAMP )
   END_RUNG
   RUNG wire#w1
      Contact( "DB1101_MACHINE_SEQUENCE".RUNNING )
      Contact( "M_0.5_SEC_2HZ" )
   END_RUNG wire#w2
   RUNG wire#powerrail
      Contact( "LTLP_HMIProInterfaceData".pLamptest )
   END_RUNG wire#w2
   // the same network as SCL:
   #END_OF_CYCLE_LAMP := (NOT (NOT "DB440_MACHINE_ALARM_DECODING".GLOBAL_ALARMS_MACHINE.SEOC_ALARMS AND NOT "DB440_MACHINE_ALARM_DECODING".GLOBAL_ALARMS_MACHINE.SEOC_WARNING AND NOT "DB440_MACHINE_ALARM_DECODING".ALARMS_CENTRAL.SEOC_ALARMS AND NOT "DB2120_MPP_ITC_IPC".STOP_END_OF_CYCLE_BY_OPERATOR_AUX_1 AND NOT "DB2120_MPP_ITC_IPC".STOP_END_OF_CYCLE_BY_OPERATOR_AUX_2) AND (NOT "DB1101_MACHINE_SEQUENCE".RUNNING OR ("DB1101_MACHINE_SEQUENCE".RUNNING AND "M_0.5_SEC_2HZ"))) OR "LTLP_HMIProInterfaceData".pLamptest;
END_REGION

REGION Network 7: RESET LAMP
   RUNG wire#powerrail
      Contact( "DB440_MACHINE_ALARM_DECODING".GLOBAL_ALARMS_MACHINE.ALARM )
      Contact( "M_1_SEC_1HZ" )
      wire#w1
      Coil( #RESET_LAMP )
   END_RUNG
   RUNG wire#powerrail
      Contact( "LTLP_HMIProInterfaceData".pLamptest )
   END_RUNG wire#w1
   // the same network as SCL:
   #RESET_LAMP := ("DB440_MACHINE_ALARM_DECODING".GLOBAL_ALARMS_MACHINE.ALARM AND "M_1_SEC_1HZ") OR "LTLP_HMIProInterfaceData".pLamptest;
END_REGION

